(* PLC project marvel_common, Institute of Astronomy Onto 0.0.1 *)
(* stored: creationDateTime 2025-01-01T00:00:00.0, modificationDateTime 2025-01-01T00:00:00.0 *)

{attribute 'qualified_only'}
TYPE InitializationStates : (SHUTDOWN := 0, INITIALIZING := 1, INITIALIZING_FAILED := 2, INITIALIZED := 3, LOCKED := 4);
END_TYPE

{attribute 'qualified_only'}
TYPE OperatorStates : (NONE := 0, OBSERVER := 1, TECH := 2);
END_TYPE

{attribute 'qualified_only'}
TYPE OperatingStates : (AUTO := 0, MANUAL := 1);
END_TYPE

{attribute 'qualified_only'}
TYPE OperatingModeStates : (LOCAL := 0, REMOTE := 1);
END_TYPE

{attribute 'qualified_only'}
TYPE LimitSwitches : (POSITIVE_LIMIT_SWITCH := 0, NEGATIVE_LIMIT_SWITCH := 1);
END_TYPE

{attribute 'qualified_only'}
TYPE Units : (DEGREE := 0, RADIAN := 1, PERCENT := 2, RADIANS_PER_SECOND := 3, DEGREES_PER_SECOND := 4, MILLIMETERS_PER_SECOND := 5, REVOLUTIONS_PER_SECOND := 6, REVOLUTIONS_PER_MINUTE := 7, AMPS := 8, MILLIAMPS := 9, MILLIMETER := 10, MICROMETER := 11, DEGREES_CELSIUS := 12, KELVIN := 13, BAR := 14, PASCAL := 15, UNITLESS := 16, NEWTON := 17, DECANEWTON := 18, VOLT := 19, MILLIVOLT := 20, HERTZ := 21, G := 22, MILLIG := 23, NEWTONMETER := 24, ARCSECONDS := 25, ARCSECONDS_PER_SECOND := 26, RADIANS_PER_SQUARE_SECOND := 27, DEGREES_PER_SQUARE_SECOND := 28, ARCSECONDS_PER_SQUARE_SECOND := 29, METERS_PER_SECOND := 30, HECTOPASCAL := 31, SECONDS := 32, MINUTES := 33, MILLIMETERS_PER_HOUR := 34, HITS_PER_SQUARE_CENTIMETER := 35, HITS_PER_SQUARE_CENTIMETER_PER_HOUR := 36);
END_TYPE

{attribute 'qualified_only'}
TYPE RequestResults : (ACCEPTED := 0, REJECTED := 1);
END_TYPE

{attribute 'qualified_only'}
TYPE ApertureStatus : (unknown := 0, invalid_model := 1, open := 2, closed := 3, partiallyOpen := 4, undefined := 5) BYTE;
END_TYPE

{attribute 'qualified_only'}
TYPE BusyStatus : (unknown := 0, invalid_model := 1, idle := 2, busy := 3) BYTE;
END_TYPE

{attribute 'qualified_only'}
TYPE StartedStatus : (unknown := 0, invalid_model := 1, started := 2, notStarted := 3) BYTE;
END_TYPE

{attribute 'qualified_only'}
TYPE EnabledStatus : (unknown := 0, invalid_model := 1, enabled := 2, disabled := 3) BYTE;
END_TYPE

{attribute 'qualified_only'}
TYPE PoweredStatus : (unknown := 0, invalid_model := 1, enabled := 2, disabled := 3) BYTE;
END_TYPE

{attribute 'qualified_only'}
TYPE HealthStatus : (unknown := 0, invalid_model := 1, good := 2, warning := 3, bad := 4) BYTE;
END_TYPE

{attribute 'qualified_only'}
TYPE InitializationStatus : (unknown := 0, invalid_model := 1, shutdown := 2, initializing := 3, initializingFailed := 4, initialized := 5, locked := 6) BYTE;
END_TYPE

{attribute 'qualified_only'}
TYPE MotionStatus : (unknown := 0, invalid_model := 1, forward := 2, backward := 3, standstill := 4) BYTE;
END_TYPE

{attribute 'qualified_only'}
TYPE HiHiLoLoAlarmStatus : (unknown := 0, invalid_model := 1, disabled := 2, hiHi := 3, hi := 4, ok := 5, lo := 6, loLo := 7) BYTE;
END_TYPE

{attribute 'qualified_only'}
TYPE OpeningStatus : (unknown := 0, invalid_model := 1, opening := 2, closing := 3, standstill := 4) BYTE;
END_TYPE

{attribute 'qualified_only'}
TYPE OperatorStatus : (unknown := 0, invalid_model := 1, none := 2, tech := 3, observer := 4) BYTE;
END_TYPE

{attribute 'qualified_only'}
TYPE OperatingStatus : (unknown := 0, invalid_model := 1, auto := 2, manual := 3) BYTE;
END_TYPE

{attribute 'qualified_only'}
TYPE OperatingModeStatus : (unknown := 0, invalid_model := 1, local := 2, remote := 3) BYTE;
END_TYPE

{attribute 'qualified_only'}
TYPE ActivityStatus : (unknown := 0, invalid_model := 1, notRunning := 2, running := 3) BYTE;
END_TYPE

{attribute 'qualified_only'}
TYPE GigECameraParams : (_NONE_ := 0, fExposureTime := 1, fAcquisitionFrameRate := 2, fLinkAcquisitionFrameRate := 3, nGainSelector := 4, fGain := 5, nWidth := 6, nHeight := 7, nWidthMax := 8, nHeightMax := 9, nOffsetX := 10, nOffsetY := 11, nBinningSelector := 12, nBinningHorizontal := 13, nBinningVertical := 14, nTriggerSelector := 15, nTriggerMode := 16, fDeviceTemperature := 17, nAcquisitionMode := 18, fBlackLevel := 19, nBlackLevelAuto := 20, _END_ := 21);
END_TYPE

{attribute 'qualified_only'}
TYPE GigECameraSources : (CAMERA := 0, ACQUISITION_EXAMPLE := 1);
END_TYPE

{attribute 'qualified_only'}
TYPE GigECameraMultiTriggerAlgorithms : (SUM := 0);
END_TYPE

{attribute 'qualified_only'}
TYPE ELL14Command : (HOME_FWD := 0, HOME_BWD := 1, SEARCHFREQ_MOT1 := 2, SEARCHFREQ_MOT2 := 3, GET_STATUS := 4, GET_POSITION := 5, MOVE_ABS := 6, MOVE_REL := 7, CUSTOM := 8, _END_ := 9);
END_TYPE

{attribute 'qualified_only'}
TYPE ELL14StatusCode : (OK := 0, COMM_TIMEOUT := 1, MECH_TIMEOUT := 2, CMD_ERROR := 3, VALUE_OUT_OF_RANGE := 4, MOD_ISOLATED := 5, MOD_OUT_OF_ISOLATION := 6, INIT_ERROR := 7, THERMAL_ERROR := 8, BUSY := 9, SENSOR_ERROR := 10, MOTOR_ERROR := 11, OUT_OF_RANGE := 12, OVERCURRENT_ERROR := 13, UNKNOWN := 14);
END_TYPE

{attribute 'qualified_only'}
TYPE ActionActor : (NONE := 0, SEQUENCER := 1, MARVEL := 2, U := 3, U_DOME := 4, U_DOME_SHUTTER := 5, U_DOME_ROTATION := 6, U_TELESCOPE := 7, U_TELESCOPE_COVER := 8, U_TELESCOPE_M2 := 9, U_TELESCOPE_M3 := 10, U_FEM := 11, U_FEM_PWR_GUIDECAM := 12, U_FEM_PWR_FIBREVIEWCAM := 13, U_FEM_PWR_ADC := 14, U_FEM_PWR_TIPTILT := 15, U_FEM_CALMIRROR := 16, U_FEM_ADC1 := 17, U_FEM_ADC2 := 18, U_FEM_FIBRESELECTOR := 19, U_FEM_LED_HGF := 20, U_FEM_LED_UGF := 21, U_FEM_LED_HSF := 22, U_FEM_LED_USF := 23, U_FEM_GUIDECAM := 24, U_FEM_FIBREVIEWCAM := 25, U_FEM_TIPTILT := 26, _END_ := 27);
END_TYPE

{attribute 'qualified_only'}
TYPE ActionKind : (NONE := 0, SLEEP := 1, WAIT_FOR_COMPLETION := 2, INITIALIZE := 3, OPEN := 4, CLOSE := 5, STOP := 6, MOVE_TO_NUMBER := 7, MOVE_ABS_MM := 8, MOVE_ABS_DEG := 9, MOVE_AZI_ELE := 10, ENABLE := 11, DISABLE := 12, SET_ENABLED := 13, MOVE_REL_MM := 14, MOVE_REL_DEG := 15, SET_CURRENT := 16, SET_VOLTAGE := 17, SET_AXIS_VOLTAGE := 18, POWER := 19, _END_ := 20);
END_TYPE

{attribute 'qualified_only'}
TYPE ActionStatus : (IDLE := 0, REQUESTED := 1, BUSY := 2, DONE_SUCCESS := 3, DONE_ERROR := 4, DONE_ERROR_ABORTED := 5, DONE_ERROR_PROCESS_FAILED := 6, DONE_ERROR_INVALID_TYPE := 7, DONE_ERROR_INVALID_ARG := 8, DONE_ERROR_INVALID_ACTOR := 9);
END_TYPE

TYPE SequencerParts : STRUCT
  {attribute 'TcHmiSymbol.Show'}
  configManager : ConfigManager;  (* The config manager (to load/save/activate configuration data) *)
END_STRUCT;
END_TYPE

TYPE BaseAxisProcesses : STRUCT
  {attribute 'TcHmiSymbol.Show'}
  moveAbsolute : McMoveAbsoluteProcess;  (* Move absolute *)
  {attribute 'TcHmiSymbol.Show'}
  moveRelative : McMoveRelativeProcess;  (* Move relative *)
  {attribute 'TcHmiSymbol.Show'}
  moveVelocity : McMoveVelocityProcess;  (* Move at a constant velocity *)
  {attribute 'TcHmiSymbol.Show'}
  reset : McProcess;  (* Reset any errors *)
  {attribute 'TcHmiSymbol.Show'}
  stop : McProcess;  (* Stop any movement *)
  {attribute 'TcHmiSymbol.Show'}
  stopParametrized : McStopProcess;  (* Stop any movement *)
  {attribute 'TcHmiSymbol.Show'}
  power : McPowerProcess;  (* Power on/off the axis *)
  {attribute 'TcHmiSymbol.Show'}
  home : McProcess;  (* Peform a homing *)
  {attribute 'TcHmiSymbol.Show'}
  initialize : Process;  (* Start initializing the axis *)
  {attribute 'TcHmiSymbol.Show'}
  setPosition : McSetPositionProcess;  (* Set the axis position *)
  {attribute 'TcHmiSymbol.Show'}
  readParameter : McReadParameter;  (* Read a numerical parameter *)
  {attribute 'TcHmiSymbol.Show'}
  readBoolParameter : McReadBoolParameter;  (* Read a boolean parameter *)
  {attribute 'TcHmiSymbol.Show'}
  writeParameter : McWriteParameter;  (* Write a numerical parameter *)
  {attribute 'TcHmiSymbol.Show'}
  writeBoolParameter : McWriteBoolParameter;  (* Write a boolean parameter *)
END_STRUCT;
END_TYPE

TYPE IncrementalEncoderProcesses : STRUCT
  {attribute 'TcHmiSymbol.Show'}
  enableCounterResetC : Process;  (* Enable the counter reset on the C pulse *)
  {attribute 'TcHmiSymbol.Show'}
  disableCounterResetC : Process;  (* Disable the counter reset on the C pulse *)
END_STRUCT;
END_TYPE

TYPE SimpleRelayProcesses : STRUCT
  {attribute 'TcHmiSymbol.Show'}
  setEnabled : SetEnabledProcess;  (* Set the relay enabled or disabled *)
END_STRUCT;
END_TYPE

TYPE FuseProcesses : STRUCT
  {attribute 'TcHmiSymbol.Show'}
  setEnabled : SetEnabledProcess;  (* Set the relay enabled or disabled *)
  {attribute 'TcHmiSymbol.Show'}
  reset : Process;  (* Reset the fuse *)
END_STRUCT;
END_TYPE

TYPE LedProcesses : STRUCT
  {attribute 'TcHmiSymbol.Show'}
  setMilliAmps : ChangeSetpointProcess;  (* Set the output in milliampere *)
END_STRUCT;
END_TYPE

TYPE TipTiltProcesses : STRUCT
  {attribute 'TcHmiSymbol.Show'}
  setV1 : ChangeSetpointProcess;  (* Set the output in milliampere *)
  {attribute 'TcHmiSymbol.Show'}
  setV2 : ChangeSetpointProcess;  (* Set the output in milliampere *)
  {attribute 'TcHmiSymbol.Show'}
  setV3 : ChangeSetpointProcess;  (* Set the output in milliampere *)
END_STRUCT;
END_TYPE

TYPE ConfigManagerProcesses : STRUCT
  {attribute 'TcHmiSymbol.Show'}
  save : WriteXmlProcess;  (* Save the currently active config to disk *)
  {attribute 'TcHmiSymbol.Show'}
  load : ReadXmlProcess;  (* Load the config from disk *)
  {attribute 'TcHmiSymbol.Show'}
  activate : ActivateProcess;  (* Activate the loaded config *)
END_STRUCT;
END_TYPE

TYPE ModbusRTUBusProcesses : STRUCT
  {attribute 'TcHmiSymbol.Show'}
  readCoil : ModbusRTUBusReadCoilProcess;  (* Read coil *)
  {attribute 'TcHmiSymbol.Show'}
  writeCoil : ModbusRTUBusWriteCoilProcess;  (* Write coil *)
  {attribute 'TcHmiSymbol.Show'}
  readRegister : ModbusRTUBusReadRegisterProcess;  (* Read register *)
  {attribute 'TcHmiSymbol.Show'}
  writeRegister : ModbusRTUBusWriteRegisterProcess;  (* Write register *)
  {attribute 'TcHmiSymbol.Show'}
  diagnostics : ModbusRTUBusDiagnosticsProcess;  (* Diagnostics *)
END_STRUCT;
END_TYPE

TYPE GigECameraProcesses : STRUCT
  {attribute 'TcHmiSymbol.Show'}
  open : Process;  (* Open the camera *)
  {attribute 'TcHmiSymbol.Show'}
  close : Process;  (* Close the camera *)
  {attribute 'TcHmiSymbol.Show'}
  startAcquiring : Process;  (* Start acquiring frames *)
  {attribute 'TcHmiSymbol.Show'}
  stopAcquiring : Process;  (* Stop acquiring frames *)
  {attribute 'TcHmiSymbol.Show'}
  reset : Process;  (* Reset any errors *)
  {attribute 'TcHmiSymbol.Show'}
  setup : GigECameraSetupProcess;  (* Setup the camera with the given parameters *)
  {attribute 'TcHmiSymbol.Show'}
  setParam : GigECameraSetParamProcess;  (* Set a param value *)
  {attribute 'TcHmiSymbol.Show'}
  setParam2 : GigECameraSetParam2Process;  (* Set 2 param values (e.g. selector + value) *)
  {attribute 'TcHmiSymbol.Show'}
  trigger : Process;  (* Send a software trigger *)
  {attribute 'TcHmiSymbol.Show'}
  pulseTrigger : GigECameraPulseTrigger;  (* Send 2 software triggers, with a given duration in between *)
  {attribute 'TcHmiSymbol.Show'}
  multiTrigger : GigECameraMultiTriggerProcess;  (* Send multiple software triggers *)
  {attribute 'TcHmiSymbol.Show'}
  multiTriggerAbort : Process;  (* Abort the multi-trigger process *)
  {attribute 'TcHmiSymbol.Show'}
  setSource : GigECameraSetSourceProcess;  (* Set the camera source *)
END_STRUCT;
END_TYPE

TYPE ELL14StageProcesses : STRUCT
  {attribute 'TcHmiSymbol.Show'}
  moveAbs : Arg1LrealProcess;  (* Move absolute to the specified position in ° *)
  {attribute 'TcHmiSymbol.Show'}
  moveRel : Arg1LrealProcess;  (* Move relative with the specified offset in ° *)
  {attribute 'TcHmiSymbol.Show'}
  send : Ell114SendProcess;  (* Send raw command *)
END_STRUCT;
END_TYPE

TYPE SequencerProcesses : STRUCT
  {attribute 'TcHmiSymbol.Show'}
  selectEditable : IndexProcess;  (* Select the given sequence for editing *)
  {attribute 'TcHmiSymbol.Show'}
  selectRunnable : IndexProcess;  (* Select the given sequence for running *)
  {attribute 'TcHmiSymbol.Show'}
  start : IdProcess;  (* Select the given sequence for running (leave empty for current) + start running it *)
  {attribute 'TcHmiSymbol.Show'}
  stop : Process;  (* Stop the runnable sequence *)
  {attribute 'TcHmiSymbol.Show'}
  apply : Process;  (* Apply changes (activate, save, reload) *)
  {attribute 'TcHmiSymbol.Show'}
  cancel : Process;  (* Cancel changes (i.e. overwrite editableSeq) *)
END_STRUCT;
END_TYPE

TYPE BaseProcessStatuses : STRUCT
  {attribute 'OPC.UA.DA' := '1'}
  {attribute 'OPC.UA.DA.Access' := '1'}
  {attribute 'TcHmiSymbol.Show'}
  handle : UDINT;  (* Actual handle of the stat data *)
  {attribute 'OPC.UA.DA' := '1'}
  {attribute 'OPC.UA.DA.Access' := '1'}
  {attribute 'TcHmiSymbol.Show'}
  enabled : EnabledStatus;  (* Is the process enabled or not? *)
  {attribute 'OPC.UA.DA' := '1'}
  {attribute 'OPC.UA.DA.Access' := '1'}
  {attribute 'TcHmiSymbol.Show'}
  busy : BusyStatus;  (* Is the process busy or not? *)
  {attribute 'OPC.UA.DA' := '1'}
  {attribute 'OPC.UA.DA.Access' := '1'}
  {attribute 'TcHmiSymbol.Show'}
  health : HealthStatus;  (* Is the process in a healthy state or not? *)
  {attribute 'OPC.UA.DA' := '1'}
  {attribute 'OPC.UA.DA.Access' := '1'}
  {attribute 'TcHmiSymbol.Show'}
  started : StartedStatus;  (* Is the process started or not? *)
END_STRUCT;
END_TYPE

TYPE ProcessStepStatuses : STRUCT
  {attribute 'OPC.UA.DA' := '1'}
  {attribute 'OPC.UA.DA.Access' := '1'}
  {attribute 'TcHmiSymbol.Show'}
  enabled : EnabledStatus;  (* Is the process step enabled or not? *)
END_STRUCT;
END_TYPE

TYPE BaseAxisStatuses : STRUCT
  {attribute 'OPC.UA.DA' := '1'}
  {attribute 'OPC.UA.DA.Access' := '1'}
  {attribute 'TcHmiSymbol.Show'}
  busy : BusyStatus;  (* Is the NcAxis in a busy state? *)
  {attribute 'OPC.UA.DA' := '1'}
  {attribute 'OPC.UA.DA.Access' := '1'}
  {attribute 'TcHmiSymbol.Show'}
  health : HealthStatus;  (* Is the NcAxis in a healthy state? *)
  {attribute 'OPC.UA.DA' := '1'}
  {attribute 'OPC.UA.DA.Access' := '1'}
  {attribute 'TcHmiSymbol.Show'}
  powered : PoweredStatus;  (* Is the NcAxis powered? *)
  {attribute 'OPC.UA.DA' := '1'}
  {attribute 'OPC.UA.DA.Access' := '1'}
  {attribute 'TcHmiSymbol.Show'}
  extSetGen : EnabledStatus;  (* Is the NcAxis its external setpoint generator enabled? *)
  {attribute 'OPC.UA.DA' := '1'}
  {attribute 'OPC.UA.DA.Access' := '1'}
  {attribute 'TcHmiSymbol.Show'}
  motion : MotionStatus;  (* Is the NcAxis moving forward or backward or standing still? *)
END_STRUCT;
END_TYPE

TYPE SSIEncoderStatuses : STRUCT
  {attribute 'OPC.UA.DA' := '1'}
  {attribute 'OPC.UA.DA.Access' := '1'}
  {attribute 'TcHmiSymbol.Show'}
  health : HealthStatus;  (* Is the device in a healthy state? *)
END_STRUCT;
END_TYPE

TYPE IncrementalEncoderStatuses : STRUCT
  {attribute 'OPC.UA.DA' := '1'}
  {attribute 'OPC.UA.DA.Access' := '1'}
  {attribute 'TcHmiSymbol.Show'}
  health : HealthStatus;  (* Is the device in a healthy state? *)
  {attribute 'OPC.UA.DA' := '1'}
  {attribute 'OPC.UA.DA.Access' := '1'}
  {attribute 'TcHmiSymbol.Show'}
  busy : BusyStatus;  (* Is the device in a busy state? *)
END_STRUCT;
END_TYPE

TYPE EtherCatDeviceStatuses : STRUCT
  {attribute 'OPC.UA.DA' := '1'}
  {attribute 'OPC.UA.DA.Access' := '1'}
  {attribute 'TcHmiSymbol.Show'}
  health : HealthStatus;  (* Is the device in a healthy state? *)
END_STRUCT;
END_TYPE

TYPE CANopenBusStatuses : STRUCT
  {attribute 'OPC.UA.DA' := '1'}
  {attribute 'OPC.UA.DA.Access' := '1'}
  {attribute 'TcHmiSymbol.Show'}
  health : HealthStatus;  (* Is the device in a healthy state? *)
END_STRUCT;
END_TYPE

TYPE CurrentMeasurementStatuses : STRUCT
  {attribute 'OPC.UA.DA' := '1'}
  {attribute 'OPC.UA.DA.Access' := '1'}
  {attribute 'TcHmiSymbol.Show'}
  health : HealthStatus;  (* Is the measurement valid? *)
END_STRUCT;
END_TYPE

TYPE VoltageMeasurementStatuses : STRUCT
  {attribute 'OPC.UA.DA' := '1'}
  {attribute 'OPC.UA.DA.Access' := '1'}
  {attribute 'TcHmiSymbol.Show'}
  enabled : EnabledStatus;  (* Is the voltage being measured? *)
  {attribute 'OPC.UA.DA' := '1'}
  {attribute 'OPC.UA.DA.Access' := '1'}
  {attribute 'TcHmiSymbol.Show'}
  health : HealthStatus;  (* Is the measurement OK? *)
  {attribute 'OPC.UA.DA' := '1'}
  {attribute 'OPC.UA.DA.Access' := '1'}
  {attribute 'TcHmiSymbol.Show'}
  alarm : HiHiLoLoAlarmStatus;  (* Alarm status *)
END_STRUCT;
END_TYPE

TYPE SimpleTemperatureStatuses : STRUCT
  {attribute 'OPC.UA.DA' := '1'}
  {attribute 'OPC.UA.DA.Access' := '1'}
  {attribute 'TcHmiSymbol.Show'}
  enabled : EnabledStatus;  (* Is the temperature being measured? *)
  {attribute 'OPC.UA.DA' := '1'}
  {attribute 'OPC.UA.DA.Access' := '1'}
  {attribute 'TcHmiSymbol.Show'}
  health : HealthStatus;  (* Is the measurement OK? *)
  {attribute 'OPC.UA.DA' := '1'}
  {attribute 'OPC.UA.DA.Access' := '1'}
  {attribute 'TcHmiSymbol.Show'}
  alarm : HiHiLoLoAlarmStatus;  (* Alarm status *)
END_STRUCT;
END_TYPE

TYPE TemperatureMeasurementStatuses : STRUCT
  {attribute 'OPC.UA.DA' := '1'}
  {attribute 'OPC.UA.DA.Access' := '1'}
  {attribute 'TcHmiSymbol.Show'}
  enabled : EnabledStatus;  (* Is the temperature being measured? *)
  {attribute 'OPC.UA.DA' := '1'}
  {attribute 'OPC.UA.DA.Access' := '1'}
  {attribute 'TcHmiSymbol.Show'}
  health : HealthStatus;  (* Is the measurement OK? *)
  {attribute 'OPC.UA.DA' := '1'}
  {attribute 'OPC.UA.DA.Access' := '1'}
  {attribute 'TcHmiSymbol.Show'}
  alarm : HiHiLoLoAlarmStatus;  (* Alarm status *)
END_STRUCT;
END_TYPE

TYPE PressureMeasurementStatuses : STRUCT
  {attribute 'OPC.UA.DA' := '1'}
  {attribute 'OPC.UA.DA.Access' := '1'}
  {attribute 'TcHmiSymbol.Show'}
  enabled : EnabledStatus;  (* Is the pressure being measured? *)
  {attribute 'OPC.UA.DA' := '1'}
  {attribute 'OPC.UA.DA.Access' := '1'}
  {attribute 'TcHmiSymbol.Show'}
  health : HealthStatus;  (* Is the measurement OK? *)
  {attribute 'OPC.UA.DA' := '1'}
  {attribute 'OPC.UA.DA.Access' := '1'}
  {attribute 'TcHmiSymbol.Show'}
  alarm : HiHiLoLoAlarmStatus;  (* Alarm status *)
END_STRUCT;
END_TYPE

TYPE FrequencyMeasurementStatuses : STRUCT
  {attribute 'OPC.UA.DA' := '1'}
  {attribute 'OPC.UA.DA.Access' := '1'}
  {attribute 'TcHmiSymbol.Show'}
  enabled : EnabledStatus;  (* Is the frequency being measured? *)
  {attribute 'OPC.UA.DA' := '1'}
  {attribute 'OPC.UA.DA.Access' := '1'}
  {attribute 'TcHmiSymbol.Show'}
  health : HealthStatus;  (* Is the measurement OK? *)
  {attribute 'OPC.UA.DA' := '1'}
  {attribute 'OPC.UA.DA.Access' := '1'}
  {attribute 'TcHmiSymbol.Show'}
  alarm : HiHiLoLoAlarmStatus;  (* Alarm status *)
END_STRUCT;
END_TYPE

TYPE GForceMeasurementStatuses : STRUCT
  {attribute 'OPC.UA.DA' := '1'}
  {attribute 'OPC.UA.DA.Access' := '1'}
  {attribute 'TcHmiSymbol.Show'}
  health : HealthStatus;  (* Is the measurement OK? *)
END_STRUCT;
END_TYPE

TYPE RelativeHumidityMeasurementStatuses : STRUCT
  {attribute 'OPC.UA.DA' := '1'}
  {attribute 'OPC.UA.DA.Access' := '1'}
  {attribute 'TcHmiSymbol.Show'}
  enabled : EnabledStatus;  (* Is the relative humidity being measured? *)
  {attribute 'OPC.UA.DA' := '1'}
  {attribute 'OPC.UA.DA.Access' := '1'}
  {attribute 'TcHmiSymbol.Show'}
  health : HealthStatus;  (* Is the measurement OK? *)
  {attribute 'OPC.UA.DA' := '1'}
  {attribute 'OPC.UA.DA.Access' := '1'}
  {attribute 'TcHmiSymbol.Show'}
  alarm : HiHiLoLoAlarmStatus;  (* Alarm status *)
END_STRUCT;
END_TYPE

TYPE ForceMeasurementStatuses : STRUCT
  {attribute 'OPC.UA.DA' := '1'}
  {attribute 'OPC.UA.DA.Access' := '1'}
  {attribute 'TcHmiSymbol.Show'}
  enabled : EnabledStatus;  (* Is the force being measured? *)
  {attribute 'OPC.UA.DA' := '1'}
  {attribute 'OPC.UA.DA.Access' := '1'}
  {attribute 'TcHmiSymbol.Show'}
  health : HealthStatus;  (* Is the measurement OK? *)
  {attribute 'OPC.UA.DA' := '1'}
  {attribute 'OPC.UA.DA.Access' := '1'}
  {attribute 'TcHmiSymbol.Show'}
  alarm : HiHiLoLoAlarmStatus;  (* Alarm status *)
END_STRUCT;
END_TYPE

TYPE LinearPositionMeasurement16Statuses : STRUCT
  {attribute 'OPC.UA.DA' := '1'}
  {attribute 'OPC.UA.DA.Access' := '1'}
  {attribute 'TcHmiSymbol.Show'}
  enabled : EnabledStatus;  (* Is the position being measured? *)
  {attribute 'OPC.UA.DA' := '1'}
  {attribute 'OPC.UA.DA.Access' := '1'}
  {attribute 'TcHmiSymbol.Show'}
  health : HealthStatus;  (* Is the measurement OK? *)
  {attribute 'OPC.UA.DA' := '1'}
  {attribute 'OPC.UA.DA.Access' := '1'}
  {attribute 'TcHmiSymbol.Show'}
  alarm : HiHiLoLoAlarmStatus;  (* Alarm status *)
END_STRUCT;
END_TYPE

TYPE LinearPositionMeasurementU32Statuses : STRUCT
  {attribute 'OPC.UA.DA' := '1'}
  {attribute 'OPC.UA.DA.Access' := '1'}
  {attribute 'TcHmiSymbol.Show'}
  enabled : EnabledStatus;  (* Is the position being measured? *)
  {attribute 'OPC.UA.DA' := '1'}
  {attribute 'OPC.UA.DA.Access' := '1'}
  {attribute 'TcHmiSymbol.Show'}
  health : HealthStatus;  (* Is the measurement OK? *)
  {attribute 'OPC.UA.DA' := '1'}
  {attribute 'OPC.UA.DA.Access' := '1'}
  {attribute 'TcHmiSymbol.Show'}
  alarm : HiHiLoLoAlarmStatus;  (* Alarm status *)
END_STRUCT;
END_TYPE

TYPE SimpleRelayStatuses : STRUCT
  {attribute 'OPC.UA.DA' := '1'}
  {attribute 'OPC.UA.DA.Access' := '1'}
  {attribute 'TcHmiSymbol.Show'}
  busy : BusyStatus;  (* Is the SimpleRelay in a busy state? *)
END_STRUCT;
END_TYPE

TYPE FuseStatuses : STRUCT
  {attribute 'OPC.UA.DA' := '1'}
  {attribute 'OPC.UA.DA.Access' := '1'}
  {attribute 'TcHmiSymbol.Show'}
  busy : BusyStatus;  (* Is the Fuse in a busy state? *)
  {attribute 'OPC.UA.DA' := '1'}
  {attribute 'OPC.UA.DA.Access' := '1'}
  {attribute 'TcHmiSymbol.Show'}
  health : HealthStatus;  (* Is the Fuse in a healthy state? *)
END_STRUCT;
END_TYPE

TYPE LedStatuses : STRUCT
  {attribute 'OPC.UA.DA' := '1'}
  {attribute 'OPC.UA.DA.Access' := '1'}
  {attribute 'TcHmiSymbol.Show'}
  busy : BusyStatus;  (* Is the Led in a busy state? *)
END_STRUCT;
END_TYPE

TYPE TipTiltStatuses : STRUCT
  {attribute 'OPC.UA.DA' := '1'}
  {attribute 'OPC.UA.DA.Access' := '1'}
  {attribute 'TcHmiSymbol.Show'}
  busy : BusyStatus;  (* Is the TipTilt in a busy state? *)
END_STRUCT;
END_TYPE

TYPE ConfigManagerStatuses : STRUCT
  {attribute 'OPC.UA.DA' := '1'}
  {attribute 'OPC.UA.DA.Access' := '1'}
  {attribute 'TcHmiSymbol.Show'}
  busy : BusyStatus;  (* Is the config manager in a busy state? *)
  {attribute 'OPC.UA.DA' := '1'}
  {attribute 'OPC.UA.DA.Access' := '1'}
  {attribute 'TcHmiSymbol.Show'}
  health : HealthStatus;  (* Is the config manager in a healthy state? *)
END_STRUCT;
END_TYPE

TYPE ModbusRTUBusStatuses : STRUCT
  {attribute 'OPC.UA.DA' := '1'}
  {attribute 'OPC.UA.DA.Access' := '1'}
  {attribute 'TcHmiSymbol.Show'}
  busy : BusyStatus;  (* Is the config manager in a busy state? *)
END_STRUCT;
END_TYPE

TYPE GigECameraStatuses : STRUCT
  {attribute 'OPC.UA.DA' := '1'}
  {attribute 'OPC.UA.DA.Access' := '1'}
  {attribute 'TcHmiSymbol.Show'}
  health : HealthStatus;
  {attribute 'OPC.UA.DA' := '1'}
  {attribute 'OPC.UA.DA.Access' := '1'}
  {attribute 'TcHmiSymbol.Show'}
  busy : BusyStatus;
END_STRUCT;
END_TYPE

TYPE ELL14StageStatuses : STRUCT
  {attribute 'OPC.UA.DA' := '1'}
  {attribute 'OPC.UA.DA.Access' := '1'}
  {attribute 'TcHmiSymbol.Show'}
  health : HealthStatus;  (* Is the device in a healthy state? *)
  {attribute 'OPC.UA.DA' := '1'}
  {attribute 'OPC.UA.DA.Access' := '1'}
  {attribute 'TcHmiSymbol.Show'}
  busy : BusyStatus;  (* Is the device in a busy state? *)
END_STRUCT;
END_TYPE

TYPE SequencerStatuses : STRUCT
  {attribute 'OPC.UA.DA' := '1'}
  {attribute 'OPC.UA.DA.Access' := '1'}
  {attribute 'TcHmiSymbol.Show'}
  health : HealthStatus;  (* Is the sequencer in a healthy state? *)
  {attribute 'OPC.UA.DA' := '1'}
  {attribute 'OPC.UA.DA.Access' := '1'}
  {attribute 'TcHmiSymbol.Show'}
  busy : BusyStatus;  (* Is the sequencer in a busy state? *)
END_STRUCT;
END_TYPE

TYPE EventManagerStatuses : STRUCT
  {attribute 'OPC.UA.DA' := '1'}
  {attribute 'OPC.UA.DA.Access' := '1'}
  {attribute 'TcHmiSymbol.Show'}
  health : HealthStatus;  (* Is the event manager in a healthy state? *)
  {attribute 'OPC.UA.DA' := '1'}
  {attribute 'OPC.UA.DA.Access' := '1'}
  {attribute 'TcHmiSymbol.Show'}
  busy : BusyStatus;  (* Is the event manager in a busy state? *)
END_STRUCT;
END_TYPE

TYPE HiHiLoLoAlarmConfig : STRUCT
  {attribute 'TcHmiSymbol.Show'}
  enabled : BOOL;  (* Is the alarm enabled? *)
  {attribute 'TcHmiSymbol.Show'}
  loLo : LREAL;  (* LowLow alarm limit (produces ERROR) *)
  {attribute 'TcHmiSymbol.Show'}
  lo : LREAL;  (* Low alarm limit (produces WARNING) *)
  {attribute 'TcHmiSymbol.Show'}
  hi : LREAL;  (* High alarm limit (produces WARNING) *)
  {attribute 'TcHmiSymbol.Show'}
  hiHi : LREAL;  (* HighHigh alarm limit (produces ERROR) *)
END_STRUCT;
END_TYPE

TYPE MeasurementConfig : STRUCT
  {attribute 'TcHmiSymbol.Show'}
  enabled : BOOL;  (* Is the quantity being measured? (Can be false e.g. if the sensor is deliberately not connected (yet).) *)
  {attribute 'TcHmiSymbol.Show'}
  gain : LREAL := 1.0;  (* Gain to be applied to the measured value (default: 1 = no gain) *)
  {attribute 'TcHmiSymbol.Show'}
  offset : LREAL;  (* Offset to be added to the measured value (default: 0 = no offset) *)
  {attribute 'TcHmiSymbol.Show'}
  alarms : HiHiLoLoAlarmConfig;  (* Config *)
END_STRUCT;
END_TYPE

TYPE ActionArgConfig : STRUCT
  {attribute 'TcHmiSymbol.Show'}
  str : STRING(30);  (* Arg as a STRING *)
  {attribute 'TcHmiSymbol.Show'}
  f : LREAL;  (* Arg as an LREAL *)
  {attribute 'TcHmiSymbol.Show'}
  n : DINT;  (* Arg as an DINT *)
  {attribute 'TcHmiSymbol.Show'}
  b : BOOL;  (* Arg as an BOOL *)
END_STRUCT;
END_TYPE

TYPE ActionStringConfig : STRUCT
  {attribute 'TcHmiSymbol.Show'}
  actor : STRING(50);  (* Actor of the action *)
  {attribute 'TcHmiSymbol.Show'}
  kind : STRING(50);  (* Kind of the action *)
  {attribute 'TcHmiSymbol.Show'}
  block : BOOL := TRUE;  (* TRUE if the action is blocking (for the next one) *)
  {attribute 'TcHmiSymbol.Show'}
  args : ARRAY[0..1] OF ActionArgConfig;  (* Arguments *)
  {attribute 'TcHmiSymbol.Show'}
  u1 : BOOL := TRUE;  (* Apply to U1 (if relevant) *)
  {attribute 'TcHmiSymbol.Show'}
  u2 : BOOL := TRUE;  (* Apply to U2 (if relevant) *)
  {attribute 'TcHmiSymbol.Show'}
  u3 : BOOL := TRUE;  (* Apply to U3 (if relevant) *)
  {attribute 'TcHmiSymbol.Show'}
  u4 : BOOL := TRUE;  (* Apply to U4 (if relevant) *)
END_STRUCT;
END_TYPE

TYPE ActionEnumConfig : STRUCT
  {attribute 'TcHmiSymbol.Show'}
  actor : ActionActor;  (* Actor of the action *)
  {attribute 'TcHmiSymbol.Show'}
  kind : ActionKind;  (* Kind of the action *)
  {attribute 'TcHmiSymbol.Show'}
  block : BOOL := TRUE;  (* TRUE if the action is blocking (for the next one) *)
  {attribute 'TcHmiSymbol.Show'}
  args : ARRAY[0..1] OF ActionArgConfig;  (* Arguments *)
  {attribute 'TcHmiSymbol.Show'}
  u1 : BOOL := TRUE;  (* Apply to U1 (if relevant) *)
  {attribute 'TcHmiSymbol.Show'}
  u2 : BOOL := TRUE;  (* Apply to U2 (if relevant) *)
  {attribute 'TcHmiSymbol.Show'}
  u3 : BOOL := TRUE;  (* Apply to U3 (if relevant) *)
  {attribute 'TcHmiSymbol.Show'}
  u4 : BOOL := TRUE;  (* Apply to U4 (if relevant) *)
END_STRUCT;
END_TYPE

TYPE SequenceStringConfig_M : STRUCT
  {attribute 'TcHmiSymbol.Show'}
  id : STRING(16);  (* ID of the sequence *)
  {attribute 'TcHmiSymbol.Show'}
  length : INT;  (* Number of actions *)
  {attribute 'TcHmiSymbol.Show'}
  actions : ARRAY[0..29] OF ActionStringConfig;  (* Actions *)
END_STRUCT;
END_TYPE

TYPE SequenceEnumConfig_M : STRUCT
  {attribute 'TcHmiSymbol.Show'}
  id : STRING(16);  (* ID of the sequence *)
  {attribute 'TcHmiSymbol.Show'}
  length : INT;  (* Number of actions *)
  {attribute 'TcHmiSymbol.Show'}
  configs : ARRAY[0..29] OF ActionEnumConfig;  (* Actions *)
END_STRUCT;
END_TYPE

TYPE QuantityValue : STRUCT
  {attribute 'TcHmiSymbol.Show'}
  value : LREAL;  (* Numeric value *)
END_STRUCT;
END_TYPE

TYPE AngularPosition : STRUCT
  {attribute 'TcHmiSymbol.Show'}
  radians : QuantityValue;  (* Angular position in radians *)
  {attribute 'TcHmiSymbol.Show'}
  degrees : QuantityValue;  (* Angular position in degrees *)
END_STRUCT;
END_TYPE

TYPE LinearPosition : STRUCT
  {attribute 'TcHmiSymbol.Show'}
  millimeters : QuantityValue;  (* Linear position in millimeters *)
  {attribute 'TcHmiSymbol.Show'}
  micrometers : QuantityValue;  (* Linear position in micrometers *)
END_STRUCT;
END_TYPE

TYPE AngularVelocity : STRUCT
  {attribute 'TcHmiSymbol.Show'}
  radiansPerSecond : QuantityValue;  (* Angular velocity in radians per second *)
  {attribute 'TcHmiSymbol.Show'}
  degreesPerSecond : QuantityValue;  (* Angular velocity in degrees per second *)
END_STRUCT;
END_TYPE

TYPE AngularAcceleration : STRUCT
  {attribute 'TcHmiSymbol.Show'}
  radiansPerSquareSecond : QuantityValue;  (* Angular velocity in radians per second^2 *)
  {attribute 'TcHmiSymbol.Show'}
  degreesPerSquareSecond : QuantityValue;  (* Angular velocity in degrees per second^2 *)
END_STRUCT;
END_TYPE

TYPE LinearVelocity : STRUCT
  {attribute 'TcHmiSymbol.Show'}
  millimetersPerSecond : QuantityValue;  (* Linear velocity in millimeters per second *)
END_STRUCT;
END_TYPE

TYPE Voltage : STRUCT
  {attribute 'TcHmiSymbol.Show'}
  volt : QuantityValue;  (* Voltage in Volt *)
  {attribute 'TcHmiSymbol.Show'}
  milliVolt : QuantityValue;  (* Voltage in millivolt *)
END_STRUCT;
END_TYPE

TYPE GForce : STRUCT
  {attribute 'TcHmiSymbol.Show'}
  g : QuantityValue;  (* Acceleration in g units *)
  {attribute 'TcHmiSymbol.Show'}
  milliG : QuantityValue;  (* Acceleration in in milli g units *)
END_STRUCT;
END_TYPE

TYPE Current : STRUCT
  {attribute 'TcHmiSymbol.Show'}
  amps : QuantityValue;  (* Current in amps *)
  {attribute 'TcHmiSymbol.Show'}
  milliAmps : QuantityValue;  (* Current in milliamps *)
END_STRUCT;
END_TYPE

TYPE Torque : STRUCT
  {attribute 'TcHmiSymbol.Show'}
  newtonmeter : QuantityValue;  (* Torque in Nm *)
END_STRUCT;
END_TYPE

TYPE TorqueLimit : STRUCT
  {attribute 'TcHmiSymbol.Show'}
  unitless : QuantityValue;  (* Torque limit as a unitless fraction *)
  {attribute 'TcHmiSymbol.Show'}
  percent : QuantityValue;  (* Torque limit in percent *)
  {attribute 'TcHmiSymbol.Show'}
  newtonmeter : QuantityValue;  (* Torque in Nm *)
END_STRUCT;
END_TYPE

TYPE Duration : STRUCT
  {attribute 'TcHmiSymbol.Show'}
  seconds : QuantityValue;  (* Duration in seconds *)
  {attribute 'TcHmiSymbol.Show'}
  minutes : QuantityValue;  (* Duration in minutes *)
END_STRUCT;
END_TYPE

TYPE Temperature : STRUCT
  {attribute 'TcHmiSymbol.Show'}
  celsius : QuantityValue;  (* Temperature in degrees Celsius *)
  {attribute 'TcHmiSymbol.Show'}
  kelvin : QuantityValue;  (* Temperature in Kelvin *)
END_STRUCT;
END_TYPE

TYPE Pressure : STRUCT
  {attribute 'TcHmiSymbol.Show'}
  bar : QuantityValue;  (* Pressure in Bar *)
  {attribute 'TcHmiSymbol.Show'}
  pascal : QuantityValue;  (* Pressure in Pascal *)
  {attribute 'TcHmiSymbol.Show'}
  hectoPascal : QuantityValue;  (* Pressure in HectoPascal *)
END_STRUCT;
END_TYPE

TYPE Frequency : STRUCT
  {attribute 'TcHmiSymbol.Show'}
  hertz : QuantityValue;  (* Frequency in Hertz *)
END_STRUCT;
END_TYPE

TYPE Force : STRUCT
  {attribute 'TcHmiSymbol.Show'}
  newton : QuantityValue;  (* Force in Newton *)
  {attribute 'TcHmiSymbol.Show'}
  decaNewton : QuantityValue;  (* Force in decaNewton *)
END_STRUCT;
END_TYPE

TYPE Fraction : STRUCT
  {attribute 'TcHmiSymbol.Show'}
  unitless : QuantityValue;  (* Fraction as a unitless value between 0 and 1 *)
  {attribute 'TcHmiSymbol.Show'}
  percent : QuantityValue;  (* Fraction as a percentage value between 0 and 100 *)
END_STRUCT;
END_TYPE

TYPE AtomicRequest : STRUCT
  {attribute 'TcHmiSymbol.Show'}
  handle : UDINT;  (* Handle of the request *)
  {attribute 'TcHmiSymbol.Show'}
  request : BOOL;  (* Write TRUE to request the start of the process *)
END_STRUCT;
END_TYPE

TYPE MercatorMeteoExchange : STRUCT
  {attribute 'TcHmiSymbol.Show'}
  mercatorServiceHealthy : BOOL;  (* TRUE if the Mercator service health is Good *)
  {attribute 'TcHmiSymbol.Show'}
  windSpeedMinimum : LREAL;  (* Wind speed minimum *)
  {attribute 'TcHmiSymbol.Show'}
  windSpeedAverage : LREAL;  (* Wind speed average *)
  {attribute 'TcHmiSymbol.Show'}
  windSpeedMaximum : LREAL;  (* Wind speed maximum *)
  {attribute 'TcHmiSymbol.Show'}
  windDirectionMinimum : LREAL;  (* Wind direction minimum *)
  {attribute 'TcHmiSymbol.Show'}
  windDirectionAverage : LREAL;  (* Wind direction average *)
  {attribute 'TcHmiSymbol.Show'}
  windDirectionMaximum : LREAL;  (* Wind direction maximum *)
  {attribute 'TcHmiSymbol.Show'}
  airPressure : LREAL;  (* Air pressure *)
  {attribute 'TcHmiSymbol.Show'}
  airTemperature : LREAL;  (* Air temperature *)
  {attribute 'TcHmiSymbol.Show'}
  internalTemperature : LREAL;  (* Internal temperature *)
  {attribute 'TcHmiSymbol.Show'}
  relativeHumidity : LREAL;  (* Relative humidity *)
  {attribute 'TcHmiSymbol.Show'}
  rainAccumulation : LREAL;  (* Rain accumulation *)
  {attribute 'TcHmiSymbol.Show'}
  rainDuration : LREAL;  (* Rain duration *)
  {attribute 'TcHmiSymbol.Show'}
  rainIntensity : LREAL;  (* Rain intensity *)
  {attribute 'TcHmiSymbol.Show'}
  rainPeakIntensity : LREAL;  (* Rain peak intensity *)
  {attribute 'TcHmiSymbol.Show'}
  hailAccumulation : LREAL;  (* Hail accumulation *)
  {attribute 'TcHmiSymbol.Show'}
  hailDuration : LREAL;  (* Hail duration *)
  {attribute 'TcHmiSymbol.Show'}
  hailIntensity : LREAL;  (* Hail intensity *)
  {attribute 'TcHmiSymbol.Show'}
  hailPeakIntensity : LREAL;  (* Hail peak intensity *)
  {attribute 'TcHmiSymbol.Show'}
  heatingTemperature : LREAL;  (* Heating temperature *)
  {attribute 'TcHmiSymbol.Show'}
  heatingVoltage : LREAL;  (* Heating voltage *)
  {attribute 'TcHmiSymbol.Show'}
  supplyVoltage : LREAL;  (* Supply voltage *)
  {attribute 'TcHmiSymbol.Show'}
  referenceVoltage : LREAL;  (* Reference voltage *)
  {attribute 'TcHmiSymbol.Show'}
  dewpoint : LREAL;  (* Calculated dewpoint *)
  {attribute 'TcHmiSymbol.Show'}
  windSpeedMinimumValid : BIT;  (* TRUE if Wind speed minimum is valid *)
  {attribute 'TcHmiSymbol.Show'}
  windSpeedAverageValid : BIT;  (* TRUE if Wind speed average is valid *)
  {attribute 'TcHmiSymbol.Show'}
  windSpeedMaximumValid : BIT;  (* TRUE if Wind speed maximum is valid *)
  {attribute 'TcHmiSymbol.Show'}
  windDirectionMinimumValid : BIT;  (* TRUE if Wind direction minimum is valid *)
  {attribute 'TcHmiSymbol.Show'}
  windDirectionAverageValid : BIT;  (* TRUE if Wind direction average is valid *)
  {attribute 'TcHmiSymbol.Show'}
  windDirectionMaximumValid : BIT;  (* TRUE if Wind direction maximum is valid *)
  {attribute 'TcHmiSymbol.Show'}
  airPressureValid : BIT;  (* TRUE if Air pressure is valid *)
  {attribute 'TcHmiSymbol.Show'}
  airTemperatureValid : BIT;  (* TRUE if Air temperature is valid *)
  {attribute 'TcHmiSymbol.Show'}
  internalTemperatureValid : BIT;  (* TRUE if Internal temperature is valid *)
  {attribute 'TcHmiSymbol.Show'}
  relativeHumidityValid : BIT;  (* TRUE if Relative humidity is valid *)
  {attribute 'TcHmiSymbol.Show'}
  rainAccumulationValid : BIT;  (* TRUE if Rain accumulation is valid *)
  {attribute 'TcHmiSymbol.Show'}
  rainDurationValid : BIT;  (* TRUE if Rain duration is valid *)
  {attribute 'TcHmiSymbol.Show'}
  rainIntensityValid : BIT;  (* TRUE if Rain intensity is valid *)
  {attribute 'TcHmiSymbol.Show'}
  rainPeakIntensityValid : BIT;  (* TRUE if Rain peak intensity is valid *)
  {attribute 'TcHmiSymbol.Show'}
  hailAccumulationValid : BIT;  (* TRUE if Hail accumulation is valid *)
  {attribute 'TcHmiSymbol.Show'}
  hailDurationValid : BIT;  (* TRUE if Hail duration is valid *)
  {attribute 'TcHmiSymbol.Show'}
  hailIntensityValid : BIT;  (* TRUE if Hail intensity is valid *)
  {attribute 'TcHmiSymbol.Show'}
  hailPeakIntensityValid : BIT;  (* TRUE if Hail peak intensity is valid *)
  {attribute 'TcHmiSymbol.Show'}
  heatingTemperatureValid : BIT;  (* TRUE if Heating temperature is valid *)
  {attribute 'TcHmiSymbol.Show'}
  heatingVoltageValid : BIT;  (* TRUE if Heating voltage is valid *)
  {attribute 'TcHmiSymbol.Show'}
  supplyVoltageValid : BIT;  (* TRUE if Supply voltage is valid *)
  {attribute 'TcHmiSymbol.Show'}
  referenceVoltageValid : BIT;  (* TRUE if Reference voltage is valid *)
  {attribute 'TcHmiSymbol.Show'}
  dewpointValid : BIT;  (* TRUE if Calculated dewpoint is valid *)
END_STRUCT;
END_TYPE

TYPE SequenceStatus_M : STRUCT
  {attribute 'TcHmiSymbol.Show'}
  actions : ARRAY[0..29] OF ActionStatus;
END_STRUCT;
END_TYPE

TYPE SequencerStringConfig : STRUCT
  {attribute 'TcHmiSymbol.Show'}
  seqs : ARRAY[0..50] OF SequenceStringConfig_M;  (* Sequences to be serialized to disk (with strings instead of enums) *)
END_STRUCT;
END_TYPE

TYPE SequencerEnumConfig : STRUCT
  {attribute 'TcHmiSymbol.Show'}
  seqs : ARRAY[0..50] OF SequenceEnumConfig_M;  (* Sequences after deserialization (with enums instead of strings) *)
END_STRUCT;
END_TYPE

TYPE IdProcessArgs : STRUCT
  {attribute 'TcHmiSymbol.Show'}
  id : STRING(30);
END_STRUCT;
END_TYPE

TYPE IndexProcessArgs : STRUCT
  {attribute 'TcHmiSymbol.Show'}
  id : UINT;
END_STRUCT;
END_TYPE

TYPE ChangeSetpointProcessArgs : STRUCT
  {attribute 'TcHmiSymbol.Show'}
  setpoint : LREAL;  (* New setpoint value *)
END_STRUCT;
END_TYPE

TYPE ChangeParameterProcessArgs : STRUCT
  {attribute 'TcHmiSymbol.Show'}
  parameter : LREAL;  (* New parameter value *)
END_STRUCT;
END_TYPE

TYPE McMoveAbsoluteProcessArgs : STRUCT
  {attribute 'TcHmiSymbol.Show'}
  position : LREAL;  (* New position setpoint *)
  {attribute 'TcHmiSymbol.Show'}
  maxVelocity : LREAL;  (* Maximum velocity *)
END_STRUCT;
END_TYPE

TYPE McMoveRelativeProcessArgs : STRUCT
  {attribute 'TcHmiSymbol.Show'}
  distance : LREAL;  (* Distance to move *)
  {attribute 'TcHmiSymbol.Show'}
  maxVelocity : LREAL;  (* Maximum velocity *)
END_STRUCT;
END_TYPE

TYPE McPowerProcessArgs : STRUCT
  {attribute 'TcHmiSymbol.Show'}
  enable : BOOL;  (* Enable the power or not *)
END_STRUCT;
END_TYPE

TYPE McSetPositionProcessArgs : STRUCT
  {attribute 'TcHmiSymbol.Show'}
  value : LREAL;  (* New position to be taken over by the encoder *)
END_STRUCT;
END_TYPE

TYPE McStopProcessArgs : STRUCT
  {attribute 'TcHmiSymbol.Show'}
  deceleration : LREAL;  (* Deceleration (use 0 for default). If non zero, then also jerk must be non zero! *)
  {attribute 'TcHmiSymbol.Show'}
  jerk : LREAL;  (* Jerk (use 0 for default). If non zero, then also deceleration must be non zero! *)
END_STRUCT;
END_TYPE

TYPE McMoveVelocityProcessArgs : STRUCT
  {attribute 'TcHmiSymbol.Show'}
  value : LREAL;  (* New velocity *)
END_STRUCT;
END_TYPE

TYPE SetEnabledProcessArgs : STRUCT
  {attribute 'TcHmiSymbol.Show'}
  enabled : BOOL;  (* True to enable, false to disable *)
END_STRUCT;
END_TYPE

TYPE McWriteParameterArgs : STRUCT
  {attribute 'TcHmiSymbol.Show'}
  parameterNumber : INT;  (* Number of the parameter *)
  {attribute 'TcHmiSymbol.Show'}
  value : LREAL;  (* Value to write *)
END_STRUCT;
END_TYPE

TYPE McReadParameterArgs : STRUCT
  {attribute 'TcHmiSymbol.Show'}
  parameterNumber : INT;  (* Number of the parameter *)
END_STRUCT;
END_TYPE

TYPE McWriteBoolParameterArgs : STRUCT
  {attribute 'TcHmiSymbol.Show'}
  parameterNumber : INT;  (* Number of the parameter *)
  {attribute 'TcHmiSymbol.Show'}
  value : BOOL;  (* Value to write *)
END_STRUCT;
END_TYPE

TYPE McReadBoolParameterArgs : STRUCT
  {attribute 'TcHmiSymbol.Show'}
  parameterNumber : INT;  (* Number of the parameter *)
END_STRUCT;
END_TYPE

TYPE McProbeArgs : STRUCT
  {attribute 'TcHmiSymbol.Show'}
  risingEdge : BOOL;  (* True to probe the rising edge, false to probe the falling edge *)
  {attribute 'TcHmiSymbol.Show'}
  timeout : LREAL;  (* Timeout, in seconds. After this timeout, probing is aborted. timeout <= 0 means endless probing. *)
END_STRUCT;
END_TYPE

TYPE ChangeOperatingStateProcessArgs : STRUCT
  {attribute 'TcHmiSymbol.Show'}
  state : OperatingStates;  (* New operating state (e.g. AUTO, MANUAL) *)
END_STRUCT;
END_TYPE

TYPE ChangeOperatorStateProcessArgs : STRUCT
  {attribute 'TcHmiSymbol.Show'}
  state : OperatorStates;  (* New operator state (e.g. OBSERVER, TECH, ...) *)
  {attribute 'TcHmiSymbol.Show'}
  password : STRING(12);  (* Password (only sometimes required, e.g. to go from OBSERVER to TECH) *)
END_STRUCT;
END_TYPE

TYPE ChangeOperatingModeStateProcessArgs : STRUCT
  {attribute 'TcHmiSymbol.Show'}
  state : OperatingModeStates;  (* New operating state (e.g. LOCAL, REMOTE) *)
END_STRUCT;
END_TYPE

TYPE ReadXmlProcessArgs : STRUCT
  {attribute 'TcHmiSymbol.Show'}
  filePath : STRING(30);  (* Full path of the filename to read *)
END_STRUCT;
END_TYPE

TYPE WriteXmlProcessArgs : STRUCT
  {attribute 'TcHmiSymbol.Show'}
  filePath : STRING(30);  (* Full path of the filename to write *)
END_STRUCT;
END_TYPE

TYPE ModbusRTUBusReadCoilProcessArgs : STRUCT
  {attribute 'TcHmiSymbol.Show'}
  unitID : USINT;  (* Modbus station address (1..247) *)
  {attribute 'TcHmiSymbol.Show'}
  address : UINT;  (* Modbus data address *)
END_STRUCT;
END_TYPE

TYPE ModbusRTUBusWriteCoilProcessArgs : STRUCT
  {attribute 'TcHmiSymbol.Show'}
  unitID : USINT;  (* Modbus station address (1..247) *)
  {attribute 'TcHmiSymbol.Show'}
  address : UINT;  (* Modbus data address *)
  {attribute 'TcHmiSymbol.Show'}
  value : BOOL;  (* Value to write on the coil *)
END_STRUCT;
END_TYPE

TYPE ModbusRTUBusReadRegisterProcessArgs : STRUCT
  {attribute 'TcHmiSymbol.Show'}
  unitID : USINT;  (* Modbus station address (1..247) *)
  {attribute 'TcHmiSymbol.Show'}
  address : UINT;  (* Modbus data address *)
END_STRUCT;
END_TYPE

TYPE ModbusRTUBusWriteRegisterProcessArgs : STRUCT
  {attribute 'TcHmiSymbol.Show'}
  unitID : USINT;  (* Modbus station address (1..247) *)
  {attribute 'TcHmiSymbol.Show'}
  address : UINT;  (* Modbus data address *)
  {attribute 'TcHmiSymbol.Show'}
  value : INT;  (* Value to write on the register *)
END_STRUCT;
END_TYPE

TYPE ModbusRTUBusDiagnosticsProcessArgs : STRUCT
  {attribute 'TcHmiSymbol.Show'}
  unitID : USINT;  (* Modbus station address (1..247) *)
  {attribute 'TcHmiSymbol.Show'}
  subFunction : UINT;  (* Modbus subFunction code *)
  {attribute 'TcHmiSymbol.Show'}
  subData : INT;  (* Modbus data for subFunction *)
END_STRUCT;
END_TYPE

TYPE PointAlphaDeltaProcessArgs : STRUCT
  {attribute 'TcHmiSymbol.Show'}
  alpha : LREAL;  (* Right ascention, in hours *)
  {attribute 'TcHmiSymbol.Show'}
  delta : LREAL;  (* Declination, in degrees *)
END_STRUCT;
END_TYPE

TYPE GigECameraSetParamProcessArgs : STRUCT
  {attribute 'TcHmiSymbol.Show'}
  param : GigECameraParams;  (* UInt32 Parameter *)
  {attribute 'TcHmiSymbol.Show'}
  nValue : UDINT;  (* Integer Value *)
  {attribute 'TcHmiSymbol.Show'}
  fvalue : LREAL;  (* Double Value *)
  {attribute 'TcHmiSymbol.Show'}
  refresh : BOOL := TRUE;  (* Refresh the parameter set after the write (slower!) *)
END_STRUCT;
END_TYPE

TYPE GigECameraSetParam2ProcessArgs : STRUCT
  {attribute 'TcHmiSymbol.Show'}
  param1 : GigECameraParams;  (* UInt32 Parameter 1 *)
  {attribute 'TcHmiSymbol.Show'}
  nValue1 : UDINT;  (* Integer Value of Parameter 1 *)
  {attribute 'TcHmiSymbol.Show'}
  fvalue1 : LREAL;  (* Double Value of Parameter 1 *)
  {attribute 'TcHmiSymbol.Show'}
  param2 : GigECameraParams;  (* UInt32 Parameter 2 *)
  {attribute 'TcHmiSymbol.Show'}
  nValue2 : UDINT;  (* Integer Value of Parameter 2 *)
  {attribute 'TcHmiSymbol.Show'}
  fvalue2 : LREAL;  (* Double Value of Parameter 2 *)
  {attribute 'TcHmiSymbol.Show'}
  refresh : BOOL := TRUE;  (* Refresh the parameter set after the write (slower!) *)
END_STRUCT;
END_TYPE

TYPE GigECameraPulseTriggerArgs : STRUCT
  {attribute 'TcHmiSymbol.Show'}
  duration : LREAL;  (* Duration in seconds of the pulse *)
END_STRUCT;
END_TYPE

TYPE GigECameraSetSourceProcessArgs : STRUCT
  {attribute 'TcHmiSymbol.Show'}
  source : GigECameraSources;  (* Camera source to set *)
END_STRUCT;
END_TYPE

TYPE GigECameraSetupProcessArgs : STRUCT
  {attribute 'TcHmiSymbol.Show'}
  doExposureTime : BOOL := TRUE;  (* If TRUE, set the exposure time *)
  {attribute 'TcHmiSymbol.Show'}
  exposureTime : LREAL;  (* Exposure time in seconds *)
  {attribute 'TcHmiSymbol.Show'}
  doFrameRate : BOOL;  (* If TRUE, set the acquisition frame rate *)
  {attribute 'TcHmiSymbol.Show'}
  frameRate : LREAL;  (* Acquisition frame rate in Hz *)
  {attribute 'TcHmiSymbol.Show'}
  doWindowXY : BOOL;  (* If TRUE, set the window XY position *)
  {attribute 'TcHmiSymbol.Show'}
  windowX : UDINT;  (* Window X position in pixels *)
  {attribute 'TcHmiSymbol.Show'}
  windowY : UDINT;  (* Window Y position in pixels *)
  {attribute 'TcHmiSymbol.Show'}
  doWindowWH : BOOL;  (* If TRUE, set the window width and height *)
  {attribute 'TcHmiSymbol.Show'}
  windowWidth : UDINT;  (* Window width in pixels *)
  {attribute 'TcHmiSymbol.Show'}
  windowHeight : UDINT;  (* Window height in pixels *)
  {attribute 'TcHmiSymbol.Show'}
  doBinning : BOOL;  (* If TRUE, set the binning *)
  {attribute 'TcHmiSymbol.Show'}
  binningX : UDINT;  (* Binning X factor *)
  {attribute 'TcHmiSymbol.Show'}
  binningY : UDINT;  (* Binning Y factor *)
  {attribute 'TcHmiSymbol.Show'}
  doAnalogGain : BOOL;  (* If TRUE, set the analog gain *)
  {attribute 'TcHmiSymbol.Show'}
  analogGain : LREAL;  (* Analog gain *)
  {attribute 'TcHmiSymbol.Show'}
  doDigitalGain : BOOL;  (* If TRUE, set the digital gain *)
  {attribute 'TcHmiSymbol.Show'}
  digitalGain : LREAL;  (* Digital gain *)
  {attribute 'TcHmiSymbol.Show'}
  blackLevel : LREAL;  (* Black level (0 .. 511 for 12-bit images) *)
  {attribute 'TcHmiSymbol.Show'}
  blackLevelAuto : BOOL;  (* If TRUE, black level is set automatically. If FALSE, black level is set manually *)
  {attribute 'TcHmiSymbol.Show'}
  doBlackLevel : BOOL;  (* If TRUE, set the black level and black level auto *)
  {attribute 'TcHmiSymbol.Show'}
  continuous : BOOL;  (* If TRUE, set the continuous acquisition mode, trigger mode, etc. to continuous imaging *)
  {attribute 'TcHmiSymbol.Show'}
  doContinuous : BOOL;  (* If TRUE, set the continuous acquisition mode, trigger mode, etc. *)
END_STRUCT;
END_TYPE

TYPE GigECameraMultiTriggerProcessArgs : STRUCT
  {attribute 'TcHmiSymbol.Show'}
  count : UDINT;  (* Number of triggers to send *)
  {attribute 'TcHmiSymbol.Show'}
  algo : GigECameraMultiTriggerAlgorithms;  (* Algorithm to use for the multi-trigger *)
END_STRUCT;
END_TYPE

TYPE Arg1LrealProcessArgs : STRUCT
  {attribute 'TcHmiSymbol.Show'}
  setpoint : LREAL;  (* New setpoint value *)
END_STRUCT;
END_TYPE

TYPE Ell114SendProcessArgs : STRUCT
  {attribute 'TcHmiSymbol.Show'}
  cmd : ELL14Command;  (* The command to be sent *)
  {attribute 'TcHmiSymbol.Show'}
  arg : STRING(10);  (* The payload of the command to be sent (excluding '0gs' or similar header, excluding $R$N suffix). Custom commands must include the header! *)
END_STRUCT;
END_TYPE

TYPE M_SM_BaseProcess : STRUCT
  {attribute 'OPC.UA.DA' := '1'}
  {attribute 'OPC.UA.DA.Access' := '3'}
  {attribute 'TcHmiSymbol.Show'}
  do_request : BOOL;
  {attribute 'OPC.UA.DA' := '1'}
  {attribute 'OPC.UA.DA.Access' := '3'}
  {attribute 'TcHmiSymbol.Show'}
  atomic_in : ULINT;
  {attribute 'OPC.UA.DA' := '1'}
  {attribute 'OPC.UA.DA.Access' := '1'}
  {attribute 'TcHmiSymbol.Show'}
  do_request_result : RequestResults;
  {attribute 'OPC.UA.DA' := '1'}
  {attribute 'OPC.UA.DA.Access' := '1'}
  {attribute 'TcHmiSymbol.Show'}
  actualStatus : STRING;
  {attribute 'OPC.UA.DA' := '1'}
  {attribute 'OPC.UA.DA.Access' := '1'}
  {attribute 'TcHmiSymbol.Show'}
  atomic_out : ULINT;
  {attribute 'OPC.UA.DA' := '1'}
  {attribute 'OPC.UA.DA.Access' := '1'}
  {attribute 'TcHmiSymbol.Show'}
  lastRejectedHandle : UDINT;
  {attribute 'OPC.UA.DA' := '1'}
  {attribute 'TcHmiSymbol.Show'}
  stat : BaseProcessStatuses;
END_STRUCT;
END_TYPE

TYPE M_SM_BaseMcProcess : STRUCT
  {attribute 'OPC.UA.DA' := '1'}
  {attribute 'OPC.UA.DA.Access' := '1'}
  {attribute 'TcHmiSymbol.Show'}
  errorId : UDINT;
END_STRUCT;
END_TYPE

TYPE M_SM_ProcessStep : STRUCT
  {attribute 'OPC.UA.DA' := '1'}
  {attribute 'OPC.UA.DA.Access' := '1'}
  {attribute 'TcHmiSymbol.Show'}
  actualStatus : STRING;
  {attribute 'OPC.UA.DA' := '1'}
  {attribute 'TcHmiSymbol.Show'}
  stat : ProcessStepStatuses;
END_STRUCT;
END_TYPE

TYPE M_SM_BaseXmlDataSrvProcess : STRUCT
  {attribute 'OPC.UA.DA' := '1'}
  {attribute 'OPC.UA.DA.Access' := '1'}
  {attribute 'TcHmiSymbol.Show'}
  errorId : UDINT;
END_STRUCT;
END_TYPE

TYPE M_SM_BaseAxis : STRUCT
  {attribute 'OPC.UA.DA' := '1'}
  {attribute 'OPC.UA.DA.Access' := '1'}
  {attribute 'TcHmiSymbol.Show'}
  isGearingSupported : BOOL;
  {attribute 'OPC.UA.DA' := '1'}
  {attribute 'OPC.UA.DA.Access' := '1'}
  {attribute 'TcHmiSymbol.Show'}
  actualStatus : STRING;
  {attribute 'OPC.UA.DA' := '1'}
  {attribute 'OPC.UA.DA.Access' := '1'}
  {attribute 'TcHmiSymbol.Show'}
  isJogEnabled : BOOL;
  {attribute 'OPC.UA.DA' := '1'}
  {attribute 'OPC.UA.DA.Access' := '1'}
  {attribute 'TcHmiSymbol.Show'}
  errorId : UDINT;
  {attribute 'OPC.UA.DA' := '1'}
  {attribute 'OPC.UA.DA.Access' := '1'}
  {attribute 'TcHmiSymbol.Show'}
  posLimitSwitch : BOOL;
  {attribute 'OPC.UA.DA' := '1'}
  {attribute 'OPC.UA.DA.Access' := '1'}
  {attribute 'TcHmiSymbol.Show'}
  negLimitSwitch : BOOL;
  {attribute 'OPC.UA.DA' := '1'}
  {attribute 'TcHmiSymbol.Show'}
  stat : BaseAxisStatuses;
  {attribute 'OPC.UA.DA' := '1'}
  {attribute 'TcHmiSymbol.Show'}
  proc : M_SM_BaseAxisProcesses;
END_STRUCT;
END_TYPE

TYPE M_SM_AngularAxis : STRUCT
  {attribute 'OPC.UA.DA' := '1'}
  {attribute 'OPC.UA.DA.Access' := '1'}
  {attribute 'TcHmiSymbol.Show'}
  actPos : AngularPosition;
  {attribute 'OPC.UA.DA' := '1'}
  {attribute 'OPC.UA.DA.Access' := '1'}
  {attribute 'TcHmiSymbol.Show'}
  actVel : AngularVelocity;
  {attribute 'OPC.UA.DA' := '1'}
  {attribute 'OPC.UA.DA.Access' := '1'}
  {attribute 'TcHmiSymbol.Show'}
  setPos : AngularPosition;
  {attribute 'OPC.UA.DA' := '1'}
  {attribute 'OPC.UA.DA.Access' := '1'}
  {attribute 'TcHmiSymbol.Show'}
  setVel : AngularVelocity;
  {attribute 'OPC.UA.DA' := '1'}
  {attribute 'OPC.UA.DA.Access' := '1'}
  {attribute 'TcHmiSymbol.Show'}
  targetPos : AngularPosition;
END_STRUCT;
END_TYPE

TYPE M_SM_LinearAxis : STRUCT
  {attribute 'OPC.UA.DA' := '1'}
  {attribute 'OPC.UA.DA.Access' := '1'}
  {attribute 'TcHmiSymbol.Show'}
  actPos : LinearPosition;
  {attribute 'OPC.UA.DA' := '1'}
  {attribute 'OPC.UA.DA.Access' := '1'}
  {attribute 'TcHmiSymbol.Show'}
  actVel : LinearVelocity;
  {attribute 'OPC.UA.DA' := '1'}
  {attribute 'OPC.UA.DA.Access' := '1'}
  {attribute 'TcHmiSymbol.Show'}
  setPos : LinearPosition;
  {attribute 'OPC.UA.DA' := '1'}
  {attribute 'OPC.UA.DA.Access' := '1'}
  {attribute 'TcHmiSymbol.Show'}
  setVel : LinearVelocity;
  {attribute 'OPC.UA.DA' := '1'}
  {attribute 'OPC.UA.DA.Access' := '1'}
  {attribute 'TcHmiSymbol.Show'}
  targetPos : LinearPosition;
END_STRUCT;
END_TYPE

TYPE M_SM_MTS50Axis : STRUCT

END_STRUCT;
END_TYPE

TYPE M_SM_SSIEncoder : STRUCT
  {attribute 'OPC.UA.DA' := '1'}
  {attribute 'OPC.UA.DA.Access' := '1'}
  {attribute 'TcHmiSymbol.Show'}
  actualStatus : STRING;
  {attribute 'OPC.UA.DA' := '1'}
  {attribute 'OPC.UA.DA.Access' := '1'}
  {attribute 'TcHmiSymbol.Show'}
  dataError : BOOL;
  {attribute 'OPC.UA.DA' := '1'}
  {attribute 'OPC.UA.DA.Access' := '1'}
  {attribute 'TcHmiSymbol.Show'}
  frameError : BOOL;
  {attribute 'OPC.UA.DA' := '1'}
  {attribute 'OPC.UA.DA.Access' := '1'}
  {attribute 'TcHmiSymbol.Show'}
  powerFailure : BOOL;
  {attribute 'OPC.UA.DA' := '1'}
  {attribute 'OPC.UA.DA.Access' := '1'}
  {attribute 'TcHmiSymbol.Show'}
  syncError : BOOL;
  {attribute 'OPC.UA.DA' := '1'}
  {attribute 'TcHmiSymbol.Show'}
  stat : SSIEncoderStatuses;
END_STRUCT;
END_TYPE

TYPE M_SM_IncrementalEncoder : STRUCT
  {attribute 'OPC.UA.DA' := '1'}
  {attribute 'OPC.UA.DA.Access' := '1'}
  {attribute 'TcHmiSymbol.Show'}
  actualStatus : STRING;
  {attribute 'OPC.UA.DA' := '1'}
  {attribute 'OPC.UA.DA.Access' := '1'}
  {attribute 'TcHmiSymbol.Show'}
  latchCValid : BOOL;
  {attribute 'OPC.UA.DA' := '1'}
  {attribute 'OPC.UA.DA.Access' := '1'}
  {attribute 'TcHmiSymbol.Show'}
  latchExternValid : BOOL;
  {attribute 'OPC.UA.DA' := '1'}
  {attribute 'OPC.UA.DA.Access' := '1'}
  {attribute 'TcHmiSymbol.Show'}
  setCounterDone : BOOL;
  {attribute 'OPC.UA.DA' := '1'}
  {attribute 'OPC.UA.DA.Access' := '1'}
  {attribute 'TcHmiSymbol.Show'}
  counterUnderflow : BOOL;
  {attribute 'OPC.UA.DA' := '1'}
  {attribute 'OPC.UA.DA.Access' := '1'}
  {attribute 'TcHmiSymbol.Show'}
  counterOverflow : BOOL;
  {attribute 'OPC.UA.DA' := '1'}
  {attribute 'OPC.UA.DA.Access' := '1'}
  {attribute 'TcHmiSymbol.Show'}
  statusOfInputStatus : BOOL;
  {attribute 'OPC.UA.DA' := '1'}
  {attribute 'OPC.UA.DA.Access' := '1'}
  {attribute 'TcHmiSymbol.Show'}
  openCircuit : BOOL;
  {attribute 'OPC.UA.DA' := '1'}
  {attribute 'OPC.UA.DA.Access' := '1'}
  {attribute 'TcHmiSymbol.Show'}
  extrapolationStall : BOOL;
  {attribute 'OPC.UA.DA' := '1'}
  {attribute 'OPC.UA.DA.Access' := '1'}
  {attribute 'TcHmiSymbol.Show'}
  statusOfInputA : BOOL;
  {attribute 'OPC.UA.DA' := '1'}
  {attribute 'OPC.UA.DA.Access' := '1'}
  {attribute 'TcHmiSymbol.Show'}
  statusOfInputB : BOOL;
  {attribute 'OPC.UA.DA' := '1'}
  {attribute 'OPC.UA.DA.Access' := '1'}
  {attribute 'TcHmiSymbol.Show'}
  statusOfInputC : BOOL;
  {attribute 'OPC.UA.DA' := '1'}
  {attribute 'OPC.UA.DA.Access' := '1'}
  {attribute 'TcHmiSymbol.Show'}
  statusOfInputGate : BOOL;
  {attribute 'OPC.UA.DA' := '1'}
  {attribute 'OPC.UA.DA.Access' := '1'}
  {attribute 'TcHmiSymbol.Show'}
  statusOfExternLatch : BOOL;
  {attribute 'OPC.UA.DA' := '1'}
  {attribute 'OPC.UA.DA.Access' := '1'}
  {attribute 'TcHmiSymbol.Show'}
  syncError : BOOL;
  {attribute 'OPC.UA.DA' := '1'}
  {attribute 'TcHmiSymbol.Show'}
  stat : IncrementalEncoderStatuses;
  {attribute 'OPC.UA.DA' := '1'}
  {attribute 'TcHmiSymbol.Show'}
  proc : M_SM_IncrementalEncoderProcesses;
END_STRUCT;
END_TYPE

TYPE M_SM_EtherCatDevice : STRUCT
  {attribute 'OPC.UA.DA' := '1'}
  {attribute 'OPC.UA.DA.Access' := '1'}
  {attribute 'TcHmiSymbol.Show'}
  id : STRING;
  {attribute 'OPC.UA.DA' := '1'}
  {attribute 'OPC.UA.DA.Access' := '1'}
  {attribute 'TcHmiSymbol.Show'}
  typeId : STRING;
  {attribute 'OPC.UA.DA' := '1'}
  {attribute 'OPC.UA.DA.Access' := '1'}
  {attribute 'TcHmiSymbol.Show'}
  wcState : BOOL;
  {attribute 'OPC.UA.DA' := '1'}
  {attribute 'OPC.UA.DA.Access' := '1'}
  {attribute 'TcHmiSymbol.Show'}
  infoData : UINT;
  {attribute 'OPC.UA.DA' := '1'}
  {attribute 'OPC.UA.DA.Access' := '1'}
  {attribute 'TcHmiSymbol.Show'}
  actualStatus : STRING;
  {attribute 'OPC.UA.DA' := '1'}
  {attribute 'TcHmiSymbol.Show'}
  stat : EtherCatDeviceStatuses;
END_STRUCT;
END_TYPE

TYPE M_SM_CANopenBus : STRUCT
  {attribute 'OPC.UA.DA' := '1'}
  {attribute 'OPC.UA.DA.Access' := '1'}
  {attribute 'TcHmiSymbol.Show'}
  error : USINT;
  {attribute 'OPC.UA.DA' := '1'}
  {attribute 'OPC.UA.DA.Access' := '1'}
  {attribute 'TcHmiSymbol.Show'}
  canState : UINT;
  {attribute 'OPC.UA.DA' := '1'}
  {attribute 'OPC.UA.DA.Access' := '1'}
  {attribute 'TcHmiSymbol.Show'}
  rxErrorCounter : USINT;
  {attribute 'OPC.UA.DA' := '1'}
  {attribute 'OPC.UA.DA.Access' := '1'}
  {attribute 'TcHmiSymbol.Show'}
  txErrorCounter : USINT;
  {attribute 'OPC.UA.DA' := '1'}
  {attribute 'OPC.UA.DA.Access' := '1'}
  {attribute 'TcHmiSymbol.Show'}
  actualStatus : STRING;
  {attribute 'OPC.UA.DA' := '1'}
  {attribute 'TcHmiSymbol.Show'}
  stat : CANopenBusStatuses;
END_STRUCT;
END_TYPE

TYPE M_SM_CurrentMeasurement : STRUCT
  {attribute 'OPC.UA.DA' := '1'}
  {attribute 'OPC.UA.DA.Access' := '1'}
  {attribute 'TcHmiSymbol.Show'}
  actualStatus : STRING;
  {attribute 'OPC.UA.DA' := '1'}
  {attribute 'OPC.UA.DA.Access' := '1'}
  {attribute 'TcHmiSymbol.Show'}
  current : Current;
  {attribute 'OPC.UA.DA' := '1'}
  {attribute 'TcHmiSymbol.Show'}
  stat : CurrentMeasurementStatuses;
END_STRUCT;
END_TYPE

TYPE M_SM_VoltageMeasurement : STRUCT
  {attribute 'OPC.UA.DA' := '1'}
  {attribute 'OPC.UA.DA.Access' := '1'}
  {attribute 'TcHmiSymbol.Show'}
  actualStatus : STRING;
  {attribute 'OPC.UA.DA' := '1'}
  {attribute 'OPC.UA.DA.Access' := '1'}
  {attribute 'TcHmiSymbol.Show'}
  actual : Voltage;
  {attribute 'OPC.UA.DA' := '1'}
  {attribute 'OPC.UA.DA.Access' := '1'}
  {attribute 'TcHmiSymbol.Show'}
  average : Voltage;
  {attribute 'OPC.UA.DA' := '1'}
  {attribute 'OPC.UA.DA.Access' := '1'}
  {attribute 'TcHmiSymbol.Show'}
  underrange : BOOL;
  {attribute 'OPC.UA.DA' := '1'}
  {attribute 'OPC.UA.DA.Access' := '1'}
  {attribute 'TcHmiSymbol.Show'}
  overrange : BOOL;
  {attribute 'OPC.UA.DA' := '1'}
  {attribute 'TcHmiSymbol.Show'}
  stat : VoltageMeasurementStatuses;
END_STRUCT;
END_TYPE

TYPE M_SM_SimpleTemperature : STRUCT
  {attribute 'OPC.UA.DA' := '1'}
  {attribute 'OPC.UA.DA.Access' := '1'}
  {attribute 'TcHmiSymbol.Show'}
  actualStatus : STRING;
  {attribute 'OPC.UA.DA' := '1'}
  {attribute 'OPC.UA.DA.Access' := '1'}
  {attribute 'TcHmiSymbol.Show'}
  value : LREAL;
  {attribute 'OPC.UA.DA' := '1'}
  {attribute 'OPC.UA.DA.Access' := '1'}
  {attribute 'TcHmiSymbol.Show'}
  error : BOOL;
  {attribute 'OPC.UA.DA' := '1'}
  {attribute 'OPC.UA.DA.Access' := '1'}
  {attribute 'TcHmiSymbol.Show'}
  underrange : BOOL;
  {attribute 'OPC.UA.DA' := '1'}
  {attribute 'OPC.UA.DA.Access' := '1'}
  {attribute 'TcHmiSymbol.Show'}
  overrange : BOOL;
  {attribute 'OPC.UA.DA' := '1'}
  {attribute 'TcHmiSymbol.Show'}
  stat : SimpleTemperatureStatuses;
END_STRUCT;
END_TYPE

TYPE M_SM_TemperatureMeasurement : STRUCT
  {attribute 'OPC.UA.DA' := '1'}
  {attribute 'OPC.UA.DA.Access' := '1'}
  {attribute 'TcHmiSymbol.Show'}
  actualStatus : STRING;
  {attribute 'OPC.UA.DA' := '1'}
  {attribute 'OPC.UA.DA.Access' := '1'}
  {attribute 'TcHmiSymbol.Show'}
  actual : Temperature;
  {attribute 'OPC.UA.DA' := '1'}
  {attribute 'OPC.UA.DA.Access' := '1'}
  {attribute 'TcHmiSymbol.Show'}
  average : Temperature;
  {attribute 'OPC.UA.DA' := '1'}
  {attribute 'OPC.UA.DA.Access' := '1'}
  {attribute 'TcHmiSymbol.Show'}
  underrange : BOOL;
  {attribute 'OPC.UA.DA' := '1'}
  {attribute 'OPC.UA.DA.Access' := '1'}
  {attribute 'TcHmiSymbol.Show'}
  overrange : BOOL;
  {attribute 'OPC.UA.DA' := '1'}
  {attribute 'TcHmiSymbol.Show'}
  stat : TemperatureMeasurementStatuses;
END_STRUCT;
END_TYPE

TYPE M_SM_PressureMeasurement : STRUCT
  {attribute 'OPC.UA.DA' := '1'}
  {attribute 'OPC.UA.DA.Access' := '1'}
  {attribute 'TcHmiSymbol.Show'}
  actualStatus : STRING;
  {attribute 'OPC.UA.DA' := '1'}
  {attribute 'OPC.UA.DA.Access' := '1'}
  {attribute 'TcHmiSymbol.Show'}
  actual : Pressure;
  {attribute 'OPC.UA.DA' := '1'}
  {attribute 'OPC.UA.DA.Access' := '1'}
  {attribute 'TcHmiSymbol.Show'}
  average : Pressure;
  {attribute 'OPC.UA.DA' := '1'}
  {attribute 'OPC.UA.DA.Access' := '1'}
  {attribute 'TcHmiSymbol.Show'}
  underrange : BOOL;
  {attribute 'OPC.UA.DA' := '1'}
  {attribute 'OPC.UA.DA.Access' := '1'}
  {attribute 'TcHmiSymbol.Show'}
  overrange : BOOL;
  {attribute 'OPC.UA.DA' := '1'}
  {attribute 'TcHmiSymbol.Show'}
  stat : PressureMeasurementStatuses;
END_STRUCT;
END_TYPE

TYPE M_SM_FrequencyMeasurement : STRUCT
  {attribute 'OPC.UA.DA' := '1'}
  {attribute 'OPC.UA.DA.Access' := '1'}
  {attribute 'TcHmiSymbol.Show'}
  actualStatus : STRING;
  {attribute 'OPC.UA.DA' := '1'}
  {attribute 'OPC.UA.DA.Access' := '1'}
  {attribute 'TcHmiSymbol.Show'}
  actual : Frequency;
  {attribute 'OPC.UA.DA' := '1'}
  {attribute 'OPC.UA.DA.Access' := '1'}
  {attribute 'TcHmiSymbol.Show'}
  average : Frequency;
  {attribute 'OPC.UA.DA' := '1'}
  {attribute 'OPC.UA.DA.Access' := '1'}
  {attribute 'TcHmiSymbol.Show'}
  underrange : BOOL;
  {attribute 'OPC.UA.DA' := '1'}
  {attribute 'OPC.UA.DA.Access' := '1'}
  {attribute 'TcHmiSymbol.Show'}
  overrange : BOOL;
  {attribute 'OPC.UA.DA' := '1'}
  {attribute 'TcHmiSymbol.Show'}
  stat : FrequencyMeasurementStatuses;
END_STRUCT;
END_TYPE

TYPE M_SM_GForceMeasurement : STRUCT
  {attribute 'OPC.UA.DA' := '1'}
  {attribute 'OPC.UA.DA.Access' := '1'}
  {attribute 'TcHmiSymbol.Show'}
  actualStatus : STRING;
  {attribute 'OPC.UA.DA' := '1'}
  {attribute 'OPC.UA.DA.Access' := '1'}
  {attribute 'TcHmiSymbol.Show'}
  actual : GForce;
  {attribute 'OPC.UA.DA' := '1'}
  {attribute 'OPC.UA.DA.Access' := '1'}
  {attribute 'TcHmiSymbol.Show'}
  average : GForce;
  {attribute 'OPC.UA.DA' := '1'}
  {attribute 'TcHmiSymbol.Show'}
  stat : GForceMeasurementStatuses;
END_STRUCT;
END_TYPE

TYPE M_SM_RelativeHumidityMeasurement : STRUCT
  {attribute 'OPC.UA.DA' := '1'}
  {attribute 'OPC.UA.DA.Access' := '1'}
  {attribute 'TcHmiSymbol.Show'}
  actualStatus : STRING;
  {attribute 'OPC.UA.DA' := '1'}
  {attribute 'OPC.UA.DA.Access' := '1'}
  {attribute 'TcHmiSymbol.Show'}
  actual : Fraction;
  {attribute 'OPC.UA.DA' := '1'}
  {attribute 'OPC.UA.DA.Access' := '1'}
  {attribute 'TcHmiSymbol.Show'}
  average : Fraction;
  {attribute 'OPC.UA.DA' := '1'}
  {attribute 'OPC.UA.DA.Access' := '1'}
  {attribute 'TcHmiSymbol.Show'}
  underrange : BOOL;
  {attribute 'OPC.UA.DA' := '1'}
  {attribute 'OPC.UA.DA.Access' := '1'}
  {attribute 'TcHmiSymbol.Show'}
  overrange : BOOL;
  {attribute 'OPC.UA.DA' := '1'}
  {attribute 'TcHmiSymbol.Show'}
  stat : RelativeHumidityMeasurementStatuses;
END_STRUCT;
END_TYPE

TYPE M_SM_ForceMeasurement : STRUCT
  {attribute 'OPC.UA.DA' := '1'}
  {attribute 'OPC.UA.DA.Access' := '1'}
  {attribute 'TcHmiSymbol.Show'}
  actualStatus : STRING;
  {attribute 'OPC.UA.DA' := '1'}
  {attribute 'OPC.UA.DA.Access' := '1'}
  {attribute 'TcHmiSymbol.Show'}
  actual : Force;
  {attribute 'OPC.UA.DA' := '1'}
  {attribute 'OPC.UA.DA.Access' := '1'}
  {attribute 'TcHmiSymbol.Show'}
  average : Force;
  {attribute 'OPC.UA.DA' := '1'}
  {attribute 'TcHmiSymbol.Show'}
  stat : ForceMeasurementStatuses;
END_STRUCT;
END_TYPE

TYPE M_SM_LinearPositionMeasurement16 : STRUCT
  {attribute 'OPC.UA.DA' := '1'}
  {attribute 'OPC.UA.DA.Access' := '1'}
  {attribute 'TcHmiSymbol.Show'}
  actualStatus : STRING;
  {attribute 'OPC.UA.DA' := '1'}
  {attribute 'OPC.UA.DA.Access' := '1'}
  {attribute 'TcHmiSymbol.Show'}
  actual : LinearPosition;
  {attribute 'OPC.UA.DA' := '1'}
  {attribute 'OPC.UA.DA.Access' := '1'}
  {attribute 'TcHmiSymbol.Show'}
  average : LinearPosition;
  {attribute 'OPC.UA.DA' := '1'}
  {attribute 'TcHmiSymbol.Show'}
  stat : LinearPositionMeasurement16Statuses;
END_STRUCT;
END_TYPE

TYPE M_SM_LinearPositionMeasurementU32 : STRUCT
  {attribute 'OPC.UA.DA' := '1'}
  {attribute 'OPC.UA.DA.Access' := '1'}
  {attribute 'TcHmiSymbol.Show'}
  actualStatus : STRING;
  {attribute 'OPC.UA.DA' := '1'}
  {attribute 'OPC.UA.DA.Access' := '1'}
  {attribute 'TcHmiSymbol.Show'}
  actual : LinearPosition;
  {attribute 'OPC.UA.DA' := '1'}
  {attribute 'OPC.UA.DA.Access' := '1'}
  {attribute 'TcHmiSymbol.Show'}
  average : LinearPosition;
  {attribute 'OPC.UA.DA' := '1'}
  {attribute 'TcHmiSymbol.Show'}
  stat : LinearPositionMeasurementU32Statuses;
END_STRUCT;
END_TYPE

TYPE M_SM_SimpleRelay : STRUCT
  {attribute 'OPC.UA.DA' := '1'}
  {attribute 'OPC.UA.DA.Access' := '1'}
  {attribute 'TcHmiSymbol.Show'}
  actualStatus : STRING;
  {attribute 'OPC.UA.DA' := '1'}
  {attribute 'OPC.UA.DA.Access' := '1'}
  {attribute 'TcHmiSymbol.Show'}
  digitalOutput : BOOL;
  {attribute 'OPC.UA.DA' := '1'}
  {attribute 'TcHmiSymbol.Show'}
  stat : SimpleRelayStatuses;
  {attribute 'OPC.UA.DA' := '1'}
  {attribute 'TcHmiSymbol.Show'}
  proc : M_SM_SimpleRelayProcesses;
END_STRUCT;
END_TYPE

TYPE M_SM_Fuse : STRUCT
  {attribute 'OPC.UA.DA' := '1'}
  {attribute 'OPC.UA.DA.Access' := '1'}
  {attribute 'TcHmiSymbol.Show'}
  enabled : BOOL;
  {attribute 'OPC.UA.DA' := '1'}
  {attribute 'OPC.UA.DA.Access' := '1'}
  {attribute 'TcHmiSymbol.Show'}
  tripped : BOOL;
  {attribute 'OPC.UA.DA' := '1'}
  {attribute 'OPC.UA.DA.Access' := '1'}
  {attribute 'TcHmiSymbol.Show'}
  overload : BOOL;
  {attribute 'OPC.UA.DA' := '1'}
  {attribute 'OPC.UA.DA.Access' := '1'}
  {attribute 'TcHmiSymbol.Show'}
  actualStatus : STRING;
  {attribute 'OPC.UA.DA' := '1'}
  {attribute 'OPC.UA.DA.Access' := '1'}
  {attribute 'TcHmiSymbol.Show'}
  resetOutput : BOOL;
  {attribute 'OPC.UA.DA' := '1'}
  {attribute 'OPC.UA.DA.Access' := '1'}
  {attribute 'TcHmiSymbol.Show'}
  switchOutput : BOOL;
  {attribute 'OPC.UA.DA' := '1'}
  {attribute 'TcHmiSymbol.Show'}
  stat : FuseStatuses;
  {attribute 'OPC.UA.DA' := '1'}
  {attribute 'TcHmiSymbol.Show'}
  proc : M_SM_FuseProcesses;
END_STRUCT;
END_TYPE

TYPE M_SM_Led : STRUCT
  {attribute 'OPC.UA.DA' := '1'}
  {attribute 'OPC.UA.DA.Access' := '1'}
  {attribute 'TcHmiSymbol.Show'}
  actualStatus : STRING;
  {attribute 'OPC.UA.DA' := '1'}
  {attribute 'OPC.UA.DA.Access' := '1'}
  {attribute 'TcHmiSymbol.Show'}
  milliAmps : LREAL;
  {attribute 'OPC.UA.DA' := '1'}
  {attribute 'OPC.UA.DA.Access' := '1'}
  {attribute 'TcHmiSymbol.Show'}
  relayOn : BOOL;
  {attribute 'OPC.UA.DA' := '1'}
  {attribute 'TcHmiSymbol.Show'}
  stat : LedStatuses;
  {attribute 'OPC.UA.DA' := '1'}
  {attribute 'TcHmiSymbol.Show'}
  proc : M_SM_LedProcesses;
END_STRUCT;
END_TYPE

TYPE M_SM_TipTilt : STRUCT
  {attribute 'OPC.UA.DA' := '1'}
  {attribute 'OPC.UA.DA.Access' := '1'}
  {attribute 'TcHmiSymbol.Show'}
  actualStatus : STRING;
  {attribute 'OPC.UA.DA' := '1'}
  {attribute 'OPC.UA.DA.Access' := '1'}
  {attribute 'TcHmiSymbol.Show'}
  v1 : LREAL;
  {attribute 'OPC.UA.DA' := '1'}
  {attribute 'OPC.UA.DA.Access' := '1'}
  {attribute 'TcHmiSymbol.Show'}
  v2 : LREAL;
  {attribute 'OPC.UA.DA' := '1'}
  {attribute 'OPC.UA.DA.Access' := '1'}
  {attribute 'TcHmiSymbol.Show'}
  v3 : LREAL;
  {attribute 'OPC.UA.DA' := '1'}
  {attribute 'TcHmiSymbol.Show'}
  stat : TipTiltStatuses;
  {attribute 'OPC.UA.DA' := '1'}
  {attribute 'TcHmiSymbol.Show'}
  proc : M_SM_TipTiltProcesses;
END_STRUCT;
END_TYPE

TYPE M_SM_ConfigManager : STRUCT
  {attribute 'OPC.UA.DA' := '1'}
  {attribute 'OPC.UA.DA.Access' := '1'}
  {attribute 'TcHmiSymbol.Show'}
  filePath : STRING;
  {attribute 'OPC.UA.DA' := '1'}
  {attribute 'OPC.UA.DA.Access' := '1'}
  {attribute 'TcHmiSymbol.Show'}
  actualStatus : STRING;
  {attribute 'OPC.UA.DA' := '1'}
  {attribute 'TcHmiSymbol.Show'}
  stat : ConfigManagerStatuses;
  {attribute 'OPC.UA.DA' := '1'}
  {attribute 'TcHmiSymbol.Show'}
  proc : M_SM_ConfigManagerProcesses;
END_STRUCT;
END_TYPE

TYPE M_SM_ModbusRTUBus : STRUCT
  {attribute 'OPC.UA.DA' := '1'}
  {attribute 'OPC.UA.DA.Access' := '1'}
  {attribute 'TcHmiSymbol.Show'}
  retries : INT;
  {attribute 'OPC.UA.DA' := '1'}
  {attribute 'OPC.UA.DA.Access' := '1'}
  {attribute 'TcHmiSymbol.Show'}
  actualStatus : STRING;
  {attribute 'OPC.UA.DA' := '1'}
  {attribute 'TcHmiSymbol.Show'}
  stat : ModbusRTUBusStatuses;
  {attribute 'OPC.UA.DA' := '1'}
  {attribute 'TcHmiSymbol.Show'}
  proc : M_SM_ModbusRTUBusProcesses;
END_STRUCT;
END_TYPE

TYPE M_SM_GigECamera : STRUCT
  {attribute 'OPC.UA.DA' := '1'}
  {attribute 'OPC.UA.DA.Access' := '1'}
  {attribute 'TcHmiSymbol.Show'}
  state : ETcVnCameraState;
  {attribute 'OPC.UA.DA' := '1'}
  {attribute 'OPC.UA.DA.Access' := '1'}
  {attribute 'TcHmiSymbol.Show'}
  source : GigECameraSources;
  {attribute 'OPC.UA.DA' := '1'}
  {attribute 'OPC.UA.DA.Access' := '1'}
  {attribute 'TcHmiSymbol.Show'}
  actualStatus : STRING;
  {attribute 'OPC.UA.DA' := '1'}
  {attribute 'OPC.UA.DA.Access' := '1'}
  {attribute 'TcHmiSymbol.Show'}
  frameCounter : UDINT;
  {attribute 'OPC.UA.DA' := '1'}
  {attribute 'OPC.UA.DA.Access' := '1'}
  {attribute 'TcHmiSymbol.Show'}
  loopCounter : UDINT;
  {attribute 'OPC.UA.DA' := '1'}
  {attribute 'OPC.UA.DA.Access' := '1'}
  {attribute 'TcHmiSymbol.Show'}
  loopSuccessCounter : UDINT;
  {attribute 'OPC.UA.DA' := '1'}
  {attribute 'OPC.UA.DA.Access' := '1'}
  {attribute 'TcHmiSymbol.Show'}
  channelOpen : BOOL;
  {attribute 'OPC.UA.DA' := '1'}
  {attribute 'OPC.UA.DA.Access' := '1'}
  {attribute 'TcHmiSymbol.Show'}
  acquiring : BOOL;
  {attribute 'OPC.UA.DA' := '1'}
  {attribute 'OPC.UA.DA.Access' := '1'}
  {attribute 'TcHmiSymbol.Show'}
  actualMultiTriggerNumber : UDINT;
  {attribute 'OPC.UA.DA' := '1'}
  {attribute 'OPC.UA.DA.Access' := '1'}
  {attribute 'TcHmiSymbol.Show'}
  maxMultiTriggerNumber : UDINT;
  {attribute 'OPC.UA.DA' := '1'}
  {attribute 'OPC.UA.DA.Access' := '1'}
  {attribute 'TcHmiSymbol.Show'}
  acquisitionFrameRate : LREAL;
  {attribute 'OPC.UA.DA' := '1'}
  {attribute 'OPC.UA.DA.Access' := '1'}
  {attribute 'TcHmiSymbol.Show'}
  linkAcquisitionFrameRate : LREAL;
  {attribute 'OPC.UA.DA' := '1'}
  {attribute 'OPC.UA.DA.Access' := '1'}
  {attribute 'TcHmiSymbol.Show'}
  exposureTime : LREAL;
  {attribute 'OPC.UA.DA' := '1'}
  {attribute 'OPC.UA.DA.Access' := '1'}
  {attribute 'TcHmiSymbol.Show'}
  gainSelector : UDINT;
  {attribute 'OPC.UA.DA' := '1'}
  {attribute 'OPC.UA.DA.Access' := '1'}
  {attribute 'TcHmiSymbol.Show'}
  gain : LREAL;
  {attribute 'OPC.UA.DA' := '1'}
  {attribute 'OPC.UA.DA.Access' := '1'}
  {attribute 'TcHmiSymbol.Show'}
  gainAnalog : LREAL;
  {attribute 'OPC.UA.DA' := '1'}
  {attribute 'OPC.UA.DA.Access' := '1'}
  {attribute 'TcHmiSymbol.Show'}
  gainDigital : LREAL;
  {attribute 'OPC.UA.DA' := '1'}
  {attribute 'OPC.UA.DA.Access' := '1'}
  {attribute 'TcHmiSymbol.Show'}
  width : UDINT;
  {attribute 'OPC.UA.DA' := '1'}
  {attribute 'OPC.UA.DA.Access' := '1'}
  {attribute 'TcHmiSymbol.Show'}
  height : UDINT;
  {attribute 'OPC.UA.DA' := '1'}
  {attribute 'OPC.UA.DA.Access' := '1'}
  {attribute 'TcHmiSymbol.Show'}
  offsetX : UDINT;
  {attribute 'OPC.UA.DA' := '1'}
  {attribute 'OPC.UA.DA.Access' := '1'}
  {attribute 'TcHmiSymbol.Show'}
  offsetY : UDINT;
  {attribute 'OPC.UA.DA' := '1'}
  {attribute 'OPC.UA.DA.Access' := '1'}
  {attribute 'TcHmiSymbol.Show'}
  widthMax : UDINT;
  {attribute 'OPC.UA.DA' := '1'}
  {attribute 'OPC.UA.DA.Access' := '1'}
  {attribute 'TcHmiSymbol.Show'}
  heightMax : UDINT;
  {attribute 'OPC.UA.DA' := '1'}
  {attribute 'OPC.UA.DA.Access' := '1'}
  {attribute 'TcHmiSymbol.Show'}
  binningSelector : UDINT;
  {attribute 'OPC.UA.DA' := '1'}
  {attribute 'OPC.UA.DA.Access' := '1'}
  {attribute 'TcHmiSymbol.Show'}
  binningHorizontal : UDINT;
  {attribute 'OPC.UA.DA' := '1'}
  {attribute 'OPC.UA.DA.Access' := '1'}
  {attribute 'TcHmiSymbol.Show'}
  binningVertical : UDINT;
  {attribute 'OPC.UA.DA' := '1'}
  {attribute 'OPC.UA.DA.Access' := '1'}
  {attribute 'TcHmiSymbol.Show'}
  triggerMode : UDINT;
  {attribute 'OPC.UA.DA' := '1'}
  {attribute 'OPC.UA.DA.Access' := '1'}
  {attribute 'TcHmiSymbol.Show'}
  triggerSelector : UDINT;
  {attribute 'OPC.UA.DA' := '1'}
  {attribute 'OPC.UA.DA.Access' := '1'}
  {attribute 'TcHmiSymbol.Show'}
  acquisitionMode : UDINT;
  {attribute 'OPC.UA.DA' := '1'}
  {attribute 'OPC.UA.DA.Access' := '1'}
  {attribute 'TcHmiSymbol.Show'}
  blackLevel : LREAL;
  {attribute 'OPC.UA.DA' := '1'}
  {attribute 'OPC.UA.DA.Access' := '1'}
  {attribute 'TcHmiSymbol.Show'}
  blackLevelAuto : UDINT;
  {attribute 'OPC.UA.DA' := '1'}
  {attribute 'OPC.UA.DA.Access' := '1'}
  {attribute 'TcHmiSymbol.Show'}
  deviceTemperature : LREAL;
  {attribute 'OPC.UA.DA' := '1'}
  {attribute 'TcHmiSymbol.Show'}
  stat : GigECameraStatuses;
  {attribute 'OPC.UA.DA' := '1'}
  {attribute 'TcHmiSymbol.Show'}
  proc : M_SM_GigECameraProcesses;
END_STRUCT;
END_TYPE

TYPE M_SM_ELL14Stage : STRUCT
  {attribute 'OPC.UA.DA' := '1'}
  {attribute 'OPC.UA.DA.Access' := '1'}
  {attribute 'TcHmiSymbol.Show'}
  simulated : BOOL;
  {attribute 'OPC.UA.DA' := '1'}
  {attribute 'OPC.UA.DA.Access' := '1'}
  {attribute 'TcHmiSymbol.Show'}
  actualStatus : STRING;
  {attribute 'OPC.UA.DA' := '1'}
  {attribute 'OPC.UA.DA.Access' := '1'}
  {attribute 'TcHmiSymbol.Show'}
  commError : BOOL;
  {attribute 'OPC.UA.DA' := '1'}
  {attribute 'OPC.UA.DA.Access' := '1'}
  {attribute 'TcHmiSymbol.Show'}
  homed : BOOL;
  {attribute 'OPC.UA.DA' := '1'}
  {attribute 'OPC.UA.DA.Access' := '1'}
  {attribute 'TcHmiSymbol.Show'}
  position : LREAL;
  {attribute 'OPC.UA.DA' := '1'}
  {attribute 'OPC.UA.DA.Access' := '1'}
  {attribute 'TcHmiSymbol.Show'}
  statusCode : ELL14StatusCode;
  {attribute 'OPC.UA.DA' := '1'}
  {attribute 'TcHmiSymbol.Show'}
  stat : ELL14StageStatuses;
  {attribute 'OPC.UA.DA' := '1'}
  {attribute 'TcHmiSymbol.Show'}
  proc : M_SM_ELL14StageProcesses;
END_STRUCT;
END_TYPE

TYPE M_SM_Sequencer : STRUCT
  {attribute 'OPC.UA.DA' := '1'}
  {attribute 'OPC.UA.DA.Access' := '3'}
  {attribute 'TcHmiSymbol.Show'}
  editableSeq : SequenceEnumConfig_M;
  {attribute 'OPC.UA.DA' := '1'}
  {attribute 'OPC.UA.DA.Access' := '1'}
  {attribute 'TcHmiSymbol.Show'}
  actualStatus : STRING;
  {attribute 'OPC.UA.DA' := '1'}
  {attribute 'OPC.UA.DA.Access' := '1'}
  {attribute 'TcHmiSymbol.Show'}
  runnableSeq : SequenceEnumConfig_M;
  {attribute 'OPC.UA.DA' := '1'}
  {attribute 'OPC.UA.DA.Access' := '1'}
  {attribute 'TcHmiSymbol.Show'}
  runnableStat : ARRAY[0..29] OF ActionStatus;
  {attribute 'OPC.UA.DA' := '1'}
  {attribute 'OPC.UA.DA.Access' := '1'}
  {attribute 'TcHmiSymbol.Show'}
  runnableIndex : UINT;
  {attribute 'OPC.UA.DA' := '1'}
  {attribute 'OPC.UA.DA.Access' := '1'}
  {attribute 'TcHmiSymbol.Show'}
  editableIndex : UINT;
  {attribute 'OPC.UA.DA' := '1'}
  {attribute 'OPC.UA.DA.Access' := '1'}
  {attribute 'TcHmiSymbol.Show'}
  ids : ARRAY[0..50] OF STRING(30);
  {attribute 'OPC.UA.DA' := '1'}
  {attribute 'TcHmiSymbol.Show'}
  stat : SequencerStatuses;
  {attribute 'OPC.UA.DA' := '1'}
  {attribute 'TcHmiSymbol.Show'}
  parts : M_SM_SequencerParts;
  {attribute 'OPC.UA.DA' := '1'}
  {attribute 'TcHmiSymbol.Show'}
  proc : M_SM_SequencerProcesses;
END_STRUCT;
END_TYPE

TYPE M_SM_EventManager : STRUCT
  {attribute 'OPC.UA.DA' := '1'}
  {attribute 'OPC.UA.DA.Access' := '1'}
  {attribute 'TcHmiSymbol.Show'}
  actualStatus : STRING;
  {attribute 'OPC.UA.DA' := '1'}
  {attribute 'OPC.UA.DA.Access' := '1'}
  {attribute 'TcHmiSymbol.Show'}
  alarmCount : INT;
  {attribute 'OPC.UA.DA' := '1'}
  {attribute 'TcHmiSymbol.Show'}
  stat : EventManagerStatuses;
END_STRUCT;
END_TYPE

TYPE M_Process : STRUCT

END_STRUCT;
END_TYPE

TYPE M_IdProcess : STRUCT
  {attribute 'OPC.UA.DA' := '1'}
  {attribute 'OPC.UA.DA.Access' := '3'}
  {attribute 'TcHmiSymbol.Show'}
  set : IdProcessArgs;
END_STRUCT;
END_TYPE

TYPE M_IndexProcess : STRUCT
  {attribute 'OPC.UA.DA' := '1'}
  {attribute 'OPC.UA.DA.Access' := '3'}
  {attribute 'TcHmiSymbol.Show'}
  set : IndexProcessArgs;
END_STRUCT;
END_TYPE

TYPE M_McProcess : STRUCT

END_STRUCT;
END_TYPE

TYPE M_ChangeSetpointProcess : STRUCT
  {attribute 'OPC.UA.DA' := '1'}
  {attribute 'OPC.UA.DA.Access' := '3'}
  {attribute 'TcHmiSymbol.Show'}
  set : ChangeSetpointProcessArgs;
END_STRUCT;
END_TYPE

TYPE M_ChangeParameterProcess : STRUCT
  {attribute 'OPC.UA.DA' := '1'}
  {attribute 'OPC.UA.DA.Access' := '3'}
  {attribute 'TcHmiSymbol.Show'}
  set : ChangeParameterProcessArgs;
END_STRUCT;
END_TYPE

TYPE M_McMoveAbsoluteProcess : STRUCT
  {attribute 'OPC.UA.DA' := '1'}
  {attribute 'OPC.UA.DA.Access' := '3'}
  {attribute 'TcHmiSymbol.Show'}
  set : McMoveAbsoluteProcessArgs;
END_STRUCT;
END_TYPE

TYPE M_McMoveRelativeProcess : STRUCT
  {attribute 'OPC.UA.DA' := '1'}
  {attribute 'OPC.UA.DA.Access' := '3'}
  {attribute 'TcHmiSymbol.Show'}
  set : McMoveRelativeProcessArgs;
END_STRUCT;
END_TYPE

TYPE M_McPowerProcess : STRUCT
  {attribute 'OPC.UA.DA' := '1'}
  {attribute 'OPC.UA.DA.Access' := '3'}
  {attribute 'TcHmiSymbol.Show'}
  set : McPowerProcessArgs;
END_STRUCT;
END_TYPE

TYPE M_McSetPositionProcess : STRUCT
  {attribute 'OPC.UA.DA' := '1'}
  {attribute 'OPC.UA.DA.Access' := '3'}
  {attribute 'TcHmiSymbol.Show'}
  set : McSetPositionProcessArgs;
END_STRUCT;
END_TYPE

TYPE M_McStopProcess : STRUCT
  {attribute 'OPC.UA.DA' := '1'}
  {attribute 'OPC.UA.DA.Access' := '3'}
  {attribute 'TcHmiSymbol.Show'}
  set : McStopProcessArgs;
END_STRUCT;
END_TYPE

TYPE M_McMoveVelocityProcess : STRUCT
  {attribute 'OPC.UA.DA' := '1'}
  {attribute 'OPC.UA.DA.Access' := '3'}
  {attribute 'TcHmiSymbol.Show'}
  set : McMoveVelocityProcessArgs;
END_STRUCT;
END_TYPE

TYPE M_SetEnabledProcess : STRUCT
  {attribute 'OPC.UA.DA' := '1'}
  {attribute 'OPC.UA.DA.Access' := '3'}
  {attribute 'TcHmiSymbol.Show'}
  set : SetEnabledProcessArgs;
END_STRUCT;
END_TYPE

TYPE M_McWriteParameter : STRUCT
  {attribute 'OPC.UA.DA' := '1'}
  {attribute 'OPC.UA.DA.Access' := '3'}
  {attribute 'TcHmiSymbol.Show'}
  set : McWriteParameterArgs;
END_STRUCT;
END_TYPE

TYPE M_McReadParameter : STRUCT
  {attribute 'OPC.UA.DA' := '1'}
  {attribute 'OPC.UA.DA.Access' := '1'}
  {attribute 'TcHmiSymbol.Show'}
  value : LREAL;
  {attribute 'OPC.UA.DA' := '1'}
  {attribute 'OPC.UA.DA.Access' := '3'}
  {attribute 'TcHmiSymbol.Show'}
  set : McReadParameterArgs;
END_STRUCT;
END_TYPE

TYPE M_McWriteBoolParameter : STRUCT
  {attribute 'OPC.UA.DA' := '1'}
  {attribute 'OPC.UA.DA.Access' := '3'}
  {attribute 'TcHmiSymbol.Show'}
  set : McWriteBoolParameterArgs;
END_STRUCT;
END_TYPE

TYPE M_McReadBoolParameter : STRUCT
  {attribute 'OPC.UA.DA' := '1'}
  {attribute 'OPC.UA.DA.Access' := '1'}
  {attribute 'TcHmiSymbol.Show'}
  value : BOOL;
  {attribute 'OPC.UA.DA' := '1'}
  {attribute 'OPC.UA.DA.Access' := '3'}
  {attribute 'TcHmiSymbol.Show'}
  set : McReadBoolParameterArgs;
END_STRUCT;
END_TYPE

TYPE M_McProbe : STRUCT
  {attribute 'OPC.UA.DA' := '1'}
  {attribute 'OPC.UA.DA.Access' := '1'}
  {attribute 'TcHmiSymbol.Show'}
  recordedPosition : LREAL;
  {attribute 'OPC.UA.DA' := '1'}
  {attribute 'OPC.UA.DA.Access' := '3'}
  {attribute 'TcHmiSymbol.Show'}
  set : McProbeArgs;
END_STRUCT;
END_TYPE

TYPE M_ChangeOperatingStateProcess : STRUCT
  {attribute 'OPC.UA.DA' := '1'}
  {attribute 'OPC.UA.DA.Access' := '3'}
  {attribute 'TcHmiSymbol.Show'}
  set : ChangeOperatingStateProcessArgs;
END_STRUCT;
END_TYPE

TYPE M_ChangeOperatorStateProcess : STRUCT
  {attribute 'OPC.UA.DA' := '1'}
  {attribute 'OPC.UA.DA.Access' := '3'}
  {attribute 'TcHmiSymbol.Show'}
  set : ChangeOperatorStateProcessArgs;
END_STRUCT;
END_TYPE

TYPE M_ChangeOperatingModeStateProcess : STRUCT
  {attribute 'OPC.UA.DA' := '1'}
  {attribute 'OPC.UA.DA.Access' := '3'}
  {attribute 'TcHmiSymbol.Show'}
  set : ChangeOperatingModeStateProcessArgs;
END_STRUCT;
END_TYPE

TYPE M_ReadXmlProcess : STRUCT
  {attribute 'OPC.UA.DA' := '1'}
  {attribute 'OPC.UA.DA.Access' := '3'}
  {attribute 'TcHmiSymbol.Show'}
  set : ReadXmlProcessArgs;
END_STRUCT;
END_TYPE

TYPE M_WriteXmlProcess : STRUCT
  {attribute 'OPC.UA.DA' := '1'}
  {attribute 'OPC.UA.DA.Access' := '3'}
  {attribute 'TcHmiSymbol.Show'}
  set : WriteXmlProcessArgs;
END_STRUCT;
END_TYPE

TYPE M_ActivateProcess : STRUCT

END_STRUCT;
END_TYPE

TYPE M_ModbusRTUBusReadCoilProcess : STRUCT
  {attribute 'OPC.UA.DA' := '1'}
  {attribute 'OPC.UA.DA.Access' := '1'}
  {attribute 'TcHmiSymbol.Show'}
  value : BOOL;
  {attribute 'OPC.UA.DA' := '1'}
  {attribute 'OPC.UA.DA.Access' := '1'}
  {attribute 'TcHmiSymbol.Show'}
  errorId : INT;
  {attribute 'OPC.UA.DA' := '1'}
  {attribute 'OPC.UA.DA.Access' := '3'}
  {attribute 'TcHmiSymbol.Show'}
  set : ModbusRTUBusReadCoilProcessArgs;
END_STRUCT;
END_TYPE

TYPE M_ModbusRTUBusWriteCoilProcess : STRUCT
  {attribute 'OPC.UA.DA' := '1'}
  {attribute 'OPC.UA.DA.Access' := '1'}
  {attribute 'TcHmiSymbol.Show'}
  errorId : INT;
  {attribute 'OPC.UA.DA' := '1'}
  {attribute 'OPC.UA.DA.Access' := '3'}
  {attribute 'TcHmiSymbol.Show'}
  set : ModbusRTUBusWriteCoilProcessArgs;
END_STRUCT;
END_TYPE

TYPE M_ModbusRTUBusReadRegisterProcess : STRUCT
  {attribute 'OPC.UA.DA' := '1'}
  {attribute 'OPC.UA.DA.Access' := '1'}
  {attribute 'TcHmiSymbol.Show'}
  value : INT;
  {attribute 'OPC.UA.DA' := '1'}
  {attribute 'OPC.UA.DA.Access' := '1'}
  {attribute 'TcHmiSymbol.Show'}
  errorId : INT;
  {attribute 'OPC.UA.DA' := '1'}
  {attribute 'OPC.UA.DA.Access' := '3'}
  {attribute 'TcHmiSymbol.Show'}
  set : ModbusRTUBusReadRegisterProcessArgs;
END_STRUCT;
END_TYPE

TYPE M_ModbusRTUBusWriteRegisterProcess : STRUCT
  {attribute 'OPC.UA.DA' := '1'}
  {attribute 'OPC.UA.DA.Access' := '1'}
  {attribute 'TcHmiSymbol.Show'}
  errorId : INT;
  {attribute 'OPC.UA.DA' := '1'}
  {attribute 'OPC.UA.DA.Access' := '3'}
  {attribute 'TcHmiSymbol.Show'}
  set : ModbusRTUBusWriteRegisterProcessArgs;
END_STRUCT;
END_TYPE

TYPE M_ModbusRTUBusDiagnosticsProcess : STRUCT
  {attribute 'OPC.UA.DA' := '1'}
  {attribute 'OPC.UA.DA.Access' := '1'}
  {attribute 'TcHmiSymbol.Show'}
  value : INT;
  {attribute 'OPC.UA.DA' := '1'}
  {attribute 'OPC.UA.DA.Access' := '1'}
  {attribute 'TcHmiSymbol.Show'}
  errorId : INT;
  {attribute 'OPC.UA.DA' := '1'}
  {attribute 'OPC.UA.DA.Access' := '3'}
  {attribute 'TcHmiSymbol.Show'}
  set : ModbusRTUBusDiagnosticsProcessArgs;
END_STRUCT;
END_TYPE

TYPE M_PointAlphaDeltaProcess : STRUCT
  {attribute 'OPC.UA.DA' := '1'}
  {attribute 'OPC.UA.DA.Access' := '3'}
  {attribute 'TcHmiSymbol.Show'}
  set : PointAlphaDeltaProcessArgs;
END_STRUCT;
END_TYPE

TYPE M_GigECameraSetParamProcess : STRUCT
  {attribute 'OPC.UA.DA' := '1'}
  {attribute 'OPC.UA.DA.Access' := '3'}
  {attribute 'TcHmiSymbol.Show'}
  set : GigECameraSetParamProcessArgs;
END_STRUCT;
END_TYPE

TYPE M_GigECameraSetParam2Process : STRUCT
  {attribute 'OPC.UA.DA' := '1'}
  {attribute 'OPC.UA.DA.Access' := '3'}
  {attribute 'TcHmiSymbol.Show'}
  set : GigECameraSetParam2ProcessArgs;
END_STRUCT;
END_TYPE

TYPE M_GigECameraPulseTrigger : STRUCT
  {attribute 'OPC.UA.DA' := '1'}
  {attribute 'OPC.UA.DA.Access' := '3'}
  {attribute 'TcHmiSymbol.Show'}
  set : GigECameraPulseTriggerArgs;
END_STRUCT;
END_TYPE

TYPE M_GigECameraSetSourceProcess : STRUCT
  {attribute 'OPC.UA.DA' := '1'}
  {attribute 'OPC.UA.DA.Access' := '3'}
  {attribute 'TcHmiSymbol.Show'}
  set : GigECameraSetSourceProcessArgs;
END_STRUCT;
END_TYPE

TYPE M_GigECameraSetupProcess : STRUCT
  {attribute 'OPC.UA.DA' := '1'}
  {attribute 'OPC.UA.DA.Access' := '3'}
  {attribute 'TcHmiSymbol.Show'}
  set : GigECameraSetupProcessArgs;
END_STRUCT;
END_TYPE

TYPE M_GigECameraMultiTriggerProcess : STRUCT
  {attribute 'OPC.UA.DA' := '1'}
  {attribute 'OPC.UA.DA.Access' := '3'}
  {attribute 'TcHmiSymbol.Show'}
  set : GigECameraMultiTriggerProcessArgs;
END_STRUCT;
END_TYPE

TYPE M_Arg1LrealProcess : STRUCT
  {attribute 'OPC.UA.DA' := '1'}
  {attribute 'OPC.UA.DA.Access' := '3'}
  {attribute 'TcHmiSymbol.Show'}
  set : Arg1LrealProcessArgs;
END_STRUCT;
END_TYPE

TYPE M_Ell114SendProcess : STRUCT
  {attribute 'OPC.UA.DA' := '1'}
  {attribute 'OPC.UA.DA.Access' := '1'}
  {attribute 'TcHmiSymbol.Show'}
  reply : STRING;
  {attribute 'OPC.UA.DA' := '1'}
  {attribute 'OPC.UA.DA.Access' := '3'}
  {attribute 'TcHmiSymbol.Show'}
  set : Ell114SendProcessArgs;
END_STRUCT;
END_TYPE

TYPE M_SM_BaseAxisProcesses : STRUCT
  {attribute 'TcHmiSymbol.Show'}
  moveAbsolute : M_McMoveAbsoluteProcess;
  {attribute 'TcHmiSymbol.Show'}
  moveRelative : M_McMoveRelativeProcess;
  {attribute 'TcHmiSymbol.Show'}
  moveVelocity : M_McMoveVelocityProcess;
  {attribute 'TcHmiSymbol.Show'}
  reset : M_McProcess;
  {attribute 'TcHmiSymbol.Show'}
  stop : M_McProcess;
  {attribute 'TcHmiSymbol.Show'}
  stopParametrized : M_McStopProcess;
  {attribute 'TcHmiSymbol.Show'}
  power : M_McPowerProcess;
  {attribute 'TcHmiSymbol.Show'}
  home : M_McProcess;
  {attribute 'TcHmiSymbol.Show'}
  initialize : M_Process;
  {attribute 'TcHmiSymbol.Show'}
  setPosition : M_McSetPositionProcess;
  {attribute 'TcHmiSymbol.Show'}
  readParameter : M_McReadParameter;
  {attribute 'TcHmiSymbol.Show'}
  readBoolParameter : M_McReadBoolParameter;
  {attribute 'TcHmiSymbol.Show'}
  writeParameter : M_McWriteParameter;
  {attribute 'TcHmiSymbol.Show'}
  writeBoolParameter : M_McWriteBoolParameter;
END_STRUCT;
END_TYPE

TYPE M_SM_IncrementalEncoderProcesses : STRUCT
  {attribute 'TcHmiSymbol.Show'}
  enableCounterResetC : M_Process;
  {attribute 'TcHmiSymbol.Show'}
  disableCounterResetC : M_Process;
END_STRUCT;
END_TYPE

TYPE M_SM_SimpleRelayProcesses : STRUCT
  {attribute 'TcHmiSymbol.Show'}
  setEnabled : M_SetEnabledProcess;
END_STRUCT;
END_TYPE

TYPE M_SM_FuseProcesses : STRUCT
  {attribute 'TcHmiSymbol.Show'}
  setEnabled : M_SetEnabledProcess;
  {attribute 'TcHmiSymbol.Show'}
  reset : M_Process;
END_STRUCT;
END_TYPE

TYPE M_SM_LedProcesses : STRUCT
  {attribute 'TcHmiSymbol.Show'}
  setMilliAmps : M_ChangeSetpointProcess;
END_STRUCT;
END_TYPE

TYPE M_SM_TipTiltProcesses : STRUCT
  {attribute 'TcHmiSymbol.Show'}
  setV1 : M_ChangeSetpointProcess;
  {attribute 'TcHmiSymbol.Show'}
  setV2 : M_ChangeSetpointProcess;
  {attribute 'TcHmiSymbol.Show'}
  setV3 : M_ChangeSetpointProcess;
END_STRUCT;
END_TYPE

TYPE M_SM_ConfigManagerProcesses : STRUCT
  {attribute 'TcHmiSymbol.Show'}
  save : M_WriteXmlProcess;
  {attribute 'TcHmiSymbol.Show'}
  load : M_ReadXmlProcess;
  {attribute 'TcHmiSymbol.Show'}
  activate : M_ActivateProcess;
END_STRUCT;
END_TYPE

TYPE M_SM_ModbusRTUBusProcesses : STRUCT
  {attribute 'TcHmiSymbol.Show'}
  readCoil : M_ModbusRTUBusReadCoilProcess;
  {attribute 'TcHmiSymbol.Show'}
  writeCoil : M_ModbusRTUBusWriteCoilProcess;
  {attribute 'TcHmiSymbol.Show'}
  readRegister : M_ModbusRTUBusReadRegisterProcess;
  {attribute 'TcHmiSymbol.Show'}
  writeRegister : M_ModbusRTUBusWriteRegisterProcess;
  {attribute 'TcHmiSymbol.Show'}
  diagnostics : M_ModbusRTUBusDiagnosticsProcess;
END_STRUCT;
END_TYPE

TYPE M_SM_GigECameraProcesses : STRUCT
  {attribute 'TcHmiSymbol.Show'}
  open : M_Process;
  {attribute 'TcHmiSymbol.Show'}
  close : M_Process;
  {attribute 'TcHmiSymbol.Show'}
  startAcquiring : M_Process;
  {attribute 'TcHmiSymbol.Show'}
  stopAcquiring : M_Process;
  {attribute 'TcHmiSymbol.Show'}
  reset : M_Process;
  {attribute 'TcHmiSymbol.Show'}
  setup : M_GigECameraSetupProcess;
  {attribute 'TcHmiSymbol.Show'}
  setParam : M_GigECameraSetParamProcess;
  {attribute 'TcHmiSymbol.Show'}
  setParam2 : M_GigECameraSetParam2Process;
  {attribute 'TcHmiSymbol.Show'}
  trigger : M_Process;
  {attribute 'TcHmiSymbol.Show'}
  pulseTrigger : M_GigECameraPulseTrigger;
  {attribute 'TcHmiSymbol.Show'}
  multiTrigger : M_GigECameraMultiTriggerProcess;
  {attribute 'TcHmiSymbol.Show'}
  multiTriggerAbort : M_Process;
  {attribute 'TcHmiSymbol.Show'}
  setSource : M_GigECameraSetSourceProcess;
END_STRUCT;
END_TYPE

TYPE M_SM_ELL14StageProcesses : STRUCT
  {attribute 'TcHmiSymbol.Show'}
  moveAbs : M_Arg1LrealProcess;
  {attribute 'TcHmiSymbol.Show'}
  moveRel : M_Arg1LrealProcess;
  {attribute 'TcHmiSymbol.Show'}
  send : M_Ell114SendProcess;
END_STRUCT;
END_TYPE

TYPE M_SM_SequencerParts : STRUCT
  {attribute 'TcHmiSymbol.Show'}
  configManager : M_ConfigManager;
END_STRUCT;
END_TYPE

TYPE M_SM_SequencerProcesses : STRUCT
  {attribute 'TcHmiSymbol.Show'}
  selectEditable : M_IndexProcess;
  {attribute 'TcHmiSymbol.Show'}
  selectRunnable : M_IndexProcess;
  {attribute 'TcHmiSymbol.Show'}
  start : M_IdProcess;
  {attribute 'TcHmiSymbol.Show'}
  stop : M_Process;
  {attribute 'TcHmiSymbol.Show'}
  apply : M_Process;
  {attribute 'TcHmiSymbol.Show'}
  cancel : M_Process;
END_STRUCT;
END_TYPE

{attribute 'TcRpcEnable' := '1'}
FUNCTION F_ApertureStatus : ApertureStatus
  VAR_INPUT
    superState : BOOL := TRUE;  (* Super state (TRUE if the super state is active, or if there is no super state) *)
    isOpen : BOOL;  (* TRUE if the 'open' limit switch is active *)
    isClosed : BOOL;  (* TRUE if the 'open' limit switch is active *)
  END_VAR

              IF NOT(superState) THEN
    F_ApertureStatus := ApertureStatus.unknown;
ELSIF isOpen AND (NOT(isClosed)) THEN
    F_ApertureStatus := ApertureStatus.open;
ELSIF isClosed AND (NOT(isOpen)) THEN
    F_ApertureStatus := ApertureStatus.closed;
ELSIF NOT(isOpen OR isClosed) THEN
    F_ApertureStatus := ApertureStatus.partiallyOpen;
ELSIF isOpen AND isClosed THEN
    F_ApertureStatus := ApertureStatus.undefined;
ELSE
    F_ApertureStatus := ApertureStatus.invalid_model;
END_IF;

            
END_FUNCTION

{attribute 'TcRpcEnable' := '1'}
FUNCTION F_BusyStatus : BusyStatus
  VAR_INPUT
    superState : BOOL := TRUE;  (* Super state (TRUE if the super state is active, or if there is no super state) *)
    isBusy : BOOL;  (* TRUE if busy *)
  END_VAR

              IF NOT(superState) THEN
    F_BusyStatus := BusyStatus.unknown;
ELSIF NOT(isBusy) THEN
    F_BusyStatus := BusyStatus.idle;
ELSIF isBusy THEN
    F_BusyStatus := BusyStatus.busy;
ELSE
    F_BusyStatus := BusyStatus.invalid_model;
END_IF;

            
END_FUNCTION

{attribute 'TcRpcEnable' := '1'}
FUNCTION F_StartedStatus : StartedStatus
  VAR_INPUT
    superState : BOOL := TRUE;  (* Super state (TRUE if the super state is active, or if there is no super state) *)
    isStarted : BOOL;  (* TRUE if started *)
  END_VAR

              IF NOT(superState) THEN
    F_StartedStatus := StartedStatus.unknown;
ELSIF isStarted THEN
    F_StartedStatus := StartedStatus.started;
ELSIF NOT(isStarted) THEN
    F_StartedStatus := StartedStatus.notStarted;
ELSE
    F_StartedStatus := StartedStatus.invalid_model;
END_IF;

            
END_FUNCTION

{attribute 'TcRpcEnable' := '1'}
FUNCTION F_EnabledStatus : EnabledStatus
  VAR_INPUT
    superState : BOOL := TRUE;  (* Super state (TRUE if the super state is active, or if there is no super state) *)
    isEnabled : BOOL;  (* TRUE if enabled *)
  END_VAR

              IF NOT(superState) THEN
    F_EnabledStatus := EnabledStatus.unknown;
ELSIF isEnabled THEN
    F_EnabledStatus := EnabledStatus.enabled;
ELSIF NOT(isEnabled) THEN
    F_EnabledStatus := EnabledStatus.disabled;
ELSE
    F_EnabledStatus := EnabledStatus.invalid_model;
END_IF;

            
END_FUNCTION

{attribute 'TcRpcEnable' := '1'}
FUNCTION F_PoweredStatus : PoweredStatus
  VAR_INPUT
    superState : BOOL := TRUE;  (* Super state (TRUE if the super state is active, or if there is no super state) *)
    isEnabled : BOOL;  (* TRUE if power is enabled *)
  END_VAR

              IF NOT(superState) THEN
    F_PoweredStatus := PoweredStatus.unknown;
ELSIF isEnabled THEN
    F_PoweredStatus := PoweredStatus.enabled;
ELSIF NOT(isEnabled) THEN
    F_PoweredStatus := PoweredStatus.disabled;
ELSE
    F_PoweredStatus := PoweredStatus.invalid_model;
END_IF;

            
END_FUNCTION

{attribute 'TcRpcEnable' := '1'}
FUNCTION F_HealthStatus : HealthStatus
  VAR_INPUT
    superState : BOOL := TRUE;  (* Super state (TRUE if the super state is active, or if there is no super state) *)
    isGood : BOOL;  (* TRUE if the subject is in Good health *)
    hasWarning : BOOL := FALSE;  (* TRUE to add a warning to the Good health state *)
  END_VAR

              IF NOT(superState) THEN
    F_HealthStatus := HealthStatus.unknown;
ELSIF isGood AND (NOT(hasWarning)) THEN
    F_HealthStatus := HealthStatus.good;
ELSIF isGood AND hasWarning THEN
    F_HealthStatus := HealthStatus.warning;
ELSIF NOT(isGood) THEN
    F_HealthStatus := HealthStatus.bad;
ELSE
    F_HealthStatus := HealthStatus.invalid_model;
END_IF;

            
END_FUNCTION

{attribute 'TcRpcEnable' := '1'}
FUNCTION F_InitializationStatus : InitializationStatus
  VAR_INPUT
    superState : BOOL := TRUE;  (* Super state (TRUE if the super state is active, or if there is no super state) *)
    state : InitializationStates;  (* Enum! *)
  END_VAR

              IF NOT(superState) THEN
    F_InitializationStatus := InitializationStatus.unknown;
ELSIF state = InitializationStates.SHUTDOWN THEN
    F_InitializationStatus := InitializationStatus.shutdown;
ELSIF state = InitializationStates.INITIALIZING THEN
    F_InitializationStatus := InitializationStatus.initializing;
ELSIF state = InitializationStates.INITIALIZING_FAILED THEN
    F_InitializationStatus := InitializationStatus.initializingFailed;
ELSIF state = InitializationStates.INITIALIZED THEN
    F_InitializationStatus := InitializationStatus.initialized;
ELSIF state = InitializationStates.LOCKED THEN
    F_InitializationStatus := InitializationStatus.locked;
ELSE
    F_InitializationStatus := InitializationStatus.invalid_model;
END_IF;

            
END_FUNCTION

{attribute 'TcRpcEnable' := '1'}
FUNCTION F_MotionStatus : MotionStatus
  VAR_INPUT
    superState : BOOL := TRUE;  (* Super state (TRUE if the super state is active, or if there is no super state) *)
    actVel : LREAL;  (* Actual velocity *)
    tolerance : LREAL;  (* Tolerance (should be positive)! *)
  END_VAR

              IF NOT(superState) THEN
    F_MotionStatus := MotionStatus.unknown;
ELSIF actVel > (ABS(tolerance)) THEN
    F_MotionStatus := MotionStatus.forward;
ELSIF actVel < (-(ABS(tolerance))) THEN
    F_MotionStatus := MotionStatus.backward;
ELSIF TRUE THEN
    F_MotionStatus := MotionStatus.standstill;
ELSE
    F_MotionStatus := MotionStatus.invalid_model;
END_IF;

            
END_FUNCTION

{attribute 'TcRpcEnable' := '1'}
FUNCTION F_HiHiLoLoAlarmStatus : HiHiLoLoAlarmStatus
  VAR_INPUT
    superState : BOOL := TRUE;  (* Super state (TRUE if the super state is active, or if there is no super state) *)
    config : HiHiLoLoAlarmConfig;  (* Config *)
    value : LREAL;  (* Value in the correct units to compare to the values from the config *)
  END_VAR

              IF NOT(superState) THEN
    F_HiHiLoLoAlarmStatus := HiHiLoLoAlarmStatus.unknown;
ELSIF NOT(config.enabled) THEN
    F_HiHiLoLoAlarmStatus := HiHiLoLoAlarmStatus.disabled;
ELSIF config.enabled AND (value >= config.hiHi) THEN
    F_HiHiLoLoAlarmStatus := HiHiLoLoAlarmStatus.hiHi;
ELSIF config.enabled AND ((value >= config.hi) AND (value < config.hiHi)) THEN
    F_HiHiLoLoAlarmStatus := HiHiLoLoAlarmStatus.hi;
ELSIF config.enabled AND ((value > config.lo) AND (value < config.hi)) THEN
    F_HiHiLoLoAlarmStatus := HiHiLoLoAlarmStatus.ok;
ELSIF config.enabled AND ((value <= config.lo) AND (value < config.loLo)) THEN
    F_HiHiLoLoAlarmStatus := HiHiLoLoAlarmStatus.lo;
ELSIF config.enabled AND (value <= config.loLo) THEN
    F_HiHiLoLoAlarmStatus := HiHiLoLoAlarmStatus.loLo;
ELSE
    F_HiHiLoLoAlarmStatus := HiHiLoLoAlarmStatus.invalid_model;
END_IF;

            
END_FUNCTION

{attribute 'TcRpcEnable' := '1'}
FUNCTION F_OpeningStatus : OpeningStatus
  VAR_INPUT
    superState : BOOL := TRUE;  (* Super state (TRUE if the super state is active, or if there is no super state) *)
    isOpening : BOOL;  (* TRUE if opening *)
    isClosing : BOOL;  (* TRUE if closing *)
  END_VAR

              IF NOT(superState) THEN
    F_OpeningStatus := OpeningStatus.unknown;
ELSIF isOpening AND (NOT(isClosing)) THEN
    F_OpeningStatus := OpeningStatus.opening;
ELSIF isClosing AND (NOT(isOpening)) THEN
    F_OpeningStatus := OpeningStatus.closing;
ELSIF NOT(isClosing OR isOpening) THEN
    F_OpeningStatus := OpeningStatus.standstill;
ELSE
    F_OpeningStatus := OpeningStatus.invalid_model;
END_IF;

            
END_FUNCTION

{attribute 'TcRpcEnable' := '1'}
FUNCTION F_OperatorStatus : OperatorStatus
  VAR_INPUT
    superState : BOOL := TRUE;  (* Super state (TRUE if the super state is active, or if there is no super state) *)
    state : OperatorStates;  (* Enum! *)
  END_VAR

              IF NOT(superState) THEN
    F_OperatorStatus := OperatorStatus.unknown;
ELSIF state = OperatorStates.NONE THEN
    F_OperatorStatus := OperatorStatus.none;
ELSIF state = OperatorStates.TECH THEN
    F_OperatorStatus := OperatorStatus.tech;
ELSIF state = OperatorStates.OBSERVER THEN
    F_OperatorStatus := OperatorStatus.observer;
ELSE
    F_OperatorStatus := OperatorStatus.invalid_model;
END_IF;

            
END_FUNCTION

{attribute 'TcRpcEnable' := '1'}
FUNCTION F_OperatingStatus : OperatingStatus
  VAR_INPUT
    superState : BOOL := TRUE;  (* Super state (TRUE if the super state is active, or if there is no super state) *)
    state : OperatingStates;  (* Enum! *)
  END_VAR

              IF NOT(superState) THEN
    F_OperatingStatus := OperatingStatus.unknown;
ELSIF state = OperatingStates.AUTO THEN
    F_OperatingStatus := OperatingStatus.auto;
ELSIF state = OperatingStates.MANUAL THEN
    F_OperatingStatus := OperatingStatus.manual;
ELSE
    F_OperatingStatus := OperatingStatus.invalid_model;
END_IF;

            
END_FUNCTION

{attribute 'TcRpcEnable' := '1'}
FUNCTION F_OperatingModeStatus : OperatingModeStatus
  VAR_INPUT
    superState : BOOL := TRUE;  (* Super state (TRUE if the super state is active, or if there is no super state) *)
    state : OperatingModeStates;  (* Enum! *)
  END_VAR

              IF NOT(superState) THEN
    F_OperatingModeStatus := OperatingModeStatus.unknown;
ELSIF state = OperatingModeStates.LOCAL THEN
    F_OperatingModeStatus := OperatingModeStatus.local;
ELSIF state = OperatingModeStates.REMOTE THEN
    F_OperatingModeStatus := OperatingModeStatus.remote;
ELSE
    F_OperatingModeStatus := OperatingModeStatus.invalid_model;
END_IF;

            
END_FUNCTION

{attribute 'TcRpcEnable' := '1'}
FUNCTION F_ActivityStatus : ActivityStatus
  VAR_INPUT
    superState : BOOL := TRUE;  (* Super state (TRUE if the super state is active, or if there is no super state) *)
    isRunning : BOOL;
  END_VAR

              IF NOT(superState) THEN
    F_ActivityStatus := ActivityStatus.unknown;
ELSIF NOT(isRunning) THEN
    F_ActivityStatus := ActivityStatus.notRunning;
ELSIF isRunning THEN
    F_ActivityStatus := ActivityStatus.running;
ELSE
    F_ActivityStatus := ActivityStatus.invalid_model;
END_IF;

            
END_FUNCTION

FUNCTION_BLOCK SM_BaseProcess
  VAR_INPUT
    {attribute 'OPC.UA.DA' := '0'}
    isEnabled : BOOL;  (* Should the trigger be enabled? *)
    {attribute 'OPC.UA.DA' := '0'}
    atomic : AtomicRequest;  (* Handle of the request *)
  END_VAR
  VAR_OUTPUT
    {attribute 'OPC.UA.DA' := '1'}
    {attribute 'OPC.UA.DA.Access' := '1'}
    actualStatus : STRING(50);  (* Current status description *)
    {attribute 'OPC.UA.DA' := '1'}
    {attribute 'OPC.UA.DA.Access' := '1'}
    atomic_out : ULINT;  (* Atomic output variable *)
    {attribute 'OPC.UA.DA' := '1'}
    {attribute 'OPC.UA.DA.Access' := '1'}
    lastRejectedHandle : UDINT;  (* Handle of the last rejected request *)
    {attribute 'OPC.UA.DA' := '1'}
    stat : BaseProcessStatuses;  (* Statuses of the state machine *)
  END_VAR
  VAR
    {attribute 'OPC.UA.DA' := '1'}
    {attribute 'OPC.UA.DA.Access' := '3'}
    do_request : BOOL;  (* Write TRUE to request the start of the process *)
    {attribute 'OPC.UA.DA' := '1'}
    {attribute 'OPC.UA.DA.Access' := '3'}
    atomic_in : ULINT;  (* Atomic input variable (4 bytes ) *)
    {attribute 'OPC.UA.DA' := '1'}
    do_request_result : RequestResults;  (* Result of the request *)
  END_VAR

            stat.enabled := F_EnabledStatus(
    superState := TRUE,
    isEnabled := isEnabled);

          

METHOD _copyFromModel_SM_BaseProcess
  VAR_IN_OUT
    {attribute 'OPC.UA.DA' := '0'}
    model : M_SM_BaseProcess;
  END_VAR
                  THIS^.do_request := model.do_request;
THIS^.atomic_in := model.atomic_in;

                
END_METHOD

METHOD _copyToModel_SM_BaseProcess
  VAR_IN_OUT
    {attribute 'OPC.UA.DA' := '0'}
    model : M_SM_BaseProcess;
  END_VAR
                  model.do_request := THIS^.do_request;
model.atomic_in := THIS^.atomic_in;
model.do_request_result := THIS^.do_request_result;
model.actualStatus := THIS^.actualStatus;
model.atomic_out := THIS^.atomic_out;
model.lastRejectedHandle := THIS^.lastRejectedHandle;
model.stat := THIS^.stat;

                
END_METHOD
END_FUNCTION_BLOCK

FUNCTION_BLOCK SM_BaseMcProcess EXTENDS BaseProcess
  VAR_INPUT
    {attribute 'OPC.UA.DA' := '1'}
    {attribute 'OPC.UA.DA.Access' := '1'}
    errorId : UDINT;  (* Error ID according to Beckhoff/PlcOpen Motion Control *)
  END_VAR

            SUPER^();

          

METHOD _copyFromModel_SM_BaseMcProcess
  VAR_IN_OUT
    {attribute 'OPC.UA.DA' := '0'}
    model : M_SM_BaseMcProcess;
  END_VAR
                  SUPER^._copyFromModel_BaseProcess( model := model );

                
END_METHOD

METHOD _copyToModel_SM_BaseMcProcess
  VAR_IN_OUT
    {attribute 'OPC.UA.DA' := '0'}
    model : M_SM_BaseMcProcess;
  END_VAR
                  model.errorId := THIS^.errorId;
SUPER^._copyToModel_BaseProcess( model := model );

                
END_METHOD
END_FUNCTION_BLOCK

FUNCTION_BLOCK SM_ProcessStep
  VAR_INPUT
    {attribute 'OPC.UA.DA' := '0'}
    isEnabled : BOOL;  (* Is the step enabled? *)
  END_VAR
  VAR_OUTPUT
    {attribute 'OPC.UA.DA' := '1'}
    {attribute 'OPC.UA.DA.Access' := '1'}
    actualStatus : STRING(50);  (* Current status description *)
    {attribute 'OPC.UA.DA' := '1'}
    stat : ProcessStepStatuses;  (* Statuses of the state machine *)
  END_VAR
  VAR_IN_OUT
    {attribute 'OPC.UA.DA' := '0'}
    process : BaseProcess;  (* The process corresponding to the step *)
  END_VAR

            stat.enabled := F_EnabledStatus(
    superState := TRUE,
    isEnabled := isEnabled);

          

METHOD _copyFromModel_SM_ProcessStep
  VAR_IN_OUT
    {attribute 'OPC.UA.DA' := '0'}
    model : M_SM_ProcessStep;
  END_VAR
                  
                
END_METHOD

METHOD _copyToModel_SM_ProcessStep
  VAR_IN_OUT
    {attribute 'OPC.UA.DA' := '0'}
    model : M_SM_ProcessStep;
  END_VAR
                  model.actualStatus := THIS^.actualStatus;
model.stat := THIS^.stat;

                
END_METHOD
END_FUNCTION_BLOCK

FUNCTION_BLOCK SM_BaseXmlDataSrvProcess EXTENDS BaseProcess
  VAR_INPUT
    {attribute 'OPC.UA.DA' := '1'}
    {attribute 'OPC.UA.DA.Access' := '1'}
    errorId : UDINT;  (* Error ID according to Beckhoff XML Data Server library *)
  END_VAR

            SUPER^();

          

METHOD _copyFromModel_SM_BaseXmlDataSrvProcess
  VAR_IN_OUT
    {attribute 'OPC.UA.DA' := '0'}
    model : M_SM_BaseXmlDataSrvProcess;
  END_VAR
                  SUPER^._copyFromModel_BaseProcess( model := model );

                
END_METHOD

METHOD _copyToModel_SM_BaseXmlDataSrvProcess
  VAR_IN_OUT
    {attribute 'OPC.UA.DA' := '0'}
    model : M_SM_BaseXmlDataSrvProcess;
  END_VAR
                  model.errorId := THIS^.errorId;
SUPER^._copyToModel_BaseProcess( model := model );

                
END_METHOD
END_FUNCTION_BLOCK

FUNCTION_BLOCK SM_BaseAxis
  VAR_INPUT
    {attribute 'OPC.UA.DA' := '1'}
    {attribute 'OPC.UA.DA.Access' := '1'}
    isGearingSupported : BOOL := FALSE;  (* Is gearIn/gearOut supported? *)
    {attribute 'TcHmiSymbol.Hide'}
    {attribute 'OPC.UA.DA' := '1'}
    {attribute 'OPC.UA.DA.Access' := '1'}
    axis_ref : AXIS_REF;  (* The AXIS_REF to be linked to the NC I/O *)
    {attribute 'OPC.UA.DA' := '0'}
    isEnabled : BOOL;  (* Is control enabled? *)
    {attribute 'OPC.UA.DA' := '0'}
    standstillTolerance : LREAL;  (* Tolerance in [main units] per second: if < ABS(this value), then the axis is considered to be standing still *)
    {attribute 'OPC.UA.DA' := '0'}
    _axis_ref : REFERENCE TO AXIS_REF;  (* The AXIS_REF to be linked to the NC I/O *)
    {attribute 'OPC.UA.DA' := '0'}
    usePosLimitSwitch : BOOL := FALSE;  (* TRUE to use a hardware forward limit switch *)
    {attribute 'OPC.UA.DA' := '0'}
    useNegLimitSwitch : BOOL := FALSE;  (* TRUE to use a hardware reverse limit switch *)
    {attribute 'OPC.UA.DA' := '0'}
    posLimitSwitchSig AT %I* : BOOL;  (* Limit switch raw signal in forward direction (e.g. at +105 mm for a stage of 100 mm travel range *)
    {attribute 'OPC.UA.DA' := '0'}
    negLimitSwitchSig AT %I* : BOOL;  (* Limit switch raw signal in negative direction (e.g. at or a little bit below 0 mm) *)
    {attribute 'OPC.UA.DA' := '0'}
    invertPosLimitSwitch : BOOL;  (* Invert positive limit switch raw signal *)
    {attribute 'OPC.UA.DA' := '0'}
    invertNegLimitSwitch : BOOL;  (* Invert positive limit switch raw signal *)
  END_VAR
  VAR_OUTPUT
    {attribute 'OPC.UA.DA' := '1'}
    {attribute 'OPC.UA.DA.Access' := '1'}
    actualStatus : STRING(50);  (* Current status description *)
    {attribute 'OPC.UA.DA' := '1'}
    {attribute 'OPC.UA.DA.Access' := '1'}
    isJogEnabled : BOOL;  (* True if jog is enabled *)
    {attribute 'OPC.UA.DA' := '1'}
    {attribute 'OPC.UA.DA.Access' := '1'}
    errorId : UDINT;  (* Axis error ID *)
    {attribute 'OPC.UA.DA' := '1'}
    {attribute 'OPC.UA.DA.Access' := '1'}
    posLimitSwitch : BOOL;  (* Limit switch in forward direction (e.g. at +105 mm for a stage of 100 mm travel range *)
    {attribute 'OPC.UA.DA' := '1'}
    {attribute 'OPC.UA.DA.Access' := '1'}
    negLimitSwitch : BOOL;  (* Limit switch in negative direction (e.g. at or a little bit below 0 mm) *)
    {attribute 'OPC.UA.DA' := '1'}
    stat : BaseAxisStatuses;  (* Statuses of the state machine *)
    {attribute 'OPC.UA.DA' := '1'}
    proc : BaseAxisProcesses;  (* Processes of the state machine *)
  END_VAR

            stat.busy := F_BusyStatus(
    superState := TRUE,
    isBusy := (proc.moveAbsolute.stat.busy = BusyStatus.busy) OR ((proc.moveRelative.stat.busy = BusyStatus.busy) OR ((proc.reset.stat.busy = BusyStatus.busy) OR ((proc.power.stat.busy = BusyStatus.busy) OR ((proc.initialize.stat.busy = BusyStatus.busy) OR ((proc.setPosition.stat.busy = BusyStatus.busy) OR ((proc.readParameter.stat.busy = BusyStatus.busy) OR ((proc.readBoolParameter.stat.busy = BusyStatus.busy) OR ((proc.writeParameter.stat.busy = BusyStatus.busy) OR ((proc.writeBoolParameter.stat.busy = BusyStatus.busy) OR (proc.home.stat.busy = BusyStatus.busy)))))))))));
stat.health := F_HealthStatus(
    superState := TRUE,
    isGood := NOT(_axis_ref.Status.Error),
    hasWarning := FALSE);
stat.powered := F_PoweredStatus(
    superState := TRUE,
    isEnabled := NOT(_axis_ref.Status.Disabled));
stat.extSetGen := F_EnabledStatus(
    superState := TRUE,
    isEnabled := _axis_ref.Status.ExtSetPointGenEnabled);
stat.motion := F_MotionStatus(
    superState := TRUE,
    actVel := _axis_ref.NcToPlc.ActVelo,
    tolerance := standstillTolerance);
proc.moveAbsolute( isEnabled := isEnabled );
proc.moveRelative( isEnabled := isEnabled );
proc.moveVelocity( isEnabled := isEnabled AND (proc.moveVelocity.stat.busy = BusyStatus.idle) );
proc.reset( isEnabled := isEnabled AND (proc.reset.stat.busy = BusyStatus.idle) );
proc.stop( isEnabled := isEnabled AND (proc.stop.stat.busy = BusyStatus.idle) );
proc.stopParametrized();
proc.power( isEnabled := isEnabled AND (proc.power.stat.busy = BusyStatus.idle) );
proc.home( isEnabled := isEnabled AND (stat.busy = BusyStatus.idle) );
proc.initialize( isEnabled := isEnabled AND (stat.busy = BusyStatus.idle) );
proc.setPosition( isEnabled := isEnabled AND (proc.setPosition.stat.busy = BusyStatus.idle) );
proc.readParameter( isEnabled := isEnabled AND (stat.busy = BusyStatus.idle) );
proc.readBoolParameter( isEnabled := isEnabled AND (stat.busy = BusyStatus.idle) );
proc.writeParameter( isEnabled := isEnabled AND (stat.busy = BusyStatus.idle) );
proc.writeBoolParameter( isEnabled := isEnabled AND (stat.busy = BusyStatus.idle) );

          

METHOD _copyFromModel_SM_BaseAxis
  VAR_IN_OUT
    {attribute 'OPC.UA.DA' := '0'}
    model : M_SM_BaseAxis;
  END_VAR
                  THIS^.proc.moveAbsolute._copyFromModel_McMoveAbsoluteProcess( model := model.proc.moveAbsolute );
THIS^.proc.moveRelative._copyFromModel_McMoveRelativeProcess( model := model.proc.moveRelative );
THIS^.proc.moveVelocity._copyFromModel_McMoveVelocityProcess( model := model.proc.moveVelocity );
THIS^.proc.reset._copyFromModel_McProcess( model := model.proc.reset );
THIS^.proc.stop._copyFromModel_McProcess( model := model.proc.stop );
THIS^.proc.stopParametrized._copyFromModel_McStopProcess( model := model.proc.stopParametrized );
THIS^.proc.power._copyFromModel_McPowerProcess( model := model.proc.power );
THIS^.proc.home._copyFromModel_McProcess( model := model.proc.home );
THIS^.proc.initialize._copyFromModel_Process( model := model.proc.initialize );
THIS^.proc.setPosition._copyFromModel_McSetPositionProcess( model := model.proc.setPosition );
THIS^.proc.readParameter._copyFromModel_McReadParameter( model := model.proc.readParameter );
THIS^.proc.readBoolParameter._copyFromModel_McReadBoolParameter( model := model.proc.readBoolParameter );
THIS^.proc.writeParameter._copyFromModel_McWriteParameter( model := model.proc.writeParameter );
THIS^.proc.writeBoolParameter._copyFromModel_McWriteBoolParameter( model := model.proc.writeBoolParameter );

                
END_METHOD

METHOD _copyToModel_SM_BaseAxis
  VAR_IN_OUT
    {attribute 'OPC.UA.DA' := '0'}
    model : M_SM_BaseAxis;
  END_VAR
                  model.isGearingSupported := THIS^.isGearingSupported;
model.actualStatus := THIS^.actualStatus;
model.isJogEnabled := THIS^.isJogEnabled;
model.errorId := THIS^.errorId;
model.posLimitSwitch := THIS^.posLimitSwitch;
model.negLimitSwitch := THIS^.negLimitSwitch;
model.stat := THIS^.stat;
THIS^.proc.moveAbsolute._copyToModel_McMoveAbsoluteProcess( model := model.proc.moveAbsolute );
THIS^.proc.moveRelative._copyToModel_McMoveRelativeProcess( model := model.proc.moveRelative );
THIS^.proc.moveVelocity._copyToModel_McMoveVelocityProcess( model := model.proc.moveVelocity );
THIS^.proc.reset._copyToModel_McProcess( model := model.proc.reset );
THIS^.proc.stop._copyToModel_McProcess( model := model.proc.stop );
THIS^.proc.stopParametrized._copyToModel_McStopProcess( model := model.proc.stopParametrized );
THIS^.proc.power._copyToModel_McPowerProcess( model := model.proc.power );
THIS^.proc.home._copyToModel_McProcess( model := model.proc.home );
THIS^.proc.initialize._copyToModel_Process( model := model.proc.initialize );
THIS^.proc.setPosition._copyToModel_McSetPositionProcess( model := model.proc.setPosition );
THIS^.proc.readParameter._copyToModel_McReadParameter( model := model.proc.readParameter );
THIS^.proc.readBoolParameter._copyToModel_McReadBoolParameter( model := model.proc.readBoolParameter );
THIS^.proc.writeParameter._copyToModel_McWriteParameter( model := model.proc.writeParameter );
THIS^.proc.writeBoolParameter._copyToModel_McWriteBoolParameter( model := model.proc.writeBoolParameter );

                
END_METHOD
END_FUNCTION_BLOCK

FUNCTION_BLOCK SM_AngularAxis EXTENDS BaseAxis
  VAR_OUTPUT
    {attribute 'OPC.UA.DA' := '1'}
    {attribute 'OPC.UA.DA.Access' := '1'}
    actPos : AngularPosition;  (* Actual position of the axis *)
    {attribute 'OPC.UA.DA' := '1'}
    {attribute 'OPC.UA.DA.Access' := '1'}
    actVel : AngularVelocity;  (* Actual velocity of the axis *)
    {attribute 'OPC.UA.DA' := '1'}
    {attribute 'OPC.UA.DA.Access' := '1'}
    setPos : AngularPosition;  (* Setpoint position of the axis *)
    {attribute 'OPC.UA.DA' := '1'}
    {attribute 'OPC.UA.DA.Access' := '1'}
    setVel : AngularVelocity;  (* Setpoint velocity of the axis *)
    {attribute 'OPC.UA.DA' := '1'}
    {attribute 'OPC.UA.DA.Access' := '1'}
    targetPos : AngularPosition;  (* Target position of the axis *)
  END_VAR

            SUPER^();

          

METHOD _copyFromModel_SM_AngularAxis
  VAR_IN_OUT
    {attribute 'OPC.UA.DA' := '0'}
    model : M_SM_AngularAxis;
  END_VAR
                  SUPER^._copyFromModel_BaseAxis( model := model );

                
END_METHOD

METHOD _copyToModel_SM_AngularAxis
  VAR_IN_OUT
    {attribute 'OPC.UA.DA' := '0'}
    model : M_SM_AngularAxis;
  END_VAR
                  model.actPos := THIS^.actPos;
model.actVel := THIS^.actVel;
model.setPos := THIS^.setPos;
model.setVel := THIS^.setVel;
model.targetPos := THIS^.targetPos;
SUPER^._copyToModel_BaseAxis( model := model );

                
END_METHOD
END_FUNCTION_BLOCK

FUNCTION_BLOCK SM_LinearAxis EXTENDS BaseAxis
  VAR_OUTPUT
    {attribute 'OPC.UA.DA' := '1'}
    {attribute 'OPC.UA.DA.Access' := '1'}
    actPos : LinearPosition;  (* Actual position of the axis *)
    {attribute 'OPC.UA.DA' := '1'}
    {attribute 'OPC.UA.DA.Access' := '1'}
    actVel : LinearVelocity;  (* Actual velocity of the axis *)
    {attribute 'OPC.UA.DA' := '1'}
    {attribute 'OPC.UA.DA.Access' := '1'}
    setPos : LinearPosition;  (* Setpoint position of the axis *)
    {attribute 'OPC.UA.DA' := '1'}
    {attribute 'OPC.UA.DA.Access' := '1'}
    setVel : LinearVelocity;  (* Setpoint velocity of the axis *)
    {attribute 'OPC.UA.DA' := '1'}
    {attribute 'OPC.UA.DA.Access' := '1'}
    targetPos : LinearPosition;  (* Target position of the axis *)
  END_VAR

            SUPER^();

          

METHOD _copyFromModel_SM_LinearAxis
  VAR_IN_OUT
    {attribute 'OPC.UA.DA' := '0'}
    model : M_SM_LinearAxis;
  END_VAR
                  SUPER^._copyFromModel_BaseAxis( model := model );

                
END_METHOD

METHOD _copyToModel_SM_LinearAxis
  VAR_IN_OUT
    {attribute 'OPC.UA.DA' := '0'}
    model : M_SM_LinearAxis;
  END_VAR
                  model.actPos := THIS^.actPos;
model.actVel := THIS^.actVel;
model.setPos := THIS^.setPos;
model.setVel := THIS^.setVel;
model.targetPos := THIS^.targetPos;
SUPER^._copyToModel_BaseAxis( model := model );

                
END_METHOD
END_FUNCTION_BLOCK

FUNCTION_BLOCK SM_MTS50Axis EXTENDS LinearAxis

            SUPER^();

          

METHOD _copyFromModel_SM_MTS50Axis
  VAR_IN_OUT
    {attribute 'OPC.UA.DA' := '0'}
    model : M_SM_MTS50Axis;
  END_VAR
                  SUPER^._copyFromModel_LinearAxis( model := model );

                
END_METHOD

METHOD _copyToModel_SM_MTS50Axis
  VAR_IN_OUT
    {attribute 'OPC.UA.DA' := '0'}
    model : M_SM_MTS50Axis;
  END_VAR
                  SUPER^._copyToModel_LinearAxis( model := model );

                
END_METHOD
END_FUNCTION_BLOCK

FUNCTION_BLOCK SM_SSIEncoder
  VAR_INPUT
    {attribute 'OPC.UA.DA' := '0'}
    counterValue AT %I* : UDINT;  (* Counter value *)
    {attribute 'OPC.UA.DA' := '0'}
    status AT %I* : UINT;  (* Status *)
  END_VAR
  VAR_OUTPUT
    {attribute 'OPC.UA.DA' := '1'}
    {attribute 'OPC.UA.DA.Access' := '1'}
    actualStatus : STRING(50);  (* Current status description *)
    {attribute 'OPC.UA.DA' := '1'}
    {attribute 'OPC.UA.DA.Access' := '1'}
    dataError AT %I* : BOOL;  (* Data error *)
    {attribute 'OPC.UA.DA' := '1'}
    {attribute 'OPC.UA.DA.Access' := '1'}
    frameError AT %I* : BOOL;  (* Frame error *)
    {attribute 'OPC.UA.DA' := '1'}
    {attribute 'OPC.UA.DA.Access' := '1'}
    powerFailure AT %I* : BOOL;  (* Power failure *)
    {attribute 'OPC.UA.DA' := '1'}
    {attribute 'OPC.UA.DA.Access' := '1'}
    syncError AT %I* : BOOL;  (* Sync error *)
    {attribute 'OPC.UA.DA' := '1'}
    stat : SSIEncoderStatuses;  (* Statuses of the state machine *)
  END_VAR

            stat.health := F_HealthStatus(
    superState := TRUE,
    hasWarning := FALSE,
    isGood := NOT(dataError OR (frameError OR (powerFailure OR syncError))));

          

METHOD _copyFromModel_SM_SSIEncoder
  VAR_IN_OUT
    {attribute 'OPC.UA.DA' := '0'}
    model : M_SM_SSIEncoder;
  END_VAR
                  
                
END_METHOD

METHOD _copyToModel_SM_SSIEncoder
  VAR_IN_OUT
    {attribute 'OPC.UA.DA' := '0'}
    model : M_SM_SSIEncoder;
  END_VAR
                  model.actualStatus := THIS^.actualStatus;
model.dataError := THIS^.dataError;
model.frameError := THIS^.frameError;
model.powerFailure := THIS^.powerFailure;
model.syncError := THIS^.syncError;
model.stat := THIS^.stat;

                
END_METHOD
END_FUNCTION_BLOCK

FUNCTION_BLOCK SM_IncrementalEncoder
  VAR_INPUT
    {attribute 'OPC.UA.DA' := '0'}
    isEnabled : BOOL;  (* Is control enabled? *)
    {attribute 'OPC.UA.DA' := '0'}
    counterValue AT %I* : UDINT;  (* Actual counter value *)
    {attribute 'OPC.UA.DA' := '0'}
    status AT %I* : UINT;  (* Status *)
    {attribute 'OPC.UA.DA' := '0'}
    setCounterValue AT %Q* : UDINT;  (* Counter value to be set *)
    {attribute 'OPC.UA.DA' := '0'}
    setCounter AT %Q* : BOOL;  (* Counter value to be set *)
    {attribute 'OPC.UA.DA' := '0'}
    enableLatchC AT %Q* : BOOL;  (* Enable latch C *)
  END_VAR
  VAR_OUTPUT
    {attribute 'OPC.UA.DA' := '1'}
    {attribute 'OPC.UA.DA.Access' := '1'}
    actualStatus : STRING(50);  (* Current status description *)
    {attribute 'OPC.UA.DA' := '1'}
    {attribute 'OPC.UA.DA.Access' := '1'}
    latchCValid : BOOL;  (* Bit 0: Latch C valid *)
    {attribute 'OPC.UA.DA' := '1'}
    {attribute 'OPC.UA.DA.Access' := '1'}
    latchExternValid : BOOL;  (* Bit 1: Latch extern valid *)
    {attribute 'OPC.UA.DA' := '1'}
    {attribute 'OPC.UA.DA.Access' := '1'}
    setCounterDone : BOOL;  (* Bit 2: Set counter done *)
    {attribute 'OPC.UA.DA' := '1'}
    {attribute 'OPC.UA.DA.Access' := '1'}
    counterUnderflow : BOOL;  (* Bit 3: Counter undeflow *)
    {attribute 'OPC.UA.DA' := '1'}
    {attribute 'OPC.UA.DA.Access' := '1'}
    counterOverflow : BOOL;  (* Bit 4: Counter overflow *)
    {attribute 'OPC.UA.DA' := '1'}
    {attribute 'OPC.UA.DA.Access' := '1'}
    statusOfInputStatus : BOOL;  (* Bit 5: Status of input status *)
    {attribute 'OPC.UA.DA' := '1'}
    {attribute 'OPC.UA.DA.Access' := '1'}
    openCircuit : BOOL;  (* Bit 6: Open circuit *)
    {attribute 'OPC.UA.DA' := '1'}
    {attribute 'OPC.UA.DA.Access' := '1'}
    extrapolationStall : BOOL;  (* Bit 7: Extrapolation stall *)
    {attribute 'OPC.UA.DA' := '1'}
    {attribute 'OPC.UA.DA.Access' := '1'}
    statusOfInputA : BOOL;  (* Bit 8: Status of input A *)
    {attribute 'OPC.UA.DA' := '1'}
    {attribute 'OPC.UA.DA.Access' := '1'}
    statusOfInputB : BOOL;  (* Bit 9: Status of input B *)
    {attribute 'OPC.UA.DA' := '1'}
    {attribute 'OPC.UA.DA.Access' := '1'}
    statusOfInputC : BOOL;  (* Bit 10: Status of input C *)
    {attribute 'OPC.UA.DA' := '1'}
    {attribute 'OPC.UA.DA.Access' := '1'}
    statusOfInputGate : BOOL;  (* Bit 11: Status of input gate *)
    {attribute 'OPC.UA.DA' := '1'}
    {attribute 'OPC.UA.DA.Access' := '1'}
    statusOfExternLatch : BOOL;  (* Bit 12: Status of external latch *)
    {attribute 'OPC.UA.DA' := '1'}
    {attribute 'OPC.UA.DA.Access' := '1'}
    syncError : BOOL;  (* Bit 13: Sync error *)
    {attribute 'OPC.UA.DA' := '1'}
    stat : IncrementalEncoderStatuses;  (* Statuses of the state machine *)
    {attribute 'OPC.UA.DA' := '1'}
    proc : IncrementalEncoderProcesses;  (* Processes of the state machine *)
  END_VAR

            stat.health := F_HealthStatus(
    superState := TRUE,
    hasWarning := FALSE,
    isGood := NOT((NOT(statusOfInputStatus)) OR (openCircuit OR (extrapolationStall OR syncError))));
stat.busy := F_BusyStatus(
    superState := TRUE,
    isBusy := (proc.enableCounterResetC.stat.busy = BusyStatus.busy) OR (proc.disableCounterResetC.stat.busy = BusyStatus.busy));
proc.enableCounterResetC( isEnabled := isEnabled );
proc.disableCounterResetC( isEnabled := isEnabled );

          

METHOD _copyFromModel_SM_IncrementalEncoder
  VAR_IN_OUT
    {attribute 'OPC.UA.DA' := '0'}
    model : M_SM_IncrementalEncoder;
  END_VAR
                  THIS^.proc.enableCounterResetC._copyFromModel_Process( model := model.proc.enableCounterResetC );
THIS^.proc.disableCounterResetC._copyFromModel_Process( model := model.proc.disableCounterResetC );

                
END_METHOD

METHOD _copyToModel_SM_IncrementalEncoder
  VAR_IN_OUT
    {attribute 'OPC.UA.DA' := '0'}
    model : M_SM_IncrementalEncoder;
  END_VAR
                  model.actualStatus := THIS^.actualStatus;
model.latchCValid := THIS^.latchCValid;
model.latchExternValid := THIS^.latchExternValid;
model.setCounterDone := THIS^.setCounterDone;
model.counterUnderflow := THIS^.counterUnderflow;
model.counterOverflow := THIS^.counterOverflow;
model.statusOfInputStatus := THIS^.statusOfInputStatus;
model.openCircuit := THIS^.openCircuit;
model.extrapolationStall := THIS^.extrapolationStall;
model.statusOfInputA := THIS^.statusOfInputA;
model.statusOfInputB := THIS^.statusOfInputB;
model.statusOfInputC := THIS^.statusOfInputC;
model.statusOfInputGate := THIS^.statusOfInputGate;
model.statusOfExternLatch := THIS^.statusOfExternLatch;
model.syncError := THIS^.syncError;
model.stat := THIS^.stat;
THIS^.proc.enableCounterResetC._copyToModel_Process( model := model.proc.enableCounterResetC );
THIS^.proc.disableCounterResetC._copyToModel_Process( model := model.proc.disableCounterResetC );

                
END_METHOD
END_FUNCTION_BLOCK

FUNCTION_BLOCK SM_EtherCatDevice
  VAR_INPUT
    {attribute 'OPC.UA.DA' := '1'}
    {attribute 'OPC.UA.DA.Access' := '1'}
    id : STRING(15);  (* Label according to the electric schemes *)
    {attribute 'OPC.UA.DA' := '1'}
    {attribute 'OPC.UA.DA.Access' := '1'}
    typeId : STRING(15);  (* Manufacturer type, e.g. EL1008 *)
    {attribute 'OPC.UA.DA' := '1'}
    {attribute 'OPC.UA.DA.Access' := '1'}
    wcState AT %I* : BOOL;  (* 0 = Data valid, 1 = Data invalid *)
    {attribute 'OPC.UA.DA' := '1'}
    {attribute 'OPC.UA.DA.Access' := '1'}
    infoData AT %I* : UINT;  (* EtherCAT state *)
  END_VAR
  VAR_OUTPUT
    {attribute 'OPC.UA.DA' := '1'}
    {attribute 'OPC.UA.DA.Access' := '1'}
    actualStatus : STRING(50);  (* Current status description *)
    {attribute 'OPC.UA.DA' := '1'}
    stat : EtherCatDeviceStatuses;  (* Statuses of the state machine *)
  END_VAR

            stat.health := F_HealthStatus(
    superState := TRUE,
    hasWarning := FALSE,
    isGood := (wcState = FALSE) AND (infoData = 8));

          

METHOD _copyFromModel_SM_EtherCatDevice
  VAR_IN_OUT
    {attribute 'OPC.UA.DA' := '0'}
    model : M_SM_EtherCatDevice;
  END_VAR
                  
                
END_METHOD

METHOD _copyToModel_SM_EtherCatDevice
  VAR_IN_OUT
    {attribute 'OPC.UA.DA' := '0'}
    model : M_SM_EtherCatDevice;
  END_VAR
                  model.id := THIS^.id;
model.typeId := THIS^.typeId;
model.wcState := THIS^.wcState;
model.infoData := THIS^.infoData;
model.actualStatus := THIS^.actualStatus;
model.stat := THIS^.stat;

                
END_METHOD
END_FUNCTION_BLOCK

FUNCTION_BLOCK SM_CANopenBus
  VAR_INPUT
    {attribute 'OPC.UA.DA' := '1'}
    {attribute 'OPC.UA.DA.Access' := '1'}
    error AT %I* : USINT;  (* Number of boxes with BoxState unequal to 0 *)
    {attribute 'OPC.UA.DA' := '1'}
    {attribute 'OPC.UA.DA.Access' := '1'}
    canState AT %I* : UINT;  (* CAN state (See system manager for bit interpretation *)
    {attribute 'OPC.UA.DA' := '1'}
    {attribute 'OPC.UA.DA.Access' := '1'}
    rxErrorCounter AT %I* : USINT;  (* RxError-counter of the CAN controller *)
    {attribute 'OPC.UA.DA' := '1'}
    {attribute 'OPC.UA.DA.Access' := '1'}
    txErrorCounter AT %I* : USINT;  (* TxError-counter of the CAN controller *)
  END_VAR
  VAR_OUTPUT
    {attribute 'OPC.UA.DA' := '1'}
    {attribute 'OPC.UA.DA.Access' := '1'}
    actualStatus : STRING(50);  (* Current status description *)
    {attribute 'OPC.UA.DA' := '1'}
    stat : CANopenBusStatuses;  (* Statuses of the state machine *)
  END_VAR

            stat.health := F_HealthStatus(
    superState := TRUE,
    hasWarning := FALSE,
    isGood := error = 0);

          

METHOD _copyFromModel_SM_CANopenBus
  VAR_IN_OUT
    {attribute 'OPC.UA.DA' := '0'}
    model : M_SM_CANopenBus;
  END_VAR
                  
                
END_METHOD

METHOD _copyToModel_SM_CANopenBus
  VAR_IN_OUT
    {attribute 'OPC.UA.DA' := '0'}
    model : M_SM_CANopenBus;
  END_VAR
                  model.error := THIS^.error;
model.canState := THIS^.canState;
model.rxErrorCounter := THIS^.rxErrorCounter;
model.txErrorCounter := THIS^.txErrorCounter;
model.actualStatus := THIS^.actualStatus;
model.stat := THIS^.stat;

                
END_METHOD
END_FUNCTION_BLOCK

FUNCTION_BLOCK SM_CurrentMeasurement
  VAR_INPUT
    {attribute 'OPC.UA.DA' := '0'}
    microAmpsValue AT %I* : DINT;  (* Measured current in microamps *)
    {attribute 'OPC.UA.DA' := '0'}
    error AT %I* : BOOL;  (* Error *)
  END_VAR
  VAR_OUTPUT
    {attribute 'OPC.UA.DA' := '1'}
    {attribute 'OPC.UA.DA.Access' := '1'}
    actualStatus : STRING(50);  (* Current status description *)
    {attribute 'OPC.UA.DA' := '1'}
    {attribute 'OPC.UA.DA.Access' := '1'}
    current : Current;  (* The measured current *)
    {attribute 'OPC.UA.DA' := '1'}
    stat : CurrentMeasurementStatuses;  (* Statuses of the state machine *)
  END_VAR

            stat.health := F_HealthStatus(
    superState := TRUE,
    hasWarning := FALSE,
    isGood := NOT(error));

          

METHOD _copyFromModel_SM_CurrentMeasurement
  VAR_IN_OUT
    {attribute 'OPC.UA.DA' := '0'}
    model : M_SM_CurrentMeasurement;
  END_VAR
                  
                
END_METHOD

METHOD _copyToModel_SM_CurrentMeasurement
  VAR_IN_OUT
    {attribute 'OPC.UA.DA' := '0'}
    model : M_SM_CurrentMeasurement;
  END_VAR
                  model.actualStatus := THIS^.actualStatus;
model.current := THIS^.current;
model.stat := THIS^.stat;

                
END_METHOD
END_FUNCTION_BLOCK

FUNCTION_BLOCK SM_VoltageMeasurement
  VAR_INPUT
    {attribute 'OPC.UA.DA' := '0'}
    rawValue AT %I* : INT;  (* Measured raw value *)
    {attribute 'OPC.UA.DA' := '0'}
    error AT %I* : BOOL;  (* Error *)
    {attribute 'OPC.UA.DA' := '0'}
    conversionFactor : LREAL := 0.00030517578125;  (* rawValue * conversionFactor = volt.value *)
  END_VAR
  VAR_OUTPUT
    {attribute 'OPC.UA.DA' := '1'}
    {attribute 'OPC.UA.DA.Access' := '1'}
    actualStatus : STRING(50);  (* Current status description *)
    {attribute 'OPC.UA.DA' := '1'}
    {attribute 'OPC.UA.DA.Access' := '1'}
    actual : Voltage;  (* Actual value *)
    {attribute 'OPC.UA.DA' := '1'}
    {attribute 'OPC.UA.DA.Access' := '1'}
    average : Voltage;  (* Moving average value *)
    {attribute 'OPC.UA.DA' := '1'}
    {attribute 'OPC.UA.DA.Access' := '1'}
    underrange AT %I* : BOOL;  (* Underrange *)
    {attribute 'OPC.UA.DA' := '1'}
    {attribute 'OPC.UA.DA.Access' := '1'}
    overrange AT %I* : BOOL;  (* Overrange *)
    {attribute 'OPC.UA.DA' := '1'}
    stat : VoltageMeasurementStatuses;  (* Statuses of the state machine *)
  END_VAR
  VAR_IN_OUT
    {attribute 'OPC.UA.DA' := '0'}
    config : MeasurementConfig;  (* Reference to the config (alarms in volts) *)
  END_VAR

            stat.enabled := F_EnabledStatus(
    superState := TRUE,
    isEnabled := config.enabled);
stat.health := F_HealthStatus(
    superState := stat.enabled = EnabledStatus.enabled,
    isGood := NOT(error OR (underrange OR (overrange OR ((stat.alarm = HiHiLoLoAlarmStatus.hiHi) OR (stat.alarm = HiHiLoLoAlarmStatus.loLo))))),
    hasWarning := (stat.alarm = HiHiLoLoAlarmStatus.hi) OR (stat.alarm = HiHiLoLoAlarmStatus.lo));
stat.alarm := F_HiHiLoLoAlarmStatus(
    superState := stat.enabled = EnabledStatus.enabled,
    config := config.alarms,
    value := average.volt.value);

          

METHOD _copyFromModel_SM_VoltageMeasurement
  VAR_IN_OUT
    {attribute 'OPC.UA.DA' := '0'}
    model : M_SM_VoltageMeasurement;
  END_VAR
                  
                
END_METHOD

METHOD _copyToModel_SM_VoltageMeasurement
  VAR_IN_OUT
    {attribute 'OPC.UA.DA' := '0'}
    model : M_SM_VoltageMeasurement;
  END_VAR
                  model.actualStatus := THIS^.actualStatus;
model.actual := THIS^.actual;
model.average := THIS^.average;
model.underrange := THIS^.underrange;
model.overrange := THIS^.overrange;
model.stat := THIS^.stat;

                
END_METHOD
END_FUNCTION_BLOCK

FUNCTION_BLOCK SM_SimpleTemperature
  VAR_OUTPUT
    {attribute 'OPC.UA.DA' := '1'}
    {attribute 'OPC.UA.DA.Access' := '1'}
    actualStatus : STRING(50);  (* Current status description *)
    {attribute 'OPC.UA.DA' := '1'}
    {attribute 'OPC.UA.DA.Access' := '1'}
    value : LREAL;  (* Actual value *)
    {attribute 'OPC.UA.DA' := '1'}
    {attribute 'OPC.UA.DA.Access' := '1'}
    error AT %I* : BOOL;  (* error *)
    {attribute 'OPC.UA.DA' := '1'}
    {attribute 'OPC.UA.DA.Access' := '1'}
    underrange AT %I* : BOOL;  (* Underrange *)
    {attribute 'OPC.UA.DA' := '1'}
    {attribute 'OPC.UA.DA.Access' := '1'}
    overrange AT %I* : BOOL;  (* Overrange *)
    {attribute 'OPC.UA.DA' := '1'}
    stat : SimpleTemperatureStatuses;  (* Statuses of the state machine *)
  END_VAR
  VAR_IN_OUT
    {attribute 'OPC.UA.DA' := '0'}
    config : MeasurementConfig;  (* Reference to the config (alarms in degrees celsius) *)
  END_VAR

            stat.enabled := F_EnabledStatus(
    superState := TRUE,
    isEnabled := config.enabled);
stat.health := F_HealthStatus(
    superState := stat.enabled = EnabledStatus.enabled,
    isGood := NOT(error OR (underrange OR (overrange OR ((stat.alarm = HiHiLoLoAlarmStatus.hiHi) OR (stat.alarm = HiHiLoLoAlarmStatus.loLo))))),
    hasWarning := (stat.alarm = HiHiLoLoAlarmStatus.hi) OR (stat.alarm = HiHiLoLoAlarmStatus.lo));
stat.alarm := F_HiHiLoLoAlarmStatus(
    superState := stat.enabled = EnabledStatus.enabled,
    config := config.alarms,
    value := value);

          

METHOD _copyFromModel_SM_SimpleTemperature
  VAR_IN_OUT
    {attribute 'OPC.UA.DA' := '0'}
    model : M_SM_SimpleTemperature;
  END_VAR
                  
                
END_METHOD

METHOD _copyToModel_SM_SimpleTemperature
  VAR_IN_OUT
    {attribute 'OPC.UA.DA' := '0'}
    model : M_SM_SimpleTemperature;
  END_VAR
                  model.actualStatus := THIS^.actualStatus;
model.value := THIS^.value;
model.error := THIS^.error;
model.underrange := THIS^.underrange;
model.overrange := THIS^.overrange;
model.stat := THIS^.stat;

                
END_METHOD
END_FUNCTION_BLOCK

FUNCTION_BLOCK SM_TemperatureMeasurement
  VAR_INPUT
    {attribute 'OPC.UA.DA' := '0'}
    rawValue AT %I* : INT;  (* Measured raw value *)
    {attribute 'OPC.UA.DA' := '0'}
    error AT %I* : BOOL;  (* Error *)
    {attribute 'OPC.UA.DA' := '0'}
    conversionFactor : LREAL := 0.01;  (* rawValue * conversionFactor = temperature.degrees.value *)
  END_VAR
  VAR_OUTPUT
    {attribute 'OPC.UA.DA' := '1'}
    {attribute 'OPC.UA.DA.Access' := '1'}
    actualStatus : STRING(50);  (* Current status description *)
    {attribute 'OPC.UA.DA' := '1'}
    {attribute 'OPC.UA.DA.Access' := '1'}
    actual : Temperature;  (* Actual value *)
    {attribute 'OPC.UA.DA' := '1'}
    {attribute 'OPC.UA.DA.Access' := '1'}
    average : Temperature;  (* Moving average value *)
    {attribute 'OPC.UA.DA' := '1'}
    {attribute 'OPC.UA.DA.Access' := '1'}
    underrange AT %I* : BOOL;  (* Underrange *)
    {attribute 'OPC.UA.DA' := '1'}
    {attribute 'OPC.UA.DA.Access' := '1'}
    overrange AT %I* : BOOL;  (* Overrange *)
    {attribute 'OPC.UA.DA' := '1'}
    stat : TemperatureMeasurementStatuses;  (* Statuses of the state machine *)
  END_VAR
  VAR_IN_OUT
    {attribute 'OPC.UA.DA' := '0'}
    config : MeasurementConfig;  (* Reference to the config (alarms in degrees celsius) *)
  END_VAR

            stat.enabled := F_EnabledStatus(
    superState := TRUE,
    isEnabled := config.enabled);
stat.health := F_HealthStatus(
    superState := stat.enabled = EnabledStatus.enabled,
    isGood := NOT(error OR (underrange OR (overrange OR ((stat.alarm = HiHiLoLoAlarmStatus.hiHi) OR (stat.alarm = HiHiLoLoAlarmStatus.loLo))))),
    hasWarning := (stat.alarm = HiHiLoLoAlarmStatus.hi) OR (stat.alarm = HiHiLoLoAlarmStatus.lo));
stat.alarm := F_HiHiLoLoAlarmStatus(
    superState := stat.enabled = EnabledStatus.enabled,
    config := config.alarms,
    value := average.celsius.value);

          

METHOD _copyFromModel_SM_TemperatureMeasurement
  VAR_IN_OUT
    {attribute 'OPC.UA.DA' := '0'}
    model : M_SM_TemperatureMeasurement;
  END_VAR
                  
                
END_METHOD

METHOD _copyToModel_SM_TemperatureMeasurement
  VAR_IN_OUT
    {attribute 'OPC.UA.DA' := '0'}
    model : M_SM_TemperatureMeasurement;
  END_VAR
                  model.actualStatus := THIS^.actualStatus;
model.actual := THIS^.actual;
model.average := THIS^.average;
model.underrange := THIS^.underrange;
model.overrange := THIS^.overrange;
model.stat := THIS^.stat;

                
END_METHOD
END_FUNCTION_BLOCK

FUNCTION_BLOCK SM_PressureMeasurement
  VAR_INPUT
    {attribute 'OPC.UA.DA' := '0'}
    rawValue AT %I* : INT;  (* Measured raw value *)
    {attribute 'OPC.UA.DA' := '0'}
    error AT %I* : BOOL;  (* Error *)
    {attribute 'OPC.UA.DA' := '0'}
    conversionFactor : LREAL := 1.0;  (* rawValue * conversionFactor = bar.value *)
  END_VAR
  VAR_OUTPUT
    {attribute 'OPC.UA.DA' := '1'}
    {attribute 'OPC.UA.DA.Access' := '1'}
    actualStatus : STRING(50);  (* Current status description *)
    {attribute 'OPC.UA.DA' := '1'}
    {attribute 'OPC.UA.DA.Access' := '1'}
    actual : Pressure;  (* Actual value *)
    {attribute 'OPC.UA.DA' := '1'}
    {attribute 'OPC.UA.DA.Access' := '1'}
    average : Pressure;  (* Moving average value *)
    {attribute 'OPC.UA.DA' := '1'}
    {attribute 'OPC.UA.DA.Access' := '1'}
    underrange AT %I* : BOOL;  (* Underrange *)
    {attribute 'OPC.UA.DA' := '1'}
    {attribute 'OPC.UA.DA.Access' := '1'}
    overrange AT %I* : BOOL;  (* Overrange *)
    {attribute 'OPC.UA.DA' := '1'}
    stat : PressureMeasurementStatuses;  (* Statuses of the state machine *)
  END_VAR
  VAR_IN_OUT
    {attribute 'OPC.UA.DA' := '0'}
    config : MeasurementConfig;  (* Reference to the config (alarms in bar) *)
  END_VAR

            stat.enabled := F_EnabledStatus(
    superState := TRUE,
    isEnabled := config.enabled);
stat.health := F_HealthStatus(
    superState := stat.enabled = EnabledStatus.enabled,
    isGood := NOT(error OR (underrange OR (overrange OR ((stat.alarm = HiHiLoLoAlarmStatus.hiHi) OR (stat.alarm = HiHiLoLoAlarmStatus.loLo))))),
    hasWarning := (stat.alarm = HiHiLoLoAlarmStatus.hi) OR (stat.alarm = HiHiLoLoAlarmStatus.lo));
stat.alarm := F_HiHiLoLoAlarmStatus(
    superState := stat.enabled = EnabledStatus.enabled,
    config := config.alarms,
    value := average.bar.value);

          

METHOD _copyFromModel_SM_PressureMeasurement
  VAR_IN_OUT
    {attribute 'OPC.UA.DA' := '0'}
    model : M_SM_PressureMeasurement;
  END_VAR
                  
                
END_METHOD

METHOD _copyToModel_SM_PressureMeasurement
  VAR_IN_OUT
    {attribute 'OPC.UA.DA' := '0'}
    model : M_SM_PressureMeasurement;
  END_VAR
                  model.actualStatus := THIS^.actualStatus;
model.actual := THIS^.actual;
model.average := THIS^.average;
model.underrange := THIS^.underrange;
model.overrange := THIS^.overrange;
model.stat := THIS^.stat;

                
END_METHOD
END_FUNCTION_BLOCK

FUNCTION_BLOCK SM_FrequencyMeasurement
  VAR_INPUT
    {attribute 'OPC.UA.DA' := '0'}
    rawValue AT %I* : INT;  (* Measured raw value *)
    {attribute 'OPC.UA.DA' := '0'}
    error AT %I* : BOOL;  (* Error *)
    {attribute 'OPC.UA.DA' := '0'}
    conversionFactor : LREAL := 1.0;  (* rawValue * conversionFactor = hertz.value *)
  END_VAR
  VAR_OUTPUT
    {attribute 'OPC.UA.DA' := '1'}
    {attribute 'OPC.UA.DA.Access' := '1'}
    actualStatus : STRING(50);  (* Current status description *)
    {attribute 'OPC.UA.DA' := '1'}
    {attribute 'OPC.UA.DA.Access' := '1'}
    actual : Frequency;  (* Actual value *)
    {attribute 'OPC.UA.DA' := '1'}
    {attribute 'OPC.UA.DA.Access' := '1'}
    average : Frequency;  (* Moving average value *)
    {attribute 'OPC.UA.DA' := '1'}
    {attribute 'OPC.UA.DA.Access' := '1'}
    underrange AT %I* : BOOL;  (* Underrange *)
    {attribute 'OPC.UA.DA' := '1'}
    {attribute 'OPC.UA.DA.Access' := '1'}
    overrange AT %I* : BOOL;  (* Overrange *)
    {attribute 'OPC.UA.DA' := '1'}
    stat : FrequencyMeasurementStatuses;  (* Statuses of the state machine *)
  END_VAR
  VAR_IN_OUT
    {attribute 'OPC.UA.DA' := '0'}
    config : MeasurementConfig;  (* Reference to the config (alarms in hertz) *)
  END_VAR

            stat.enabled := F_EnabledStatus(
    superState := TRUE,
    isEnabled := config.enabled);
stat.health := F_HealthStatus(
    superState := stat.enabled = EnabledStatus.enabled,
    isGood := NOT(error OR (underrange OR (overrange OR ((stat.alarm = HiHiLoLoAlarmStatus.hiHi) OR (stat.alarm = HiHiLoLoAlarmStatus.loLo))))),
    hasWarning := (stat.alarm = HiHiLoLoAlarmStatus.hi) OR (stat.alarm = HiHiLoLoAlarmStatus.lo));
stat.alarm := F_HiHiLoLoAlarmStatus(
    superState := stat.enabled = EnabledStatus.enabled,
    config := config.alarms,
    value := average.hertz.value);

          

METHOD _copyFromModel_SM_FrequencyMeasurement
  VAR_IN_OUT
    {attribute 'OPC.UA.DA' := '0'}
    model : M_SM_FrequencyMeasurement;
  END_VAR
                  
                
END_METHOD

METHOD _copyToModel_SM_FrequencyMeasurement
  VAR_IN_OUT
    {attribute 'OPC.UA.DA' := '0'}
    model : M_SM_FrequencyMeasurement;
  END_VAR
                  model.actualStatus := THIS^.actualStatus;
model.actual := THIS^.actual;
model.average := THIS^.average;
model.underrange := THIS^.underrange;
model.overrange := THIS^.overrange;
model.stat := THIS^.stat;

                
END_METHOD
END_FUNCTION_BLOCK

FUNCTION_BLOCK SM_GForceMeasurement
  VAR_INPUT
    {attribute 'OPC.UA.DA' := '0'}
    milliGValue AT %I* : INT;  (* Measured raw milliG value (linked to I/O module) *)
    {attribute 'OPC.UA.DA' := '0'}
    error AT %I* : BOOL;  (* Error *)
  END_VAR
  VAR_OUTPUT
    {attribute 'OPC.UA.DA' := '1'}
    {attribute 'OPC.UA.DA.Access' := '1'}
    actualStatus : STRING(50);  (* Current status description *)
    {attribute 'OPC.UA.DA' := '1'}
    {attribute 'OPC.UA.DA.Access' := '1'}
    actual : GForce;  (* Actual value *)
    {attribute 'OPC.UA.DA' := '1'}
    {attribute 'OPC.UA.DA.Access' := '1'}
    average : GForce;  (* Moving average value *)
    {attribute 'OPC.UA.DA' := '1'}
    stat : GForceMeasurementStatuses;  (* Statuses of the state machine *)
  END_VAR

            stat.health := F_HealthStatus(
    superState := TRUE,
    hasWarning := FALSE,
    isGood := NOT(error));

          

METHOD _copyFromModel_SM_GForceMeasurement
  VAR_IN_OUT
    {attribute 'OPC.UA.DA' := '0'}
    model : M_SM_GForceMeasurement;
  END_VAR
                  
                
END_METHOD

METHOD _copyToModel_SM_GForceMeasurement
  VAR_IN_OUT
    {attribute 'OPC.UA.DA' := '0'}
    model : M_SM_GForceMeasurement;
  END_VAR
                  model.actualStatus := THIS^.actualStatus;
model.actual := THIS^.actual;
model.average := THIS^.average;
model.stat := THIS^.stat;

                
END_METHOD
END_FUNCTION_BLOCK

FUNCTION_BLOCK SM_RelativeHumidityMeasurement
  VAR_INPUT
    {attribute 'OPC.UA.DA' := '0'}
    rawValue AT %I* : INT;  (* Measured raw value *)
    {attribute 'OPC.UA.DA' := '0'}
    error AT %I* : BOOL;  (* Error *)
    {attribute 'OPC.UA.DA' := '0'}
    conversionFactor : LREAL := 3.051850947599719E-05;  (* rawValue * conversionFactor = fraction.value *)
  END_VAR
  VAR_OUTPUT
    {attribute 'OPC.UA.DA' := '1'}
    {attribute 'OPC.UA.DA.Access' := '1'}
    actualStatus : STRING(50);  (* Current status description *)
    {attribute 'OPC.UA.DA' := '1'}
    {attribute 'OPC.UA.DA.Access' := '1'}
    actual : Fraction;  (* Actual value *)
    {attribute 'OPC.UA.DA' := '1'}
    {attribute 'OPC.UA.DA.Access' := '1'}
    average : Fraction;  (* Moving average value *)
    {attribute 'OPC.UA.DA' := '1'}
    {attribute 'OPC.UA.DA.Access' := '1'}
    underrange AT %I* : BOOL;  (* Underrange *)
    {attribute 'OPC.UA.DA' := '1'}
    {attribute 'OPC.UA.DA.Access' := '1'}
    overrange AT %I* : BOOL;  (* Overrange *)
    {attribute 'OPC.UA.DA' := '1'}
    stat : RelativeHumidityMeasurementStatuses;  (* Statuses of the state machine *)
  END_VAR
  VAR_IN_OUT
    {attribute 'OPC.UA.DA' := '0'}
    config : MeasurementConfig;  (* Reference to the config (alarms in percent) *)
  END_VAR

            stat.enabled := F_EnabledStatus(
    superState := TRUE,
    isEnabled := config.enabled);
stat.health := F_HealthStatus(
    superState := stat.enabled = EnabledStatus.enabled,
    isGood := NOT((error AND (underrange OR overrange)) OR ((stat.alarm = HiHiLoLoAlarmStatus.hiHi) OR (stat.alarm = HiHiLoLoAlarmStatus.loLo))),
    hasWarning := (stat.alarm = HiHiLoLoAlarmStatus.hi) OR (stat.alarm = HiHiLoLoAlarmStatus.lo));
stat.alarm := F_HiHiLoLoAlarmStatus(
    superState := stat.enabled = EnabledStatus.enabled,
    config := config.alarms,
    value := average.percent.value);

          

METHOD _copyFromModel_SM_RelativeHumidityMeasurement
  VAR_IN_OUT
    {attribute 'OPC.UA.DA' := '0'}
    model : M_SM_RelativeHumidityMeasurement;
  END_VAR
                  
                
END_METHOD

METHOD _copyToModel_SM_RelativeHumidityMeasurement
  VAR_IN_OUT
    {attribute 'OPC.UA.DA' := '0'}
    model : M_SM_RelativeHumidityMeasurement;
  END_VAR
                  model.actualStatus := THIS^.actualStatus;
model.actual := THIS^.actual;
model.average := THIS^.average;
model.underrange := THIS^.underrange;
model.overrange := THIS^.overrange;
model.stat := THIS^.stat;

                
END_METHOD
END_FUNCTION_BLOCK

FUNCTION_BLOCK SM_ForceMeasurement
  VAR_INPUT
    {attribute 'OPC.UA.DA' := '0'}
    rawValue AT %I* : DINT;  (* Measured raw value *)
    {attribute 'OPC.UA.DA' := '0'}
    error AT %I* : BOOL;  (* Error *)
    {attribute 'OPC.UA.DA' := '0'}
    underrange AT %I* : BOOL;  (* Underrange *)
    {attribute 'OPC.UA.DA' := '0'}
    overrange AT %I* : BOOL;  (* Overrange *)
    {attribute 'OPC.UA.DA' := '0'}
    conversionFactor : LREAL := 1.0;  (* rawValue * conversionFactor = newton.value *)
  END_VAR
  VAR_OUTPUT
    {attribute 'OPC.UA.DA' := '1'}
    {attribute 'OPC.UA.DA.Access' := '1'}
    actualStatus : STRING(50);  (* Current status description *)
    {attribute 'OPC.UA.DA' := '1'}
    {attribute 'OPC.UA.DA.Access' := '1'}
    actual : Force;  (* Actual value *)
    {attribute 'OPC.UA.DA' := '1'}
    {attribute 'OPC.UA.DA.Access' := '1'}
    average : Force;  (* Moving average value *)
    {attribute 'OPC.UA.DA' := '1'}
    stat : ForceMeasurementStatuses;  (* Statuses of the state machine *)
  END_VAR
  VAR_IN_OUT
    {attribute 'OPC.UA.DA' := '0'}
    config : MeasurementConfig;  (* Reference to the config (alarms in Newton) *)
  END_VAR

            stat.enabled := F_EnabledStatus(
    superState := TRUE,
    isEnabled := config.enabled);
stat.health := F_HealthStatus(
    superState := stat.enabled = EnabledStatus.enabled,
    isGood := NOT(error OR (underrange OR (overrange OR ((stat.alarm = HiHiLoLoAlarmStatus.hiHi) OR (stat.alarm = HiHiLoLoAlarmStatus.loLo))))),
    hasWarning := (stat.alarm = HiHiLoLoAlarmStatus.hi) OR (stat.alarm = HiHiLoLoAlarmStatus.lo));
stat.alarm := F_HiHiLoLoAlarmStatus(
    superState := stat.enabled = EnabledStatus.enabled,
    config := config.alarms,
    value := average.newton.value);

          

METHOD _copyFromModel_SM_ForceMeasurement
  VAR_IN_OUT
    {attribute 'OPC.UA.DA' := '0'}
    model : M_SM_ForceMeasurement;
  END_VAR
                  
                
END_METHOD

METHOD _copyToModel_SM_ForceMeasurement
  VAR_IN_OUT
    {attribute 'OPC.UA.DA' := '0'}
    model : M_SM_ForceMeasurement;
  END_VAR
                  model.actualStatus := THIS^.actualStatus;
model.actual := THIS^.actual;
model.average := THIS^.average;
model.stat := THIS^.stat;

                
END_METHOD
END_FUNCTION_BLOCK

FUNCTION_BLOCK SM_LinearPositionMeasurement16
  VAR_INPUT
    {attribute 'OPC.UA.DA' := '0'}
    rawValue AT %I* : INT;  (* Measured raw value *)
    {attribute 'OPC.UA.DA' := '0'}
    error AT %I* : BOOL;  (* Error *)
    {attribute 'OPC.UA.DA' := '0'}
    underrange AT %I* : BOOL;  (* Underrange *)
    {attribute 'OPC.UA.DA' := '0'}
    overrange AT %I* : BOOL;  (* Overrange *)
    {attribute 'OPC.UA.DA' := '0'}
    conversionFactor : LREAL := 3.051850947599719E-05;  (* rawValue * conversionFactor = millimeters.value *)
  END_VAR
  VAR_OUTPUT
    {attribute 'OPC.UA.DA' := '1'}
    {attribute 'OPC.UA.DA.Access' := '1'}
    actualStatus : STRING(50);  (* Current status description *)
    {attribute 'OPC.UA.DA' := '1'}
    {attribute 'OPC.UA.DA.Access' := '1'}
    actual : LinearPosition;  (* Actual value *)
    {attribute 'OPC.UA.DA' := '1'}
    {attribute 'OPC.UA.DA.Access' := '1'}
    average : LinearPosition;  (* Moving average value *)
    {attribute 'OPC.UA.DA' := '1'}
    stat : LinearPositionMeasurement16Statuses;  (* Statuses of the state machine *)
  END_VAR
  VAR_IN_OUT
    {attribute 'OPC.UA.DA' := '0'}
    config : MeasurementConfig;  (* Reference to the config (alarms in millimeters) *)
  END_VAR

            stat.enabled := F_EnabledStatus(
    superState := TRUE,
    isEnabled := config.enabled);
stat.health := F_HealthStatus(
    superState := stat.enabled = EnabledStatus.enabled,
    isGood := NOT(error OR (underrange OR (overrange OR ((stat.alarm = HiHiLoLoAlarmStatus.hiHi) OR (stat.alarm = HiHiLoLoAlarmStatus.loLo))))),
    hasWarning := (stat.alarm = HiHiLoLoAlarmStatus.hi) OR (stat.alarm = HiHiLoLoAlarmStatus.lo));
stat.alarm := F_HiHiLoLoAlarmStatus(
    superState := stat.enabled = EnabledStatus.enabled,
    config := config.alarms,
    value := average.millimeters.value);

          

METHOD _copyFromModel_SM_LinearPositionMeasurement16
  VAR_IN_OUT
    {attribute 'OPC.UA.DA' := '0'}
    model : M_SM_LinearPositionMeasurement16;
  END_VAR
                  
                
END_METHOD

METHOD _copyToModel_SM_LinearPositionMeasurement16
  VAR_IN_OUT
    {attribute 'OPC.UA.DA' := '0'}
    model : M_SM_LinearPositionMeasurement16;
  END_VAR
                  model.actualStatus := THIS^.actualStatus;
model.actual := THIS^.actual;
model.average := THIS^.average;
model.stat := THIS^.stat;

                
END_METHOD
END_FUNCTION_BLOCK

FUNCTION_BLOCK SM_LinearPositionMeasurementU32
  VAR_INPUT
    {attribute 'OPC.UA.DA' := '0'}
    rawValue AT %I* : UDINT;  (* Measured raw value *)
    {attribute 'OPC.UA.DA' := '0'}
    error AT %I* : BOOL;  (* Error *)
    {attribute 'OPC.UA.DA' := '0'}
    underrange AT %I* : BOOL;  (* Underrange *)
    {attribute 'OPC.UA.DA' := '0'}
    overrange AT %I* : BOOL;  (* Overrange *)
    {attribute 'OPC.UA.DA' := '0'}
    conversionFactor : LREAL := 4.656612875245797E-10;  (* rawValue * conversionFactor = millimeters.value *)
  END_VAR
  VAR_OUTPUT
    {attribute 'OPC.UA.DA' := '1'}
    {attribute 'OPC.UA.DA.Access' := '1'}
    actualStatus : STRING(50);  (* Current status description *)
    {attribute 'OPC.UA.DA' := '1'}
    {attribute 'OPC.UA.DA.Access' := '1'}
    actual : LinearPosition;  (* Actual value *)
    {attribute 'OPC.UA.DA' := '1'}
    {attribute 'OPC.UA.DA.Access' := '1'}
    average : LinearPosition;  (* Moving average value *)
    {attribute 'OPC.UA.DA' := '1'}
    stat : LinearPositionMeasurementU32Statuses;  (* Statuses of the state machine *)
  END_VAR
  VAR_IN_OUT
    {attribute 'OPC.UA.DA' := '0'}
    config : MeasurementConfig;  (* Reference to the config (alarms in millimeters) *)
  END_VAR

            stat.enabled := F_EnabledStatus(
    superState := TRUE,
    isEnabled := config.enabled);
stat.health := F_HealthStatus(
    superState := stat.enabled = EnabledStatus.enabled,
    isGood := NOT(error OR (underrange OR (overrange OR ((stat.alarm = HiHiLoLoAlarmStatus.hiHi) OR (stat.alarm = HiHiLoLoAlarmStatus.loLo))))),
    hasWarning := (stat.alarm = HiHiLoLoAlarmStatus.hi) OR (stat.alarm = HiHiLoLoAlarmStatus.lo));
stat.alarm := F_HiHiLoLoAlarmStatus(
    superState := stat.enabled = EnabledStatus.enabled,
    config := config.alarms,
    value := average.millimeters.value);

          

METHOD _copyFromModel_SM_LinearPositionMeasurementU32
  VAR_IN_OUT
    {attribute 'OPC.UA.DA' := '0'}
    model : M_SM_LinearPositionMeasurementU32;
  END_VAR
                  
                
END_METHOD

METHOD _copyToModel_SM_LinearPositionMeasurementU32
  VAR_IN_OUT
    {attribute 'OPC.UA.DA' := '0'}
    model : M_SM_LinearPositionMeasurementU32;
  END_VAR
                  model.actualStatus := THIS^.actualStatus;
model.actual := THIS^.actual;
model.average := THIS^.average;
model.stat := THIS^.stat;

                
END_METHOD
END_FUNCTION_BLOCK

FUNCTION_BLOCK SM_SimpleRelay
  VAR_INPUT
    {attribute 'OPC.UA.DA' := '0'}
    isEnabled : BOOL;  (* Is control enabled? *)
  END_VAR
  VAR_OUTPUT
    {attribute 'OPC.UA.DA' := '1'}
    {attribute 'OPC.UA.DA.Access' := '1'}
    actualStatus : STRING(50);  (* Current status description *)
    {attribute 'OPC.UA.DA' := '1'}
    {attribute 'OPC.UA.DA.Access' := '1'}
    digitalOutput AT %Q* : BOOL;  (* Boolean, to bind to digital output *)
    {attribute 'OPC.UA.DA' := '1'}
    stat : SimpleRelayStatuses;  (* Statuses of the state machine *)
    {attribute 'OPC.UA.DA' := '1'}
    proc : SimpleRelayProcesses;  (* Processes of the state machine *)
  END_VAR

            stat.busy := F_BusyStatus(
    superState := TRUE,
    isBusy := proc.setEnabled.stat.busy = BusyStatus.busy);
proc.setEnabled( isEnabled := isEnabled AND (proc.setEnabled.stat.busy = BusyStatus.idle) );

          

METHOD _copyFromModel_SM_SimpleRelay
  VAR_IN_OUT
    {attribute 'OPC.UA.DA' := '0'}
    model : M_SM_SimpleRelay;
  END_VAR
                  THIS^.proc.setEnabled._copyFromModel_SetEnabledProcess( model := model.proc.setEnabled );

                
END_METHOD

METHOD _copyToModel_SM_SimpleRelay
  VAR_IN_OUT
    {attribute 'OPC.UA.DA' := '0'}
    model : M_SM_SimpleRelay;
  END_VAR
                  model.actualStatus := THIS^.actualStatus;
model.digitalOutput := THIS^.digitalOutput;
model.stat := THIS^.stat;
THIS^.proc.setEnabled._copyToModel_SetEnabledProcess( model := model.proc.setEnabled );

                
END_METHOD
END_FUNCTION_BLOCK

FUNCTION_BLOCK SM_Fuse
  VAR_INPUT
    {attribute 'OPC.UA.DA' := '1'}
    {attribute 'OPC.UA.DA.Access' := '1'}
    enabled AT %I* : BOOL;  (* Is the fuse on? *)
    {attribute 'OPC.UA.DA' := '1'}
    {attribute 'OPC.UA.DA.Access' := '1'}
    tripped AT %I* : BOOL;  (* Is the fuse tripped? *)
    {attribute 'OPC.UA.DA' := '1'}
    {attribute 'OPC.UA.DA.Access' := '1'}
    overload AT %I* : BOOL;  (* Is the fuse overloaded? *)
    {attribute 'OPC.UA.DA' := '0'}
    isEnabled : BOOL;  (* Is control enabled? *)
  END_VAR
  VAR_OUTPUT
    {attribute 'OPC.UA.DA' := '1'}
    {attribute 'OPC.UA.DA.Access' := '1'}
    actualStatus : STRING(50);  (* Current status description *)
    {attribute 'OPC.UA.DA' := '1'}
    {attribute 'OPC.UA.DA.Access' := '1'}
    resetOutput AT %Q* : BOOL;  (* Reset, to bind to EL9227-5500 *)
    {attribute 'OPC.UA.DA' := '1'}
    {attribute 'OPC.UA.DA.Access' := '1'}
    switchOutput AT %Q* : BOOL;  (* Switch, to bind to EL9227-5500 *)
    {attribute 'OPC.UA.DA' := '1'}
    stat : FuseStatuses;  (* Statuses of the state machine *)
    {attribute 'OPC.UA.DA' := '1'}
    proc : FuseProcesses;  (* Processes of the state machine *)
  END_VAR

            stat.busy := F_BusyStatus(
    superState := TRUE,
    isBusy := (proc.setEnabled.stat.busy = BusyStatus.busy) OR (proc.reset.stat.busy = BusyStatus.busy));
stat.health := F_HealthStatus(
    superState := TRUE,
    hasWarning := overload,
    isGood := NOT(tripped));
proc.setEnabled( isEnabled := isEnabled AND (proc.setEnabled.stat.busy = BusyStatus.idle) );
proc.reset( isEnabled := isEnabled AND ((proc.reset.stat.busy = BusyStatus.idle) AND tripped) );

          

METHOD _copyFromModel_SM_Fuse
  VAR_IN_OUT
    {attribute 'OPC.UA.DA' := '0'}
    model : M_SM_Fuse;
  END_VAR
                  THIS^.proc.setEnabled._copyFromModel_SetEnabledProcess( model := model.proc.setEnabled );
THIS^.proc.reset._copyFromModel_Process( model := model.proc.reset );

                
END_METHOD

METHOD _copyToModel_SM_Fuse
  VAR_IN_OUT
    {attribute 'OPC.UA.DA' := '0'}
    model : M_SM_Fuse;
  END_VAR
                  model.enabled := THIS^.enabled;
model.tripped := THIS^.tripped;
model.overload := THIS^.overload;
model.actualStatus := THIS^.actualStatus;
model.resetOutput := THIS^.resetOutput;
model.switchOutput := THIS^.switchOutput;
model.stat := THIS^.stat;
THIS^.proc.setEnabled._copyToModel_SetEnabledProcess( model := model.proc.setEnabled );
THIS^.proc.reset._copyToModel_Process( model := model.proc.reset );

                
END_METHOD
END_FUNCTION_BLOCK

FUNCTION_BLOCK SM_Led
  VAR_INPUT
    {attribute 'OPC.UA.DA' := '0'}
    isEnabled : BOOL;  (* Is control enabled? *)
  END_VAR
  VAR_OUTPUT
    {attribute 'OPC.UA.DA' := '1'}
    {attribute 'OPC.UA.DA.Access' := '1'}
    actualStatus : STRING(50);  (* Current status description *)
    {attribute 'OPC.UA.DA' := '1'}
    {attribute 'OPC.UA.DA.Access' := '1'}
    milliAmps : LREAL;  (* Actual output in milli amps *)
    {attribute 'OPC.UA.DA' := '1'}
    {attribute 'OPC.UA.DA.Access' := '1'}
    relayOn : BOOL;  (* In case the wires are passing through a relay, is the relay actuated? *)
    {attribute 'OPC.UA.DA' := '1'}
    stat : LedStatuses;  (* Statuses of the state machine *)
    {attribute 'OPC.UA.DA' := '1'}
    proc : LedProcesses;  (* Processes of the state machine *)
  END_VAR

            stat.busy := F_BusyStatus(
    superState := TRUE,
    isBusy := proc.setMilliAmps.stat.busy = BusyStatus.busy);
proc.setMilliAmps( isEnabled := isEnabled AND (proc.setMilliAmps.stat.busy = BusyStatus.idle) );

          

METHOD _copyFromModel_SM_Led
  VAR_IN_OUT
    {attribute 'OPC.UA.DA' := '0'}
    model : M_SM_Led;
  END_VAR
                  THIS^.proc.setMilliAmps._copyFromModel_ChangeSetpointProcess( model := model.proc.setMilliAmps );

                
END_METHOD

METHOD _copyToModel_SM_Led
  VAR_IN_OUT
    {attribute 'OPC.UA.DA' := '0'}
    model : M_SM_Led;
  END_VAR
                  model.actualStatus := THIS^.actualStatus;
model.milliAmps := THIS^.milliAmps;
model.relayOn := THIS^.relayOn;
model.stat := THIS^.stat;
THIS^.proc.setMilliAmps._copyToModel_ChangeSetpointProcess( model := model.proc.setMilliAmps );

                
END_METHOD
END_FUNCTION_BLOCK

FUNCTION_BLOCK SM_TipTilt
  VAR_INPUT
    {attribute 'OPC.UA.DA' := '0'}
    isEnabled : BOOL;  (* Is control enabled? *)
    {attribute 'OPC.UA.DA' := '0'}
    isSimulated : BOOL;  (* Is the TipTilt simulated? *)
  END_VAR
  VAR_OUTPUT
    {attribute 'OPC.UA.DA' := '1'}
    {attribute 'OPC.UA.DA.Access' := '1'}
    actualStatus : STRING(50);  (* Current status description *)
    {attribute 'OPC.UA.DA' := '1'}
    {attribute 'OPC.UA.DA.Access' := '1'}
    v1 : LREAL;  (* Actual output 1 in voltage *)
    {attribute 'OPC.UA.DA' := '1'}
    {attribute 'OPC.UA.DA.Access' := '1'}
    v2 : LREAL;  (* Actual output 2 in voltage *)
    {attribute 'OPC.UA.DA' := '1'}
    {attribute 'OPC.UA.DA.Access' := '1'}
    v3 : LREAL;  (* Actual output 3 in voltage *)
    {attribute 'OPC.UA.DA' := '1'}
    stat : TipTiltStatuses;  (* Statuses of the state machine *)
    {attribute 'OPC.UA.DA' := '1'}
    proc : TipTiltProcesses;  (* Processes of the state machine *)
  END_VAR

            stat.busy := F_BusyStatus(
    superState := TRUE,
    isBusy := (proc.setV1.stat.busy = BusyStatus.busy) OR ((proc.setV2.stat.busy = BusyStatus.busy) OR (proc.setV3.stat.busy = BusyStatus.busy)));
proc.setV1( isEnabled := isEnabled AND (proc.setV1.stat.busy = BusyStatus.idle) );
proc.setV2( isEnabled := isEnabled AND (proc.setV2.stat.busy = BusyStatus.idle) );
proc.setV3( isEnabled := isEnabled AND (proc.setV3.stat.busy = BusyStatus.idle) );

          

METHOD _copyFromModel_SM_TipTilt
  VAR_IN_OUT
    {attribute 'OPC.UA.DA' := '0'}
    model : M_SM_TipTilt;
  END_VAR
                  THIS^.proc.setV1._copyFromModel_ChangeSetpointProcess( model := model.proc.setV1 );
THIS^.proc.setV2._copyFromModel_ChangeSetpointProcess( model := model.proc.setV2 );
THIS^.proc.setV3._copyFromModel_ChangeSetpointProcess( model := model.proc.setV3 );

                
END_METHOD

METHOD _copyToModel_SM_TipTilt
  VAR_IN_OUT
    {attribute 'OPC.UA.DA' := '0'}
    model : M_SM_TipTilt;
  END_VAR
                  model.actualStatus := THIS^.actualStatus;
model.v1 := THIS^.v1;
model.v2 := THIS^.v2;
model.v3 := THIS^.v3;
model.stat := THIS^.stat;
THIS^.proc.setV1._copyToModel_ChangeSetpointProcess( model := model.proc.setV1 );
THIS^.proc.setV2._copyToModel_ChangeSetpointProcess( model := model.proc.setV2 );
THIS^.proc.setV3._copyToModel_ChangeSetpointProcess( model := model.proc.setV3 );

                
END_METHOD
END_FUNCTION_BLOCK

FUNCTION_BLOCK SM_ConfigManager
  VAR_INPUT
    {attribute 'OPC.UA.DA' := '1'}
    {attribute 'OPC.UA.DA.Access' := '1'}
    filePath : STRING(30);  (* Full path of the config filename *)
    {attribute 'OPC.UA.DA' := '0'}
    isEnabled : BOOL;  (* Is control enabled? *)
  END_VAR
  VAR_OUTPUT
    {attribute 'OPC.UA.DA' := '1'}
    {attribute 'OPC.UA.DA.Access' := '1'}
    actualStatus : STRING(50);  (* Current status description *)
    {attribute 'OPC.UA.DA' := '1'}
    stat : ConfigManagerStatuses;  (* Statuses of the state machine *)
    {attribute 'OPC.UA.DA' := '1'}
    proc : ConfigManagerProcesses;  (* Processes of the state machine *)
  END_VAR

            stat.busy := F_BusyStatus(
    superState := TRUE,
    isBusy := (proc.save.stat.busy = BusyStatus.busy) OR ((proc.load.stat.busy = BusyStatus.busy) OR (proc.activate.stat.busy = BusyStatus.busy)));
stat.health := F_HealthStatus(
    superState := TRUE,
    isGood := ((proc.save.stat.health = HealthStatus.good) OR (proc.save.stat.health = HealthStatus.warning)) AND (((proc.load.stat.health = HealthStatus.good) OR (proc.load.stat.health = HealthStatus.warning)) AND ((proc.activate.stat.health = HealthStatus.good) OR (proc.activate.stat.health = HealthStatus.warning))),
    hasWarning := (proc.save.stat.health = HealthStatus.warning) OR ((proc.load.stat.health = HealthStatus.warning) OR (proc.activate.stat.health = HealthStatus.warning)));
proc.save( isEnabled := isEnabled AND (stat.busy = BusyStatus.idle) );
proc.load( isEnabled := isEnabled AND (stat.busy = BusyStatus.idle) );
proc.activate( isEnabled := isEnabled AND (stat.busy = BusyStatus.idle) );

          

